Omron CX-Programmer project 新工程 (CX-Programmer 9.61)

# PLC 负压入盘机: CJ2M CPU33
I/O table (CPU CJ2M-CPU33): rack 0 slot 0 CJ1W-SCU21-V1; rack 0 slot 1 CJ1W-NC413; rack 0 slot 2 CJ1W-ID261; rack 0 slot 3 CJ1W-ID261; rack 0 slot 4 CJ1W-ID261; rack 0 slot 5 CJ1W-OD261; rack 0 slot 6 CJ1W-OD231; rack 0 slot 11 CJ2M-EIP21

## Global symbols (name address type ; comment)
17.10 BOOL  ; 料盘夹紧气缸伸出
2.13 BOOL  ; 料盒夹紧气缸伸出到位
0.00 BOOL  ; #3检漏仪行程1
0.01 BOOL  ; 上料有料感应
0.02 BOOL  ; 移栽前电池到位
0.03 BOOL  ; 移栽后电池到位
0.04 BOOL  ; #1模组左电池感应
0.05 BOOL  ; #1模组右电池感应
0.06 BOOL  ; #2模组左电池感应
0.07 BOOL  ; #2模组右电池感应
0.08 BOOL  ; #3模组左电池感应
0.09 BOOL  ; #3模组右电池感应
0.10 BOOL  ; #4模组左电池感应
0.11 BOOL  ; #4模组右电池感应
0.12 BOOL  ; #2空料盒到位感应
0.13 BOOL  ; 上料盒完成按钮（左）
0.14 BOOL  ; 龙门升降料盒到位
0.15 BOOL  ; #2满料盒到位感应
1000 CHANNEL  ; 移栽自动步序
1000.00 BOOL  ; 移栽机构在初始位
1000.15 BOOL  ; 移栽自动运行结束(步)
100.00 BOOL  ; 前门已打开
100.01 BOOL  ; 后门已打开
100.02 BOOL  ; 左侧门已打开
100.03 BOOL  ; 右侧门已打开
100.04 BOOL  ; 电脑未连接
100.05 BOOL  ; 进料移栽没归零
100.06 BOOL  ; 左机械手没归零
100.07 BOOL  ; 右机械手没归零
100.08 BOOL  ; 龙门升降伺服没归零
100.09 BOOL  ; 龙门前后伺服没归零
100.10 BOOL  ; 龙门左右伺服没归零
100.11 BOOL  ; 料盒升降伺服没归零
100.12 BOOL  ; 右机械手左夹爪有料但没夹紧
100.13 BOOL  ; 右机械手左夹爪没张开
100.14 BOOL  ; 右机械手右夹爪有料但没夹紧
100.15 BOOL  ; 右机械手右夹爪没张开
101.00 BOOL  ; 左机械手左夹爪有料但没夹紧
101.01 BOOL  ; 左机械手左夹爪没张开
101.02 BOOL  ; 左机械手右夹爪有料但没夹紧
101.03 BOOL  ; 左机械手右夹爪没张开
101.04 BOOL  ; #1模组左密封气缸没缩回
101.05 BOOL  ; #1模组右密封气缸没缩回
101.06 BOOL  ; #1模组左夹料气缸没松开
101.07 BOOL  ; #1模组右夹料气缸没松开
101.08 BOOL  ; #2模组左密封气缸没缩回
101.09 BOOL  ; #2模组右密封气缸没缩回
101.10 BOOL  ; #2模组左夹料气缸没松开
101.11 BOOL  ; #2模组右夹料气缸没松开
101.12 BOOL  ; #3模组左密封气缸没缩回
101.13 BOOL  ; #3模组右密封气缸没缩回
101.14 BOOL  ; #3模组左夹料气缸没松开
101.15 BOOL  ; #3模组右夹料气缸没松开
1020.00 BOOL  ; 移栽机构有错误
102.00 BOOL  ; #4模组左密封气缸没缩回
102.01 BOOL  ; #4模组右密封气缸没缩回
102.02 BOOL  ; #4模组左夹料气缸没松开
102.03 BOOL  ; #4模组右夹料气缸没松开
102.04 BOOL  ; 龙门夹爪没张开
102.05 BOOL  ; 龙门夹爪有料但没夹紧
103.00 BOOL  ; 移栽归零左机械手异常
103.01 BOOL  ; 移栽归零右机械手异常
103.02 BOOL  ; 移栽左移左机械手异常
103.03 BOOL  ; 移栽左移没归零异常
103.04 BOOL  ; 移栽左移左限位到达异常
103.05 BOOL  ; 移栽右移右机械手异常
103.06 BOOL  ; 移栽右移没归零异常
103.07 BOOL  ; 移栽右移右限位到达异常
103.08 BOOL  ; 移栽回进料位条件异常
103.09 BOOL  ; 移栽回进料位没归零异常
103.10 BOOL  ; 移栽回左下料位条件异常
103.11 BOOL  ; 移栽回左下料位没归零异常
103.12 BOOL  ; 移栽回右下料位条件异常
103.13 BOOL  ; 移栽回右下料没归零
104.00 BOOL  ; 左机械手升降气缸没缩回异常
104.01 BOOL  ; 左机械手伸缩气缸没缩回异常
104.02 BOOL  ; 左机械手没归零异常
104.03 BOOL  ; 伸缩气缸伸出异常
104.04 BOOL  ; 升降气缸伸出异常
104.05 BOOL  ; 左机械手夹爪松开升降气缸异常
104.06 BOOL  ; 左机械手夹爪松开伸缩气缸异常
104.07 BOOL  ; 左机械手左夹爪松开伸缩气缸异常
104.08 BOOL  ; 左机械手右夹爪松开升降气缸异常
104.09 BOOL  ; 左机械手右夹爪松开伸缩气缸异常
105.00 BOOL  ; 机械手升降气缸没缩回异常
105.01 BOOL  ; 右机械手伸缩气缸没缩回异常
105.02 BOOL  ; 右机械手没归零异常
105.03 BOOL  ; 伸缩气缸伸出异常
105.04 BOOL  ; 升降气缸伸出异常
105.05 BOOL  ; 右机械手夹爪松开升降气缸异常
106.00 BOOL  ; #1左密封气缸没缩回异常
106.01 BOOL  ; #1右密封气缸没缩回异常
106.04 BOOL  ; #2左密封气缸没缩回异常
106.05 BOOL  ; #2右密封气缸没缩回异常
106.08 BOOL  ; #3左密封气缸没缩回异常
106.09 BOOL  ; #3右密封气缸没缩回异常
106.12 BOOL  ; #4左密封气缸没缩回异常
106.13 BOOL  ; #4右密封气缸没缩回异常
107.00 BOOL  ; 龙门升降气缸没缩回异常
107.01 BOOL  ; 伺服没归零异常
107.02 BOOL  ; 料盒定位气缸没缩回
107.03 BOOL  ; 料盒升降下料处有料异常
107.04 BOOL  ; 伺服没归零异常
107.05 BOOL  ; 左、右脱离气缸没缩回异常
107.06 BOOL  ; 龙门升降气缸没缩回异常
107.07 BOOL  ; 龙门升降伺服不在原位
107.08 BOOL  ; 龙门前后、左右伺服没归零异常
107.09 BOOL  ; 龙门升降夹爪松开异常
107.10 BOOL  ; 此位有电池夹爪没打开不能下降
108.00 BOOL  ; 龙门升降气缸没缩回异常
10.00 BOOL  ; #1上顶升左气缸缩回位
10.01 BOOL  ; #1上顶升左气缸伸出位
10.02 BOOL  ; #1上顶升右气缸缩回位
10.03 BOOL  ; #1上顶升右气缸伸出位
10.04 BOOL  ; #2上顶升左气缸缩回位
10.05 BOOL  ; #2上顶升左气缸伸出位
10.06 BOOL  ; #2上顶升右气缸缩回位
10.07 BOOL  ; #2上顶升右气缸伸出位
10.08 BOOL  ; #1下顶升左气缸缩回位
10.09 BOOL  ; #1下顶升左气缸伸出位
10.10 BOOL  ; #1下顶升右气缸缩回位
10.11 BOOL  ; #1下顶升右气缸伸出位
10.12 BOOL  ; #2下顶升左气缸缩回位
10.13 BOOL  ; #2下顶升左气缸伸出位
10.14 BOOL  ; #2下顶升右气缸缩回位
10.15 BOOL  ; #2下顶升右气缸伸出位
11.00 BOOL  ; 叉车退出上对射
11.01 BOOL  ; 叉车退出下对射
11.02 BOOL  ; 右按钮（叉车伸出上到位）
11.03 BOOL  ; #1空料盒到位感应
11.04 BOOL  ; #2检漏仪行程1
11.05 BOOL  ; #2检漏仪行程0
11.06 BOOL  ; 上料盒区域1感应
11.07 BOOL  ; #2料盒区域感应
11.08 BOOL  ; 左拉带脱离气缸缩回位
11.09 BOOL  ; 左拉带脱离气缸伸出位
11.10 BOOL  ; 右拉带脱离气缸缩回位
11.11 BOOL  ; 右拉带脱离气缸伸出位
11.12 BOOL  ; 左#2放料电池感应
11.13 BOOL  ; 左#1放料电池感应
11.14 BOOL  ; 右#1放料电池感应
11.15 BOOL  ; 右#2放料电池感应
120.00 BOOL  ; 上料机构复位
120.01 BOOL  ; 上料机构在初始位
120.04 BOOL  ; 上料机构异常复位
120.05 BOOL  ; 上料机构异常复位完成
121.00 BOOL  ; 移栽机构复位
121.01 BOOL  ; 移栽伺服归零
121.02 BOOL  ; 移栽伺服到进料位置(复位)
121.03 BOOL  ; 移栽机构在初始位
121.04 BOOL  ; 移栽机构异常复位
121.05 BOOL  ; 移栽伺服异常归零
121.06 BOOL  ; 移栽伺服异常后到进料位置
121.07 BOOL  ; 移栽机构异常复位完成
121.10 BOOL  ; 龙门升降伺服异常复位
121.11 BOOL  ; 龙门升降伺服异常复位归零
121.12 BOOL  ; 龙门升降伺服异常归零后回上料盒位置
122.00 BOOL  ; 左机械手整机复位
122.01 BOOL  ; 左机械手伺服归零
122.02 BOOL  ; 左机械手回上料位(复位)
122.03 BOOL  ; 左机械手在初始位
122.04 BOOL  ; 左机械手异常复位
122.05 BOOL  ; 左机械手伺服异常归零
122.06 BOOL  ; 左机械手异常后回上料位
122.07 BOOL  ; 左机械手复位完成
123.00 BOOL  ; 右机械手复位
123.01 BOOL  ; 右机械手伺服归零
123.02 BOOL  ; 右机械手回上料位(复位)
123.03 BOOL  ; 右机械手在初始位
123.04 BOOL  ; 右机械手异常复位
123.05 BOOL  ; 右机械手伺服异常归零
123.06 BOOL  ; 右机械手伺服异常归零后回上料位
123.07 BOOL  ; 右机械手异常复位完成
124.00 BOOL  ; #1模组复位
124.01 BOOL  ; #1模组在初始位
124.02 BOOL  ; #2模组复位
124.03 BOOL  ; #2模组在初始位
124.04 BOOL  ; #3模组复位
124.05 BOOL  ; #3模组在初始位
124.06 BOOL  ; #4模组复位
124.07 BOOL  ; #4模组在初始位
124.08 BOOL  ; #1模组异常复位
124.09 BOOL  ; #1模组异常复位完成
124.10 BOOL  ; #2模组异常复位
124.11 BOOL  ; #2模组异常复位完成
124.12 BOOL  ; #3模组异常复位
124.13 BOOL  ; #3模组异常复位完成
124.14 BOOL  ; #4模组异常复位
124.15 BOOL  ; #4模组异常复位完成
125.00 BOOL  ; 龙门升降机构复位
125.01 BOOL  ; 龙门升降归零(复位)
125.02 BOOL  ; 龙门升降机构在初始位
125.03 BOOL  ; 龙门前后，左右复位
125.04 BOOL  ; 龙门前后伺服归零(复位)
125.05 BOOL  ; 龙门左右伺服归零(复位）
125.06 BOOL  ; 龙门前后，左右在初始位
125.08 BOOL  ; 龙门机构复位
125.09 BOOL  ; 料盒升降伺服整机归零
125.10 BOOL  ; 料盒升降回上料盒位置
125.11 BOOL  ; 龙门机构在初始位置
126.00 BOOL  ; 龙门升降异常复位
126.01 BOOL  ; 龙门升降伺服异常归零
126.02 BOOL  ; 龙门升降异常复位完成
126.05 BOOL  ; 龙门前后，左右异常复位
126.06 BOOL  ; 龙门前后异常复位归零
126.07 BOOL  ; 龙门左右异常复位归零
126.08 BOOL  ; 龙门前后，左右伺服异常复位完成
126.09 BOOL  ; 龙门升降伺服异常复位
126.10 BOOL  ; 料盒升降伺服异常复位归零
126.11 BOOL  ; 料盒升降伺服异常归零后回上料盒位置
126.12 BOOL  ; 料盒升降伺服异常复位完成
126.13 BOOL  ; 龙门机构异常复位
126.14 BOOL  ; 龙门机构异常复位完成
12.00 BOOL  ; 上料阻挡气缸
12.01 BOOL  ; 检测气缸
12.02 BOOL  ; 移栽阻挡气缸
12.03 BOOL  ; 左机械手升降气缸
12.04 BOOL  ; 左机械手伸缩气缸
12.05 BOOL  ; 左机械手左夹爪气缸
12.06 BOOL  ; 左机械手右夹爪气缸
12.07 BOOL  ; 右机械手升降气缸
12.08 BOOL  ; 右机械手伸缩气缸
12.09 BOOL  ; 右机械手左夹爪气缸
12.10 BOOL  ; 右机械手右夹爪气缸
12.11 BOOL  ; #1模组左夹料气缸
12.12 BOOL  ; #1模组右夹料气缸
12.13 BOOL  ; #1模组左密封气缸
12.14 BOOL  ; #1模组右密封气缸
12.15 BOOL  ; #1自检左气缸
134.15 BOOL  ; 移栽机构复位(M)
13.00 BOOL  ; #1自检右气缸
13.01 BOOL  ; #2模组左夹料气缸
13.02 BOOL  ; #2模组右夹料气缸
13.03 BOOL  ; #2模组左密封气缸
13.04 BOOL  ; #2模组右密封气缸
13.05 BOOL  ; #2自检左气缸
13.06 BOOL  ; #2自检右气缸
13.07 BOOL  ; #3左夹料气缸
13.08 BOOL  ; #3右夹料气缸
13.09 BOOL  ; #3左密封气缸
13.10 BOOL  ; #3右密封气缸
13.11 BOOL  ; #3自检左气缸
13.12 BOOL  ; #3自检右气缸
13.13 BOOL  ; #4左夹料气缸
13.14 BOOL  ; #4右夹料气缸
13.15 BOOL  ; #4左密封气缸
1404 CHANNEL  ; 第二排放料位置
1410.00 BOOL  ; 移栽机构在初始位
1410.01 BOOL  ; 前上料伺服在待机位置
1411.00 BOOL  ; 移栽机构有错误
1417 CHANNEL  ; 移栽自动步序
1417.15 BOOL  ; 移栽自动运行结束(步)
14.00 BOOL  ; #4右密封气缸
14.01 BOOL  ; #4自检左气缸
14.02 BOOL  ; #4自检右气缸
14.03 BOOL  ; 龙门#1上顶升气缸
14.04 BOOL  ; 龙门#2上顶升气缸
14.05 BOOL  ; #1下顶升气缸
14.06 BOOL  ; #2下顶升气缸
14.07 BOOL  ; 龙门料盒阻挡气缸
14.10 BOOL  ; 料盒定位气缸
14.11 BOOL  ; 龙门升降气缸
14.12 BOOL  ; 龙门夹爪气缸
14.13 BOOL  ; #1移栽电机
14.14 BOOL  ; #2移栽电机
14.15 BOOL  ; 检漏NG电机
1534.15 BOOL  ; 单元1的串口1协议执行标志
15.00 BOOL  ; 绝缘NG电机
15.01 BOOL  ; 料盒下料电机
15.02 BOOL  ; 下料缓存电机
15.03 BOOL  ; 料盒上料电机
15.04 BOOL  ; 真空泵
15.05 BOOL  ; 检测气缸
15.06 BOOL  ; 绝缘检测仪启动信号
15.07 BOOL  ; #1检漏仪启动
15.09 BOOL  ; #2检漏仪启动
15.11 BOOL  ; #3检漏仪启动
15.13 BOOL  ; #4检漏仪启动
15.14 BOOL  ; #4检漏仪启动
15.15 BOOL  ; 启动指示灯
16.00 BOOL  ; 停止指示灯
16.01 BOOL  ; 复位指示灯
16.02 BOOL  ; 三色绿灯
16.03 BOOL  ; 三色红灯
16.04 BOOL  ; 三色黄灯
16.05 BOOL  ; 蜂鸣器
16.06 BOOL  ; 移栽Serv_ON
16.08 BOOL  ; 左机械手Serv_ON
16.09 BOOL  ; 报警声关
16.10 BOOL  ; 右机械手Serv_ON
16.12 BOOL  ; 龙门升降Serv-ON
16.14 BOOL  ; 龙门左右Serv_ON
17.00 BOOL  ; 龙门前后Serv_ON
17.02 BOOL  ; 料盒Serv-ON
17.04 BOOL  ; 左拉带脱离气缸
17.05 BOOL  ; 右拉带脱离气缸
17.06 BOOL  ; 龙门升降刹车
17.07 BOOL  ; 料盒升降刹车
17.11 BOOL  ; 料盘夹紧气缸松开
18.00 BOOL  ; 扫描NG提示
19.00 BOOL  ; 左机械手左夹爪状态
19.01 BOOL  ; 左机械手右夹爪状态
19.02 BOOL  ; 右机械手左夹爪状态
19.03 BOOL  ; 右机械手右夹爪状态
1.00 BOOL  ; #1满料盒到位感应
1.01 BOOL  ; 入电池位料盒感应
1.02 BOOL  ; 料盒#1电池感应
1.03 BOOL  ; 料盒#2电池感应
1.04 BOOL  ; 料盒#3电池感应
1.05 BOOL  ; 料盒#4电池感应
1.06 BOOL  ; 料盒#5电池感应
1.07 BOOL  ; 料盒#6电池感应
1.08 BOOL  ; 料盒#7电池感应
1.09 BOOL  ; 料盒#8电池感应
1.10 BOOL  ; 料盒#9电池感应
1.11 BOOL  ; 料盒#10电池感应
1.12 BOOL  ; 料盒#11电池感应
1.13 BOOL  ; 料盒#12电池感应
1.14 BOOL  ; 料盒#13电池感应
1.15 BOOL  ; 料盒#14电池感应
2000.03 BOOL  ; 龙门前后绝对移动
2000.06 BOOL  ; 龙门前后归零
2000.09 BOOL  ; 龙门前后点动
2000.10 BOOL  ; 龙门前后方向
2000.12 BOOL  ; 龙门前后模块复位
2000.15 BOOL  ; 龙门前后停止
2002.03 BOOL  ; 龙门左右绝对运动
2002.06 BOOL  ; 龙门左右归零
2002.09 BOOL  ; 龙门左右点动
2002.10 BOOL  ; 龙门左右方向
2002.12 BOOL  ; 龙门左右模块复位
2002.15 BOOL  ; 龙门左右伺服停止
2004.03 BOOL  ; 料盒升降绝对移动
2004.06 BOOL  ; 料盒升降归零
2004.09 BOOL  ; 料盒升降点动
2004.10 BOOL  ; 料盒升降方向
2004.12 BOOL  ; 料盒升降模块复位
2004.15 BOOL  ; 料盒升降停止
2008.06 BOOL  ; 龙门前后无原点标志
2008.12 BOOL  ; 龙门前后模块有错误
2008.13 BOOL  ; 龙门前后忙标志
2009.08 BOOL  ; 龙门前后伺服前限位
2009.09 BOOL  ; 龙门前后伺服后限位
2009.10 BOOL  ; 前后近原点
2009.11 BOOL  ; 前后原点
200.00 BOOL  ; 复位位
2010 CHANNEL  ; 龙门前后轴错误代码
2011.06 BOOL  ; 龙门左右无原点标志
2011.12 BOOL  ; 龙门左右模块有错误
2011.13 BOOL  ; 龙门左右忙标志
2012.08 BOOL  ; 龙门左右伺服右限位
2012.09 BOOL  ; 龙门左右伺服左限位
2012.11 BOOL  ; 龙门左右原点
2013 CHANNEL  ; 龙门左右轴错误代码
2014.06 BOOL  ; 料盒升降无原点标志
2014.12 BOOL  ; 料盒升降模块有错误
2014.13 BOOL  ; 料盒升降忙标志
2015.08 BOOL  ; 料盒升降下限位
2015.09 BOOL  ; 料盒升降上限位
2016 CHANNEL  ; 料盒升降轴错误代码
20.00 BOOL  ; 移栽伺服手动回进料位置
20.01 BOOL  ; 移栽伺服手动回左下料位置
20.02 BOOL  ; 移栽伺服手动回右下料位置
20.03 BOOL  ; 移栽自动回右下料位
20.04 BOOL  ; 移栽自动回左下料位
20.05 BOOL  ; 移栽自动回上料位
21.00 BOOL  ; #1模组可放料
21.01 BOOL  ; #2模组可放料
21.02 BOOL  ; #3模组可放料
21.03 BOOL  ; #4模组可放料
21.04 BOOL  ; 回右下料位条件
21.05 BOOL  ; 回左下料位条件
22.00 BOOL  ; 左机械手上料位伸缩气缸伸出条件
22.01 BOOL  ; 左机械手下料位伸缩气缸伸出条件
22.02 BOOL  ; 左机械手#2模组伸缩气缸伸出条件
22.03 BOOL  ; 左机械手#4模组伸缩气缸伸出条件
22.04 BOOL  ; 左机械手伸缩气缸伸出条件
22.05 BOOL  ; 左机械手手动回上料位置
22.06 BOOL  ; 左机械手回下料位置
22.07 BOOL  ; 左机械手回#2位置
22.08 BOOL  ; 左机械手回#4位置
22.09 BOOL  ; 左机械手自动回上料位置
22.10 BOOL  ; 左机械手自动回#2位置
22.11 BOOL  ; 左机械手自动回#4位置
22.12 BOOL  ; 左机械手自动回下料位置
23 CHANNEL  ; 左机械手状态
235.02 BOOL  ; 右机械手升降气缸缩回
23.00 BOOL  ; 左机械手左夹爪上料处夹紧电池
23.01 BOOL  ; 左机械手上料处右夹爪夹紧到位
23.02 BOOL  ; 左机械手#2左放料
23.03 BOOL  ; 左机械手#4左放料
23.04 BOOL  ; 左机械手#2右放料
23.05 BOOL  ; 左机械手#4右放料
23.06 BOOL  ; 左机械手#2左取料
23.07 BOOL  ; 左机械手#2右取料
23.08 BOOL  ; 左机械手#4左取料
23.09 BOOL  ; 左机械手#4右取料
23.10 BOOL  ; 左机械手左夹爪有料状态
23.11 BOOL  ; 左机械手右夹爪有料状态
23.12 BOOL  ; 左机械手左夹爪模组放料完成
23.13 BOOL  ; 左机械手右夹爪模组放料完成
23.14 BOOL  ; 左机械手左夹爪上料处夹紧电池
23.15 BOOL  ; 左机械手上料处右夹爪夹紧到位
24.00 BOOL  ; 右机械手上料位伸缩气缸伸出条件
24.01 BOOL  ; 右机械手下料位伸缩气缸伸出条件
24.02 BOOL  ; 右机械手#1模组伸缩气缸伸出条件
24.03 BOOL  ; 右机械手#3模组伸缩气缸伸出条件
24.04 BOOL  ; 右机械手伸缩气缸伸出条件
24.05 BOOL  ; 右机械手手动回上料位置
24.06 BOOL  ; 右机械手回下料位置
24.07 BOOL  ; 右机械手回#1位置
24.08 BOOL  ; 右机械手回#3位置
24.09 BOOL  ; 右机械手自动回上料位置
24.10 BOOL  ; 右机械手自动回#1位置
24.11 BOOL  ; 右机械手回#3位置
24.12 BOOL  ; 右机械手自动回下料位
25 CHANNEL  ; 右机械手状态
25.00 BOOL  ; 右机械手右夹爪上料处夹紧电池
25.01 BOOL  ; 右机械手上料处左夹爪夹紧到位
25.02 BOOL  ; 右机械手#1左放料
25.03 BOOL  ; 右机械手#3左放料
25.04 BOOL  ; 右机械手#1右放料
25.05 BOOL  ; 右机械手#3右放料
25.06 BOOL  ; 右机械手#1左取料
25.07 BOOL  ; 右机械手#1右取料
25.08 BOOL  ; 右机械手#3左取料
25.09 BOOL  ; 右机械手#3右取料
25.10 BOOL  ; 右机械手左夹爪有料状态
25.11 BOOL  ; 右机械手右夹爪有料状态
25.12 BOOL  ; 右机械手左夹爪模组放料完成
25.13 BOOL  ; 右机械手右夹爪模组放料完成
25.14 BOOL  ; 右机械手右夹爪上料处夹紧电池
25.15 BOOL  ; 右机械手上料处左夹爪夹紧到位
2960.06 BOOL  ; 移栽伺服左限位
2960.07 BOOL  ; 移栽伺服右限位
2960.08 BOOL  ; 左机械手左限位
2960.09 BOOL  ; 左机械手右限位
2962.02 BOOL  ; 龙门升降原位
2962.06 BOOL  ; 右机械手左限位
2962.07 BOOL  ; 右机械手右限位
2962.08 BOOL  ; 龙门升降上限位
2962.09 BOOL  ; 龙门升降下限位
2.00 BOOL  ; 料盒#15电池感应
2.01 BOOL  ; 料盒#16电池感应
2.02 BOOL  ; 料盒#17电池感应
2.03 BOOL  ; 料盒#18电池感应
2.04 BOOL  ; 料盒#19电池感应
2.05 BOOL  ; 料盒#20电池感应
2.06 BOOL  ; 料盒#21电池感应
2.07 BOOL  ; 料盒#22电池感应
2.08 BOOL  ; 料盒#23电池感应
2.09 BOOL  ; 料盒#24电池感应
2.10 BOOL  ; 拉倒衔接处有料
2.11 BOOL  ; #1检漏仪行程1
2.12 BOOL  ; #1检漏仪行程0
2.14 BOOL  ; 绝缘NG放料位有料感应
2.15 BOOL  ; 检漏NG满
30.00 BOOL  ; #1检漏仪抽气临结束状态
30.01 BOOL  ; #2检漏仪抽气临结束状态
30.02 BOOL  ; #3检漏仪抽气临结束状态
30.03 BOOL  ; #4检漏仪抽气临结束状态
30.04 BOOL  ; #1#3模组不在抽气临结束状态
30.05 BOOL  ; #2#4模组不在抽气临结束状态
30.06 BOOL  ; #1模组在保压状态
30.07 BOOL  ; #1模组在保压1秒范围
30.08 BOOL  ; #1仪器抽气状态
311.00 BOOL  ; 整机复位条件
311.01 BOOL  ; 整机复位
311.02 BOOL  ; 整机在初始位
311.03 BOOL  ; 移栽机构复位
311.04 BOOL  ; 左机械手复位
311.05 BOOL  ; 右机械手复位
311.06 BOOL  ; #1模组异常复位
311.07 BOOL  ; #2模组复位
311.08 BOOL  ; #3模组复位
311.09 BOOL  ; #4模组复位
311.10 BOOL  ; 龙门升降复位
311.11 BOOL  ; 龙门前后，左右复位
311.12 BOOL  ; 龙门机构复位
311.13 BOOL  ; 上料机构复位
311.14 BOOL  ; 整机在初始位
313.00 BOOL  ; 移栽机构异常复位
313.01 BOOL  ; 左机械式异常复位
313.02 BOOL  ; 右机械式异常复位
313.03 BOOL  ; #1模组异常复位
313.04 BOOL  ; #2模组异常复位
313.05 BOOL  ; #3模组异常复位
313.06 BOOL  ; #4模组异常复位
313.07 BOOL  ; 龙门机构异常复位
313.08 BOOL  ; 龙门升降异常复位
313.09 BOOL  ; 龙门前后，左右伺服异常复位
313.10 BOOL  ; 料盒升降伺服异常复位
313.11 BOOL  ; 上料机构异常复位
31.00 BOOL  ; #2检漏仪抽气临结束状态
31.01 BOOL  ; #2检漏仪保压临结束状态
31.02 BOOL  ; #3检漏仪保压临结束状态
31.03 BOOL  ; #4检漏仪保压临结束状态
31.06 BOOL  ; #2模组在保压状态
31.07 BOOL  ; #2模组在保压1秒范围
31.08 BOOL  ; #2仪器抽气状态
32.00 BOOL  ; #3检漏仪抽气临结束状态
32.06 BOOL  ; #3模组在保压状态
32.07 BOOL  ; #3模组在保压1秒范围
32.08 BOOL  ; #3仪器抽气状态
33.00 BOOL  ; #4检漏仪抽气临结束状态
33.06 BOOL  ; #4模组在保压状态
33.07 BOOL  ; #4模组在保压1秒范围
33.08 BOOL  ; #4仪器抽气状态
34.00 BOOL  ; 龙门升降手动回取料位
34.01 BOOL  ; 龙门升降手动回OK放料位
34.02 BOOL  ; 龙门升降手动回绝缘NG位置
34.03 BOOL  ; 龙门升降手动回检漏NG位置
34.04 BOOL  ; 料盒升降伺服回上料盒位置
34.05 BOOL  ; 料盒升降伺服回放料盒位置
34.06 BOOL  ; 龙门升降自动回初始位置
34.07 BOOL  ; 龙门升降自动回取料位
34.08 BOOL  ; 龙门升降自动回OK放料位
34.09 BOOL  ; 龙门升降自动回绝缘NG位置
34.10 BOOL  ; 龙门升降在原始位置
34.11 BOOL  ; 龙门升降自动回检漏NG位置
35.00 BOOL  ; 龙门前后在#1位置
35.01 BOOL  ; 龙门前后在#2位置
35.02 BOOL  ; 龙门前后在#3位置
35.03 BOOL  ; 龙门前后在#4位置
35.04 BOOL  ; 龙门前后在#5位置
35.05 BOOL  ; 龙门前后在#6位置
35.06 BOOL  ; 龙门前后在#7位置
35.07 BOOL  ; 龙门前后在#8位置
35.08 BOOL  ; 龙门前后在#9位置
35.09 BOOL  ; 龙门前后在#10位置
35.10 BOOL  ; 龙门前后在#11位置
35.11 BOOL  ; 龙门前后在#12位置
35.12 BOOL  ; 龙门前后在#13位置
35.13 BOOL  ; 龙门前后在#14位置
35.14 BOOL  ; 龙门前后在#15位置
35.15 BOOL  ; 龙门前后在#16位置
36.00 BOOL  ; 龙门前后在#17位置
36.01 BOOL  ; 龙门前后在#18位置
36.02 BOOL  ; 龙门前后在#19位置
36.03 BOOL  ; 龙门前后在#20位置
36.04 BOOL  ; 龙门前后在#21位置
36.05 BOOL  ; 龙门前后在#22位置
36.06 BOOL  ; 龙门前后在#23位置
36.07 BOOL  ; 龙门前后在#24位置
36.08 BOOL  ; 龙门前后在#1左取料位
36.09 BOOL  ; 龙门前后在#2左取料位
36.10 BOOL  ; 龙门前后在#1右取料位
36.11 BOOL  ; 龙门前后在#2右取料位
36.12 BOOL  ; 龙门前后在绝缘NG位置
36.13 BOOL  ; 龙门前后在检漏NG位置
36.14 BOOL  ; 龙门前后在初始位置
37.00 BOOL  ; 龙门左右在#1位置
37.01 BOOL  ; 龙门左右在#2位置
37.02 BOOL  ; 龙门左右在#3位置
37.03 BOOL  ; 龙门左右在#4位置
37.04 BOOL  ; 龙门左右在#5位置
37.05 BOOL  ; 龙门左右在#6位置
37.06 BOOL  ; 龙门左右在#7位置
37.07 BOOL  ; 龙门左右在#8位置
37.08 BOOL  ; 龙门左右在#9位置
37.09 BOOL  ; 龙门左右在#10位置
37.10 BOOL  ; 龙门左右在#11位置
37.11 BOOL  ; 龙门左右在#12位置
37.12 BOOL  ; 龙门左右在#13位置
37.13 BOOL  ; 龙门左右在#14位置
37.14 BOOL  ; 龙门左右在#15位置
37.15 BOOL  ; 龙门左右在#16位置
38.00 BOOL  ; 龙门左右在#17位置
38.01 BOOL  ; 龙门左右在#18位置
38.02 BOOL  ; 龙门左右在#19位置
38.03 BOOL  ; 龙门左右在#20位置
38.04 BOOL  ; 龙门左右在#21位置
38.05 BOOL  ; 龙门左右在#22位置
38.06 BOOL  ; 龙门左右在#23位置
38.07 BOOL  ; 龙门左右在#24位置
38.08 BOOL  ; 龙门左右在#1左取料位
38.09 BOOL  ; 龙门左右在#2左取料位
38.10 BOOL  ; 龙门左右在#1右取料位
38.11 BOOL  ; 龙门左右在#2右取料位
38.12 BOOL  ; 龙门左右在绝缘NG位置
38.13 BOOL  ; 龙门左右在检漏NG位置
38.14 BOOL  ; 龙门左右在初始位置
39 CHANNEL  ; 龙门XY位置
39.01 BOOL  ; 龙门XY在#1放料位置
39.02 BOOL  ; 龙门XY在#2放料位置
39.03 BOOL  ; 龙门XY在#3放料位置
39.04 BOOL  ; 龙门XY在#4放料位置
39.05 BOOL  ; 龙门XY在#5放料位置
39.06 BOOL  ; 龙门XY在#6放料位置
39.07 BOOL  ; 龙门XY在#7放料位置
39.08 BOOL  ; 龙门XY在#8放料位置
39.09 BOOL  ; 龙门XY在#9放料位置
39.10 BOOL  ; 龙门XY在#10放料位置
39.11 BOOL  ; 龙门XY在#11放料位置
39.12 BOOL  ; 龙门XY在#12放料位置
3.00 BOOL  ; 检漏NG放料位有料感应
3.01 BOOL  ; #3检漏仪行程0
3.02 BOOL  ; #1检漏仪完成
3.03 BOOL  ; #1检漏仪异常
3.04 BOOL  ; #1检漏仪Busy信号
3.05 BOOL  ; #1检漏仪OK信号
3.06 BOOL  ; #1检漏仪NG
3.07 BOOL  ; #2检漏仪完成
3.08 BOOL  ; #2检漏仪异常
3.09 BOOL  ; #2检漏仪Busy信号
3.10 BOOL  ; #2检漏仪OK信号
3.11 BOOL  ; #2检漏仪NG
3.12 BOOL  ; #3检漏仪完成
3.13 BOOL  ; #3检漏仪异常
3.14 BOOL  ; #3检漏仪Busy信号
3.15 BOOL  ; #3检漏仪OK信号
4000 CHANNEL  ; #1模组左边状态
4001 CHANNEL  ; #1模组右边状态
4002 CHANNEL  ; #2模组左边状态
4003 CHANNEL  ; #2模组右边状态
4004 CHANNEL  ; #3模组左边状态
4005 CHANNEL  ; #3模组右边状态
4006 CHANNEL  ; #4模组左边状态
4007 CHANNEL  ; #4模组右边状态
4008 CHANNEL  ; 移栽状态
4009 CHANNEL  ; 左机械手状态
4010 CHANNEL  ; 右机械手状态
4011 CHANNEL  ; 上料机构状态
40.01 BOOL  ; 龙门XY在#13放料位置
40.02 BOOL  ; 龙门XY在#14放料位置
40.03 BOOL  ; 龙门XY在#15放料位置
40.04 BOOL  ; 龙门XY在#16放料位置
40.05 BOOL  ; 龙门XY在#17放料位置
40.06 BOOL  ; 龙门XY在#18放料位置
40.07 BOOL  ; 龙门XY在#19放料位置
40.08 BOOL  ; 龙门XY在#20放料位置
40.09 BOOL  ; 龙门XY在#21放料位置
40.10 BOOL  ; 龙门XY在#22放料位置
40.11 BOOL  ; 龙门XY在#23放料位置
40.12 BOOL  ; 龙门XY在#24放料位置
41.00 BOOL  ; 料盒升降在上料盒位置
41.01 BOOL  ; 料盒升降在放料盒位置
41.02 BOOL  ; 料盒升降在夹紧位置
42.00 BOOL  ; 龙门升降气缸下降条件
42.01 BOOL  ; 龙门升降夹爪夹紧、张开条件
42.02 BOOL  ; 右#2抓料特例
42.03 BOOL  ; 都无料回左#1待机
42.05 BOOL  ; 龙门XY在左#1取料位置
42.06 BOOL  ; 龙门XY在左#2取料位置
42.07 BOOL  ; 龙门XY在右#1取料位置
42.08 BOOL  ; 龙门XY在右#2取料位置
42.09 BOOL  ; 龙门XY在绝缘NG放料位置
42.10 BOOL  ; 龙门XY在检漏NG放料位置
43 CHANNEL  ; 上料盒状态
43.00 BOOL  ; #2下顶升气缸输出
43.01 BOOL  ; #1下顶升气缸输出
43.02 BOOL  ; #1下顶升气缸正常放料
43.03 BOOL  ; #1下顶升气缸缩回
43.04 BOOL  ; #2下顶升气缸正常放料
43.05 BOOL  ; #2下顶升气缸缩回
43.06 BOOL  ; 上料盒电机启动
44.00 BOOL  ; 料盒升降回放料盒位置
44.01 BOOL  ; 料盒升降自动回上料盒位置
44.02 BOOL  ; 左右拉带脱离气缸输出
44.03 BOOL  ; 料盒定位气缸输出
44.04 BOOL  ; 缓存电机启动
44.05 BOOL  ; 下料盒电机启动
44.06 BOOL  ; #2上顶升气缸伸出
44.07 BOOL  ; 料盒阻挡气缸伸出
44.08 BOOL  ; #1上顶升气缸伸出
44.09 BOOL  ; 绝缘NG电机启动
44.10 BOOL  ; 检漏NG电机启动
44.11 BOOL  ; 龙门回左#1抓料
44.12 BOOL  ; 龙门回左#2抓料
44.13 BOOL  ; 龙门回右#1抓料
44.14 BOOL  ; 龙门回右#2抓料
45.01 BOOL  ; 龙门回绝缘NG位
45.02 BOOL  ; 龙门回检测NG位
45.04 BOOL  ; 龙门XY到达绝缘NG位置
45.05 BOOL  ; 龙门XY到达检测NG位置
45.06 BOOL  ; 放料位判断完成
45.07 BOOL  ; 检漏电机走
45.08 BOOL  ; 绝缘NG电机走
46 CHANNEL  ; 龙门第一排位置
46.01 BOOL  ; 龙门回第一排#1位置
46.02 BOOL  ; 龙门回第一排#2位置
46.03 BOOL  ; 龙门回第一排#3位置
46.04 BOOL  ; 龙门回第一排#4位置
46.05 BOOL  ; 龙门回第一排#5位置
46.06 BOOL  ; 龙门回第一排#6位置
46.07 BOOL  ; 龙门回第一排#7位置
46.08 BOOL  ; 龙门回第一排#8位置
46.09 BOOL  ; 龙门回第一排#9位置
46.10 BOOL  ; 龙门回第一排#10位置
46.11 BOOL  ; 龙门回第一排#11位置
46.12 BOOL  ; 龙门回第一排#12位置
46.13 BOOL  ; 第一排#12位置有料
47 CHANNEL  ; 龙门第二排位置
47.00 BOOL  ; 第二排没料
47.01 BOOL  ; 龙门回第二排#1位置
47.02 BOOL  ; 龙门回第二排#2位置
47.03 BOOL  ; 龙门回第二排#3位置
47.04 BOOL  ; 龙门回第二排#4位置
47.05 BOOL  ; 龙门回第二排#5位置
47.06 BOOL  ; 龙门回第二排#6位置
47.07 BOOL  ; 龙门回第二排#7位置
47.08 BOOL  ; 龙门回第二排#8位置
47.09 BOOL  ; 龙门回第二排#9位置
47.10 BOOL  ; 龙门回第二排#10位置
47.11 BOOL  ; 龙门回第二排#11位置
47.12 BOOL  ; 龙门回第二排#12位置
48 CHANNEL  ; 龙门升降状态
48.00 BOOL  ; 龙门升降气缸输出
48.01 BOOL  ; 龙门升降回取料位置
48.02 BOOL  ; 龙门升降气缸缩回
48.03 BOOL  ; 龙门升降回原始位置
48.04 BOOL  ; 龙门升降回OK放料位置
48.05 BOOL  ; 龙门升降回绝缘NG放料位
48.06 BOOL  ; 龙门升降回检漏NG放料位
48.07 BOOL  ; 龙门升降到达指定位置
48.08 BOOL  ; 龙门升降放料完成
48.09 BOOL  ; 龙门升降回原点位置
4.00 BOOL  ; #3检漏仪NG
4.01 BOOL  ; #4检漏仪完成
4.02 BOOL  ; #4检漏仪异常
4.03 BOOL  ; #4检漏仪Busy信号
4.04 BOOL  ; #4检漏仪OK信号
4.05 BOOL  ; #4检漏仪NG
4.06 BOOL  ; 启动按钮
4.07 BOOL  ; 停止按钮
4.08 BOOL  ; 复位按钮
4.09 BOOL  ; 急停
4.10 BOOL  ; #4检漏仪行程1
4.11 BOOL  ; 后门磁感应
4.12 BOOL  ; 左门磁感应
4.13 BOOL  ; 右门磁感应
4.14 BOOL  ; 移栽Ready
4.15 BOOL  ; 移栽伺服Alarm
51.01 BOOL  ; 料盒#1电池感应
51.02 BOOL  ; 料盒#2电池感应
51.03 BOOL  ; 料盒#3电池感应
51.04 BOOL  ; 料盒#4电池感应
51.05 BOOL  ; 料盒#5电池感应
51.06 BOOL  ; 料盒#6电池感应
51.07 BOOL  ; 料盒#7电池感应
51.08 BOOL  ; 料盒#8电池感应
51.09 BOOL  ; 料盒#9电池感应
51.10 BOOL  ; 料盒#10电池感应
51.11 BOOL  ; 料盒#11电池感应
51.12 BOOL  ; 料盒#12电池感应
52.01 BOOL  ; 料盒#13电池感应
52.02 BOOL  ; 料盒#14电池感应
52.03 BOOL  ; 料盒#15电池感应
52.04 BOOL  ; 料盒#16电池感应
52.05 BOOL  ; 料盒#17电池感应
52.06 BOOL  ; 料盒#18电池感应
52.07 BOOL  ; 料盒#19电池感应
52.08 BOOL  ; 料盒#16电池感应
52.09 BOOL  ; 料盒#21电池感应
52.10 BOOL  ; 料盒#22电池感应
52.11 BOOL  ; 料盒#23电池感应
52.12 BOOL  ; 料盒#24电池感应
5.00 BOOL  ; 左机械手Ready
5.01 BOOL  ; 左机械手伺服报警
5.02 BOOL  ; 右机械手Ready
5.03 BOOL  ; 右机械手伺服报警信号
5.04 BOOL  ; 龙门升降Ready
5.05 BOOL  ; 龙门升降Alarm
5.06 BOOL  ; 龙门前后Ready
5.07 BOOL  ; 龙门前后Alarm
5.08 BOOL  ; 龙门左右Ready
5.09 BOOL  ; 龙门左右Alarm
5.10 BOOL  ; 料盒升降Ready
5.11 BOOL  ; 料盒升降Alarm
5.12 BOOL  ; 上料阻挡气缸缩回位
5.13 BOOL  ; 上料阻挡气缸伸出位
5.14 BOOL  ; 绝缘检测完成信号
5.15 BOOL  ; #4检漏仪行程0
60.01 BOOL  ; 移栽位记忆清除(HMI)
60.02 BOOL  ; 左机械手记忆清除(HMI)
60.03 BOOL  ; 右机械手记忆清除(HMI)
60.04 BOOL  ; #1模组记忆清除(HMI)
60.05 BOOL  ; #2模组记忆清除(HMI)
60.06 BOOL  ; #3模组记忆清除(HMI)
60.07 BOOL  ; #4模组记忆清除(HMI)
60.08 BOOL  ; 左下料位记忆清除(HMI)
60.09 BOOL  ; 右下料位记忆清除(HMI)
61.00 BOOL  ; 移栽位有料显示(HMI)
61.01 BOOL  ; 移栽位有料显示(HMI)
61.02 BOOL  ; 左机械手有料
61.03 BOOL  ; 右机械手有料显示(HMI)
61.04 BOOL  ; #1模组有料显示(HMI)
61.05 BOOL  ; #2模组有料显示(HMI)
61.06 BOOL  ; #3模组有料显示(HMI)
61.07 BOOL  ; #4模组有料显示(HMI)
61.08 BOOL  ; 左下料位有料显示(HMI)
61.09 BOOL  ; 右下料位有料显示(HMI)
6.00 BOOL  ; 检测气缸缩回位
6.01 BOOL  ; 检测气缸伸出位
6.02 BOOL  ; 移栽阻挡气缸缩回位
6.03 BOOL  ; 移栽阻挡气缸伸出位
6.04 BOOL  ; 左机械手升降气缸缩回位
6.05 BOOL  ; 左机械手升降气缸伸出位
6.06 BOOL  ; 左机械手伸缩气缸缩回位
6.07 BOOL  ; 左机械手伸缩气缸伸出位
6.08 BOOL  ; 左机械手左夹爪张开位
6.09 BOOL  ; 左机械手左夹爪夹紧位
6.10 BOOL  ; 左机械手右夹爪张开位
6.11 BOOL  ; 左机械手右夹爪夹紧位
6.12 BOOL  ; 右机械手升降气缸缩回位
6.13 BOOL  ; 右机械手升降气缸伸出位
6.14 BOOL  ; 右机械手伸缩气缸缩回位
6.15 BOOL  ; 右机械手伸缩气缸伸出位
7.00 BOOL  ; 右机械手左夹爪张开位
7.01 BOOL  ; 右机械手左夹爪夹紧位
7.02 BOOL  ; 右机械手右夹爪张开位
7.03 BOOL  ; 右机械手右夹爪夹紧位
7.04 BOOL  ; #1模组左密封气缸缩回位
7.05 BOOL  ; #1模组左密封气缸伸出位
7.06 BOOL  ; #1模组右密封气缸缩回位
7.07 BOOL  ; #1模组右密封气缸伸出位
7.08 BOOL  ; #1模组左夹料气缸缩回位
7.09 BOOL  ; #1模组左夹料气缸夹紧位
7.10 BOOL  ; #1模组右夹料气缸缩回位
7.11 BOOL  ; #1模组右夹料气缸夹紧位
7.12 BOOL  ; #2模组左密封气缸缩回位
7.13 BOOL  ; #2模组左密封气缸伸出位
7.14 BOOL  ; #2模组右密封气缸缩回位
7.15 BOOL  ; #2模组右密封气缸伸出位
8.00 BOOL  ; #2模组左夹料气缸张开位
8.01 BOOL  ; #2模组左夹料气缸夹紧位
8.02 BOOL  ; #2模组右夹料气缸张开位
8.03 BOOL  ; #2模组右夹料气缸夹紧位
8.04 BOOL  ; #3左密封气缸缩回位
8.05 BOOL  ; #3左密封气缸伸出位
8.06 BOOL  ; #3右密封气缸缩回位
8.07 BOOL  ; #3右密封气缸伸出位
8.08 BOOL  ; #3左夹料气张开位
8.09 BOOL  ; #3左夹料气夹紧位
8.10 BOOL  ; #3右夹料气张开位
8.11 BOOL  ; #3右夹料气夹紧位
8.12 BOOL  ; #4左密封气缸缩回位
8.13 BOOL  ; #4左密封气缸伸出位
8.14 BOOL  ; #4右密封气缸缩回位
8.15 BOOL  ; #4右密封气缸伸出位
9 CHANNEL  ; 龙门前后、左右手动按钮状态
9.00 BOOL  ; #4左夹料气缸张开位
9.01 BOOL  ; #4左夹料气缸夹紧位
9.02 BOOL  ; #4右夹料气缸张开位
9.03 BOOL  ; #4右夹料气缸夹紧位
9.04 BOOL  ; 龙门升降气缸缩回位
9.05 BOOL  ; 龙门升降气缸伸出位
9.06 BOOL  ; 龙门夹爪张开位
9.07 BOOL  ; 龙门夹爪夹紧位
9.08 BOOL  ; 料盒定位气缸缩回位
9.09 BOOL  ; 料盒定位气缸伸出位
9.10 BOOL  ; 上料盒阻挡左气缸缩回位
9.11 BOOL  ; 上料盒阻挡左气缸伸出位
9.12 BOOL  ; 龙门料盒阻挡右气缸缩回位
9.13 BOOL  ; 龙门料盒阻挡右气缸伸出位
9.14 BOOL  ; 龙门柔性报警
9.15 BOOL  ; 料盒升降下料处有料
A202.01 BOOL  ; 通信端口1允许
A276 CHANNEL  ; 移栽伺服当前脉冲
A278 CHANNEL  ; 左机械手当前脉冲
A280.04 BOOL  ; 移栽伺服脉冲输出中
A280.05 BOOL  ; 移栽伺服原点标志
A281.04 BOOL  ; 左机械手脉冲输出中
A281.05 BOOL  ; 左机械手原点标志
A322 CHANNEL  ; 右机械手当前脉冲
A324 CHANNEL  ; 龙门升降当前脉冲
A326.04 BOOL  ; 右机械手脉冲输出中
A326.05 BOOL  ; 右机械手原点标示
A327.04 BOOL  ; 龙门升降脉冲输出中
A327.05 BOOL  ; 龙门升降原点标示
A351 CHANNEL  ; 系统时间(分秒)
A352 CHANNEL  ; 系统时间(日时)
A353 CHANNEL  ; 系统时间(年月)
A540.08 BOOL  ; 移栽伺服CW
A540.09 BOOL  ; 移栽伺服CCW
A541.08 BOOL  ; 左机械手CW
A541.09 BOOL  ; 左机械手CCW
A542.08 BOOL  ; 右机械手CW
A542.09 BOOL  ; 右机械手CCW
A543.08 BOOL  ; 龙门升降CW
A543.09 BOOL  ; 龙门升降CCW
D0 CHANNEL  ; 移栽伺服自动速度(mm)
D10 CHANNEL  ; 右下料位置(mm)
D100 CHANNEL  ; 龙门前后#11位置
D1000 CHANNEL  ; 龙门前后脉冲当量
D1002 CHANNEL  ; 龙门前后脉冲当量(浮点)
D1004 CHANNEL  ; 龙门前后当前脉冲(浮点)
D1008 CHANNEL  ; 龙门前后当前位置(mm)
D1010 CHANNEL  ; 料盒前后中心距
D1012 CHANNEL  ; 料盒前后中心距(浮点)
D1014 CHANNEL  ; 料盒纵向中心距
D1016 CHANNEL  ; 料盒纵向中心距(浮点)
D102 CHANNEL  ; 龙门前后#12位置
D1020 CHANNEL  ; #1横向偏移距离
D1022 CHANNEL  ; #2横向偏移距离
D1024 CHANNEL  ; #3横向偏移距离
D1026 CHANNEL  ; #4横向偏移距离
D1028 CHANNEL  ; #5横向偏移距离
D1030 CHANNEL  ; #6横向偏移距离
D1032 CHANNEL  ; #7横向偏移距离
D1034 CHANNEL  ; #8横向偏移距离
D1036 CHANNEL  ; #9横向偏移距离
D1038 CHANNEL  ; #10横向偏移距离
D104 CHANNEL  ; 龙门前后#13位置
D1040 CHANNEL  ; #11横向偏移距离
D1050 CHANNEL  ; 抽气时间设定值
D106 CHANNEL  ; 龙门前后#14位置
D1060 CHANNEL  ; 检漏仪保压时间设定值
D1061 CHANNEL  ; 检漏仪保压结束延时设定值
D108 CHANNEL  ; 龙门前后#15位置
D110 CHANNEL  ; 龙门前后#16位置
D1102 CHANNEL  ; 龙门前后自动速度脉冲(脉冲)
D1106 CHANNEL  ; 龙门前后手动速度脉冲
D112 CHANNEL  ; 龙门前后#17位置
D114 CHANNEL  ; 龙门前后#18位置
D1140 CHANNEL  ; 报警画面跳转
D1150 CHANNEL  ; #1模组测试时间
D1152 CHANNEL  ; #2模组测试时间
D1154 CHANNEL  ; #3模组测试时间
D1156 CHANNEL  ; #4模组测试时间
D116 CHANNEL  ; 龙门前后#19位置
D118 CHANNEL  ; 龙门前后#20位置
D120 CHANNEL  ; 龙门前后#21位置
D1200 CHANNEL  ; 龙门左右脉冲当量
D1202 CHANNEL  ; 龙门左右脉冲当量(浮点)
D1204 CHANNEL  ; 龙门左右当前位置
D1208 CHANNEL  ; 龙门左右当前位置(mm)
D1210 CHANNEL  ; 料盒左右中心距
D1212 CHANNEL  ; 料盒左右中心距(浮点)
D1214 CHANNEL  ; 料盒纵向中心距(浮点)
D1216 CHANNEL  ; 料盒左右中心距*100
D122 CHANNEL  ; 龙门前后#22位置
D1220 CHANNEL  ; #1左右偏移距离
D124 CHANNEL  ; 龙门前后#23位置
D126 CHANNEL  ; 龙门前后#24位置
D130 CHANNEL  ; 龙门左右自动速度
D1300 CHANNEL  ; 轴控制预留
D1302 CHANNEL  ; 龙门左右速度脉冲(浮点)
D1304 CHANNEL  ; 龙门左右运动状态
D1306 CHANNEL  ; 龙门左右手动速度脉冲(浮点)
D132 CHANNEL  ; 龙门左右点动速度
D134 CHANNEL  ; 龙门左右加速度
D136 CHANNEL  ; 龙门左右#1位置
D138 CHANNEL  ; 龙门左右#2位置
D14 CHANNEL  ; 左机械手自动速度
D140 CHANNEL  ; 龙门左右#3位置
D1400 CHANNEL  ; 料盒升降脉冲当量
D1402 CHANNEL  ; 料盒升降脉冲当量(浮点)
D1404 CHANNEL  ; 料盒升降当前位置
D1408 CHANNEL  ; 料盒升降当前位置(mm)
D142 CHANNEL  ; 龙门左右#4位置
D144 CHANNEL  ; 龙门左右#5位置
D146 CHANNEL  ; 龙门左右#6位置
D148 CHANNEL  ; 龙门左右#7位置
D149 CHANNEL  ; 报警延迟时间
D150 CHANNEL  ; 龙门左右#8位置
D1500 CHANNEL  ; 龙门XY点位
D1502 CHANNEL  ; 料盒升降速度脉冲(浮点)
D1504 CHANNEL  ; 龙门左右运动状态
D1506 CHANNEL  ; 料盒升降手动速度脉冲(浮点)
D152 CHANNEL  ; 龙门左右#9位置
D154 CHANNEL  ; 龙门左右#10位置
D156 CHANNEL  ; 龙门左右#11位置
D158 CHANNEL  ; 龙门左右#12位置
D16 CHANNEL  ; 左机械手手动速度(mm/s)
D160 CHANNEL  ; 龙门左右#13位置
D1602 CHANNEL  ; 龙门前后运动状态
D1604 CHANNEL  ; 龙门左右运动状态
D1606 CHANNEL  ; 龙门前后、左右手动按钮状态
D162 CHANNEL  ; 龙门左右#14位置
D164 CHANNEL  ; 龙门左右#15位置
D166 CHANNEL  ; 龙门左右#16位置
D168 CHANNEL  ; 龙门左右#17位置
D170 CHANNEL  ; 龙门左右#18位置
D172 CHANNEL  ; 龙门左右#19位置
D174 CHANNEL  ; 龙门左右#20位置
D176 CHANNEL  ; 龙门左右#21位置
D178 CHANNEL  ; 龙门左右#22位置
D18 CHANNEL  ; 左机械手加速度
D180 CHANNEL  ; 龙门左右#23位置
D1800 CHANNEL  ; 报警代码
D1802 CHANNEL  ; 设备状态
D1803 CHANNEL  ; 设备状态(存储)
D1804 CHANNEL  ; 设备状态变更
D1806 CHANNEL  ; 设备状态(存储)
D182 CHANNEL  ; 龙门左右#24位置
D184 CHANNEL  ; 伺服脉冲当量(浮点)
D186 CHANNEL  ; 上料机械手当前位置(mm)
D188 CHANNEL  ; 伺服脉冲当量
D190 CHANNEL  ; 电池条码长度
D192 CHANNEL  ; 电池条码字节数
D1920 CHANNEL  ; 系统时间(年)
D1922 CHANNEL  ; 系统时间(日)
D1924 CHANNEL  ; 系统时间(分)
D1930 CHANNEL  ; #2模组电池时间
D194 CHANNEL  ; 电池条码比较字节数
D1940 CHANNEL  ; #4模组电池时间
D1950 CHANNEL  ; 左机械手电池时间
D1960 CHANNEL  ; #1模组电池时间
D1970 CHANNEL  ; #3模组电池时间
D1980 CHANNEL  ; 右机械手模组电池时间
D1990 CHANNEL  ; #1模组自检状态
D1991 CHANNEL  ; #1模组自检结果 1:OK；2:NG
D1992 CHANNEL  ; #2模组自检状态
D1993 CHANNEL  ; #2模组自检结果 1:OK；2:NG
D1994 CHANNEL  ; #3模组自检状态
D1995 CHANNEL  ; #3模组自检结果 1:OK；2:NG
D1996 CHANNEL  ; #4模组自检状态
D1997 CHANNEL  ; #4模组自检结果 1:OK；2:NG
D2 CHANNEL  ; 移栽伺服手动伺服(mm)
D20 CHANNEL  ; 左机械手进料位置(mm)
D200 CHANNEL  ; 上料阻挡气缸缩回位延时
D2000 CHANNEL  ; 龙门前后#1左取料位脉冲(浮点)
D20004 CHANNEL  ; 龙门前后伺服I/O设置
D20005 CHANNEL  ; 龙门前后伺服归零模式
D20008 CHANNEL  ; 龙门前后伺服归零初始速度
D20010 CHANNEL  ; 龙门前后伺服原点搜索高速度
D20012 CHANNEL  ; 龙门前后伺服接近原点速度
D20020 CHANNEL  ; 龙门前后伺服归零加速度
D20022 CHANNEL  ; 龙门前后伺服减速度
D20032 CHANNEL  ; 龙门左右伺服I/O设置
D20033 CHANNEL  ; 龙门左右伺服归零模式
D20036 CHANNEL  ; 龙门左右伺服归零初始速度
D20038 CHANNEL  ; 龙门左右伺服原点搜索高速度
D2004 CHANNEL  ; 龙门左右#2左取料位脉冲(浮点)
D20040 CHANNEL  ; 龙门左右伺服接近原点速度
D20048 CHANNEL  ; 龙门左右伺服归零加速度
D20050 CHANNEL  ; 龙门左右伺服减速度
D20060 CHANNEL  ; 料盒升降伺服I/O设置
D20061 CHANNEL  ; 料盒升降伺服归零模式
D20064 CHANNEL  ; 料盒升降伺服归零初始速度
D20066 CHANNEL  ; 料盒升降伺服原点搜索高速度
D20068 CHANNEL  ; 料盒升降伺服接近原点速度
D20076 CHANNEL  ; 料盒升降伺服归零加速度
D20078 CHANNEL  ; 料盒升降伺服减速度
D2008 CHANNEL  ; 龙门前后#1右取料位脉冲(浮点)
D2010 CHANNEL  ; 龙门前后轴错误
D2012 CHANNEL  ; 龙门前后#2右取料脉冲(浮点)
D20124 CHANNEL  ; 龙门前后运动位置
D20126 CHANNEL  ; 龙门前后伺服速度
D20128 CHANNEL  ; 龙门前后伺服加速度
D2013 CHANNEL  ; 龙门左右轴错误代码
D20130 CHANNEL  ; 龙门前后伺服减速度
D20132 CHANNEL  ; 龙门左右手动速度
D20136 CHANNEL  ; 龙门左右运动位移
D20138 CHANNEL  ; 龙门左右伺服速度
D20140 CHANNEL  ; 龙门左右加速度
D20142 CHANNEL  ; 龙门左右减速度
D20148 CHANNEL  ; 料盒升降运动位置
D20150 CHANNEL  ; 料盒升降伺服速度
D20152 CHANNEL  ; 料盒升降加速度
D20154 CHANNEL  ; 料盒升降加速度
D2016 CHANNEL  ; 龙门前后#1取料位置脉冲(浮点)
D20172 CHANNEL  ; 龙门前后当前脉冲
D20176 CHANNEL  ; 龙门左右当前脉冲
D20180 CHANNEL  ; 料盒升降当前脉冲
D202 CHANNEL  ; 上料阻挡气缸伸出到位延时
D2020 CHANNEL  ; 龙门前后#2取料位置脉冲(浮点)
D2024 CHANNEL  ; 龙门前后#3取料位置脉冲(浮点)
D2028 CHANNEL  ; 龙门前后#4取料位置脉冲(浮点)
D2032 CHANNEL  ; 龙门前后#5取料位置脉冲(浮点)
D2036 CHANNEL  ; 龙门前后#6取料位置脉冲(浮点)
D204 CHANNEL  ; 上料定位气缸缩回位延时
D2040 CHANNEL  ; 龙门前后#7取料位置脉冲(浮点)
D2044 CHANNEL  ; 龙门前后#8取料位置脉冲(浮点)
D2048 CHANNEL  ; 龙门前后#9取料位置脉冲(浮点)
D2052 CHANNEL  ; 龙门前后#10取料位置脉冲(浮点)
D2056 CHANNEL  ; 龙门前后#11取料位置脉冲(浮点)
D206 CHANNEL  ; 上料定位气缸伸出位延时
D2060 CHANNEL  ; 龙门前后#12取料位置脉冲(浮点)
D2064 CHANNEL  ; 龙门前后#13取料位置脉冲(浮点)
D2068 CHANNEL  ; 龙门前后#14取料位置脉冲(浮点)
D2072 CHANNEL  ; 龙门前后#15取料位置脉冲(浮点)
D2076 CHANNEL  ; 龙门前后#16取料位置脉冲(浮点)
D208 CHANNEL  ; 检测气缸缩回位延时
D2080 CHANNEL  ; 龙门前后#17取料位置脉冲(浮点)
D2084 CHANNEL  ; 龙门前后#18取料位置脉冲(浮点)
D2088 CHANNEL  ; 龙门前后#19取料位置脉冲(浮点)
D2092 CHANNEL  ; 龙门前后#20取料位置脉冲(浮点)
D2096 CHANNEL  ; 龙门前后#21取料位置脉冲(浮点)
D210 CHANNEL  ; 检测气缸伸出位延时
D2100 CHANNEL  ; 龙门前后#22取料位置脉冲(浮点)
D2104 CHANNEL  ; 龙门前后#23取料位置脉冲(浮点)
D2106 CHANNEL  ; 前上料伺服手动启动速度
D2108 CHANNEL  ; 龙门前后#24取料位置脉冲(浮点)
D2112 CHANNEL  ; 龙门前后绝缘NG位置脉冲(浮点)
D2116 CHANNEL  ; 龙门前后检漏NG位置脉冲(浮点)
D212 CHANNEL  ; 移栽阻挡气缸缩回位延时
D214 CHANNEL  ; 移栽阻挡气缸伸出位延时
D216 CHANNEL  ; 左机械手升降气缸缩回延时
D218 CHANNEL  ; 左机械手升降气缸伸出延时
D22 CHANNEL  ; 左机械手出料位置(mm）
D220 CHANNEL  ; 左机械手伸缩气缸缩回延时
D2200 CHANNEL  ; 龙门左右#1左取料位脉冲(浮点)
D2204 CHANNEL  ; 龙门左右#2左取料位脉冲(浮点)
D2208 CHANNEL  ; 龙门左右#1右取料脉冲(浮点)
D2212 CHANNEL  ; 龙门左右#2右取料脉冲(浮点)
D2216 CHANNEL  ; 龙门左右#1取料位脉冲(浮点)
D222 CHANNEL  ; 左机械手伸缩气缸伸出延时
D2220 CHANNEL  ; 龙门左右#2取料位脉冲(浮点)
D2224 CHANNEL  ; 龙门左右#3取料位脉冲(浮点)
D2228 CHANNEL  ; 龙门左右#4取料位脉冲(浮点)
D2232 CHANNEL  ; 龙门左右#5取料位脉冲(浮点)
D2236 CHANNEL  ; 龙门左右#6取料位脉冲(浮点)
D224 CHANNEL  ; 左机械手左夹爪张开位延时
D2240 CHANNEL  ; 龙门左右#7取料位脉冲(浮点)
D2244 CHANNEL  ; 龙门左右#8取料位脉冲(浮点)
D2248 CHANNEL  ; 龙门左右#9取料位脉冲(浮点)
D2252 CHANNEL  ; 龙门左右#10取料位脉冲(浮点)
D2256 CHANNEL  ; 龙门左右#11取料位脉冲(浮点)
D226 CHANNEL  ; 左机械手左夹爪夹紧位延时
D2260 CHANNEL  ; 龙门左右#12取料位脉冲(浮点)
D2264 CHANNEL  ; 龙门左右#13取料位脉冲(浮点)
D2268 CHANNEL  ; 龙门左右#14取料位脉冲(浮点)
D2272 CHANNEL  ; 龙门左右#15取料位脉冲(浮点)
D2276 CHANNEL  ; 龙门左右#16取料位脉冲(浮点)
D228 CHANNEL  ; 左机械手右夹爪张开位延时
D2280 CHANNEL  ; 龙门左右#17取料位脉冲(浮点)
D2284 CHANNEL  ; 龙门左右#18取料位脉冲(浮点)
D2288 CHANNEL  ; 龙门左右#19取料位脉冲(浮点)
D2292 CHANNEL  ; 龙门左右#20取料位脉冲(浮点)
D2294 CHANNEL  ; 龙门左右#21取料位脉冲(浮点)
D2296 CHANNEL  ; 龙门左右#21取料位脉冲(浮点)
D230 CHANNEL  ; 左机械手右夹爪夹紧位延时
D2300 CHANNEL  ; 龙门左右#22取料位脉冲(浮点)
D2304 CHANNEL  ; 龙门左右#23取料位脉冲(浮点)
D2308 CHANNEL  ; 龙门左右#24取料位脉冲(浮点)
D2312 CHANNEL  ; 龙门左右绝缘NG位脉冲(浮点)
D2316 CHANNEL  ; 龙门左右检漏NG位脉冲(浮点)
D232 CHANNEL  ; 右机械手升降气缸缩回延时
D234 CHANNEL  ; 右机械手升降气缸伸出延时
D236 CHANNEL  ; 右机械手伸缩气缸缩回延时
D238 CHANNEL  ; 右机械手伸缩气缸伸出延时
D24 CHANNEL  ; 左机械手#2进料位置(mm)
D240 CHANNEL  ; 右机械手左夹爪张开位延时
D2400 CHANNEL  ; 料盒升降上料盒位置脉冲(浮点)
D2404 CHANNEL  ; 料盒升降下料盒位置脉冲(浮点)
D242 CHANNEL  ; 右机械手左夹爪夹紧位延时
D244 CHANNEL  ; 右机械手右夹爪张开位延时
D246 CHANNEL  ; 右机械手右夹爪夹紧位延时
D248 CHANNEL  ; #1模组左密封气缸缩回延时
D250 CHANNEL  ; #1模组左密封气缸伸出延时
D2500 CHANNEL  ; 龙门左右#1取料位脉冲
D2502 CHANNEL  ; 龙门左右#2取料位脉冲
D2504 CHANNEL  ; 龙门左右#3取料位脉冲
D2506 CHANNEL  ; 龙门左右#4取料位脉冲
D2508 CHANNEL  ; 龙门左右#5取料位脉冲
D2510 CHANNEL  ; 龙门左右#6取料位脉冲
D2512 CHANNEL  ; 龙门左右#7取料位脉冲
D2514 CHANNEL  ; 龙门左右#8取料位脉冲
D2516 CHANNEL  ; 龙门左右#9取料位脉冲
D2518 CHANNEL  ; 龙门左右#10取料位脉冲
D252 CHANNEL  ; #1模组右密封气缸缩回延时
D2520 CHANNEL  ; 龙门左右#11取料位脉冲
D2522 CHANNEL  ; 龙门左右#12取料位脉冲
D2524 CHANNEL  ; 龙门左右#13取料位脉冲
D2526 CHANNEL  ; 龙门左右#14取料位脉冲
D2528 CHANNEL  ; 龙门左右#15取料位脉冲
D2530 CHANNEL  ; 龙门左右#16取料位脉冲
D2532 CHANNEL  ; 龙门左右#17取料位脉冲
D2534 CHANNEL  ; 龙门左右#18取料位脉冲
D2536 CHANNEL  ; 龙门左右#19取料位脉冲
D2538 CHANNEL  ; 龙门左右#20取料位脉冲
D254 CHANNEL  ; #1模组右密封气缸伸出延时
D2540 CHANNEL  ; 龙门左右#21取料位脉冲
D2542 CHANNEL  ; 龙门左右#22取料位脉冲
D2544 CHANNEL  ; 龙门左右#23取料位脉冲
D2546 CHANNEL  ; 龙门左右#24取料位脉冲
D256 CHANNEL  ; #1模组左夹电池张开位延时
D258 CHANNEL  ; #1模组左夹电池夹紧位延时
D26 CHANNEL  ; 左机械手#4位置(mm）
D260 CHANNEL  ; #1模组右夹电池张开位延时
D2600 CHANNEL  ; 龙门左右#1左取料位脉冲
D2602 CHANNEL  ; 龙门左右#2左取料位脉冲
D2604 CHANNEL  ; 龙门左右#1右取料脉冲
D2606 CHANNEL  ; 龙门左右#2右取料脉冲
D2608 CHANNEL  ; 龙门左右#1取料位脉冲
D262 CHANNEL  ; #1模组右夹电池夹紧位延时
D264 CHANNEL  ; #2模组左密封气缸缩回延时
D266 CHANNEL  ; #2模组左密封气缸伸出延时
D268 CHANNEL  ; #2模组右密封气缸缩回延时
D270 CHANNEL  ; #2模组右密封气缸伸出延时
D272 CHANNEL  ; #2模组左夹电池张开位延时
D274 CHANNEL  ; #2模组左夹电池夹紧位延时
D276 CHANNEL  ; #2模组右夹电池张开位延时
D278 CHANNEL  ; #2模组右夹电池夹紧位延时
D280 CHANNEL  ; #3模组左密封气缸缩回延时
D282 CHANNEL  ; #3模组左密封气缸伸出延时
D284 CHANNEL  ; #3模组右密封气缸缩回延时
D286 CHANNEL  ; #3模组右密封气缸伸出延时
D288 CHANNEL  ; #3模组左夹电池张开位延时
D290 CHANNEL  ; #3模组左夹电池夹紧位延时
D292 CHANNEL  ; #3模组右夹电池张开位延时
D294 CHANNEL  ; #3模组右夹电池夹紧位延时
D296 CHANNEL  ; #4模组左密封气缸缩回延时
D298 CHANNEL  ; #4模组左密封气缸伸出延时
D30 CHANNEL  ; 右机械手自动速度(mm)
D300 CHANNEL  ; #4模组右密封气缸缩回延时
D3000 CHANNEL  ; 托盘脱离料盒的距离
D3002 CHANNEL  ; 托盘脱离料盒的距离(浮点)
D3004 CHANNEL  ; 料盒下降安全距离
D3006 CHANNEL  ; 料盒下降安全距离
D3008 CHANNEL  ; 料盒脱离安全距离
D302 CHANNEL  ; #4模组右密封气缸伸出延时
D304 CHANNEL  ; #4模组左夹电池张开位延时
D306 CHANNEL  ; #4模组左夹电池夹紧位延时
D308 CHANNEL  ; #4模组右夹电池张开位延时
D310 CHANNEL  ; #4模组右夹电池夹紧位延时
D312 CHANNEL  ; 龙门升降气缸缩回位延时
D314 CHANNEL  ; 龙门升降气缸伸出位延时
D316 CHANNEL  ; 龙门夹爪气缸张开位延时
D318 CHANNEL  ; 龙门夹爪气缸夹紧位延时
D32 CHANNEL  ; 右机械手手动速度
D320 CHANNEL  ; 上料盒阻挡气缸缩回位延时
D322 CHANNEL  ; 上料盒阻挡气缸伸出位延时
D324 CHANNEL  ; #1上顶升左气缸缩回位延时
D326 CHANNEL  ; #1上顶升左气缸伸出位延时
D328 CHANNEL  ; #1上顶升右气缸缩回位延时
D330 CHANNEL  ; #1上顶升右气缸伸出位延时
D332 CHANNEL  ; #2上顶升左气缸缩回位延时
D334 CHANNEL  ; #2上顶升左气缸伸出位延时
D336 CHANNEL  ; #2上顶升右气缸缩回位延时
D338 CHANNEL  ; #2上顶升右气缸伸出位延时
D34 CHANNEL  ; 右机械手加速度
D340 CHANNEL  ; #1下顶升左气缸缩回位延时
D342 CHANNEL  ; #1下顶升左气缸伸出位延时
D344 CHANNEL  ; #1下顶升右气缸缩回位延时
D346 CHANNEL  ; #1下顶升右气缸伸出位延时
D348 CHANNEL  ; #2下顶升左气缸缩回位延时
D350 CHANNEL  ; #2下顶升左气缸伸出位延时
D352 CHANNEL  ; #2下顶升右气缸缩回位延时
D354 CHANNEL  ; #2下顶升右气缸伸出位延时
D356 CHANNEL  ; 上料阻挡右气缸缩回位时间
D358 CHANNEL  ; 上料盒阻挡右气缸伸出位时间
D36 CHANNEL  ; 右机械手进料位置(mm)
D360 CHANNEL  ; 左拉带脱离气缸缩回位时间
D362 CHANNEL  ; 左拉带脱离气缸伸出位时间
D364 CHANNEL  ; 右拉带脱离气缸缩回位时间
D366 CHANNEL  ; 右拉带脱离气缸伸出位时间
D368 CHANNEL  ; 料盒定位气缸缩回位时间
D370 CHANNEL  ; 料盒定位气缸伸出位时间
D372 CHANNEL  ; 龙门前后绝缘NG位置
D374 CHANNEL  ; 龙门前后检漏NG位置
D376 CHANNEL  ; 龙门左右绝缘NG位
D378 CHANNEL  ; 龙门左右检漏NG位置
D38 CHANNEL  ; 右机械手出料位置(mm)
D380 CHANNEL  ; #1左取料位置
D382 CHANNEL  ; #2左取料位置
D384 CHANNEL  ; #1右取料位置
D386 CHANNEL  ; #2右取料位置
D388 CHANNEL  ; 龙门左右#1左取料位置
D390 CHANNEL  ; 龙门左右#2左取料位置
D392 CHANNEL  ; 龙门左右#1右取料位置
D394 CHANNEL  ; 龙门左右#2右取料位置
D396 CHANNEL  ; 传感器到位延时
D398 CHANNEL  ; 报警延时时间
D4 CHANNEL  ; 移栽伺服加速度
D40 CHANNEL  ; 右机械手#1位置(mm)
D400 CHANNEL  ; 上料阻挡气缸缩回位延时
D4000 CHANNEL  ; #1模组状态
D4002 CHANNEL  ; #2模组状态
D4004 CHANNEL  ; #3模组状态
D4006 CHANNEL  ; #4模组状态
D402 CHANNEL  ; 上料阻挡气缸伸出到位延时
D404 CHANNEL  ; 上料定位气缸缩回位延时
D406 CHANNEL  ; 上料定位气缸伸出位延时
D408 CHANNEL  ; 检测气缸缩回位延时
D410 CHANNEL  ; 检测气缸伸出位延时
D4100 CHANNEL  ; 条码长度
D412 CHANNEL  ; 移栽阻挡气缸缩回位延时
D414 CHANNEL  ; 移栽阻挡气缸伸出位延时
D416 CHANNEL  ; 左机械手升降气缸缩回延时
D418 CHANNEL  ; 左机械手升降气缸伸出延时
D42 CHANNEL  ; 右机械手#3位置(mm）
D420 CHANNEL  ; 左机械手伸缩气缸缩回延时
D422 CHANNEL  ; 左机械手伸缩气缸伸出延时
D424 CHANNEL  ; 左机械手左夹爪张开位延时
D426 CHANNEL  ; 左机械手左夹爪夹紧位延时
D428 CHANNEL  ; 左机械手右夹爪张开位延时
D430 CHANNEL  ; 左机械手右夹爪夹紧位延时
D432 CHANNEL  ; 右机械手升降气缸缩回延时
D434 CHANNEL  ; 右机械手升降气缸伸出延时
D436 CHANNEL  ; 右机械手伸缩气缸缩回延时
D438 CHANNEL  ; 右机械手伸缩气缸伸出延时
D440 CHANNEL  ; 右机械手左夹爪张开位延时
D442 CHANNEL  ; 右机械手左夹爪夹紧位延时
D444 CHANNEL  ; 右机械手右夹爪张开位延时
D446 CHANNEL  ; 右机械手右夹爪夹紧位延时
D448 CHANNEL  ; #1模组左密封气缸缩回延时
D450 CHANNEL  ; #1模组左密封气缸伸出延时
D452 CHANNEL  ; #1模组右密封气缸缩回延时
D454 CHANNEL  ; #1模组右密封气缸伸出延时
D456 CHANNEL  ; #1模组左夹电池张开位延时
D458 CHANNEL  ; #1模组左夹电池夹紧位延时
D46 CHANNEL  ; 龙门升降自动速度(mm）
D460 CHANNEL  ; #1模组右夹电池张开位延时
D462 CHANNEL  ; #1模组右夹电池夹紧位延时
D464 CHANNEL  ; #2模组左密封气缸缩回延时
D466 CHANNEL  ; #2模组左密封气缸伸出延时
D468 CHANNEL  ; #2模组右密封气缸缩回延时
D470 CHANNEL  ; #2模组右密封气缸伸出延时
D472 CHANNEL  ; #2模组左夹电池张开位延时
D474 CHANNEL  ; #2模组左夹电池夹紧位延时
D476 CHANNEL  ; #2模组右夹电池张开位延时
D478 CHANNEL  ; #2模组右夹电池夹紧位延时
D48 CHANNEL  ; 龙门升降手动速度
D480 CHANNEL  ; #3模组左密封气缸缩回延时
D482 CHANNEL  ; #3模组左密封气缸伸出延时
D484 CHANNEL  ; #3模组右密封气缸缩回延时
D486 CHANNEL  ; #3模组右密封气缸伸出延时
D488 CHANNEL  ; #3模组左夹电池张开位延时
D490 CHANNEL  ; #3模组左夹电池夹紧位延时
D492 CHANNEL  ; #3模组右夹电池张开位延时
D494 CHANNEL  ; #3模组右夹电池夹紧位延时
D496 CHANNEL  ; #4模组左密封气缸缩回延时
D498 CHANNEL  ; #4模组左密封气缸伸出延时
D50 CHANNEL  ; 龙门升降加速度
D500 CHANNEL  ; #4模组右密封气缸缩回延时
D502 CHANNEL  ; #4模组右密封气缸伸出延时
D504 CHANNEL  ; #4模组左夹电池张开位延时
D506 CHANNEL  ; #4模组左夹电池夹紧位延时
D508 CHANNEL  ; #4模组右夹电池张开位延时
D510 CHANNEL  ; #4模组右夹电池夹紧位延时
D512 CHANNEL  ; 龙门升降气缸缩回位延时
D514 CHANNEL  ; 龙门升降气缸伸出位延时
D516 CHANNEL  ; 龙门夹爪气缸张开位延时
D518 CHANNEL  ; 龙门夹爪气缸夹紧位延时
D52 CHANNEL  ; 龙门升降取料位置(mm）
D520 CHANNEL  ; 上料盒阻挡左气缸缩回位延时
D522 CHANNEL  ; 上料盒阻挡左气缸伸出位延时
D524 CHANNEL  ; #1上顶升左气缸缩回位延时
D526 CHANNEL  ; #1上顶升左气缸伸出位延时
D528 CHANNEL  ; #1上顶升右气缸缩回位延时
D530 CHANNEL  ; #1上顶升右气缸伸出位延时
D532 CHANNEL  ; #2上顶升左气缸缩回位延时
D534 CHANNEL  ; #2上顶升左气缸伸出位延时
D536 CHANNEL  ; #2上顶升右气缸缩回位延时
D538 CHANNEL  ; #2上顶升右气缸伸出位延时
D54 CHANNEL  ; 龙门升降绝缘NG位置(mm)
D540 CHANNEL  ; #1下顶升左气缸缩回位延时
D542 CHANNEL  ; #1下顶升左气缸伸出位延时
D544 CHANNEL  ; #1下顶升右气缸缩回位延时
D546 CHANNEL  ; #1下顶升右气缸伸出位延时
D548 CHANNEL  ; #2下顶升左气缸缩回位延时
D550 CHANNEL  ; #2下顶升左气缸伸出位延时
D552 CHANNEL  ; #2下顶升右气缸缩回位延时
D554 CHANNEL  ; #2下顶升右气缸伸出位延时
D556 CHANNEL  ; 上料阻挡右气缸缩回位时间
D558 CHANNEL  ; 上料盒阻挡右气缸伸出位时间
D56 CHANNEL  ; 龙门升降检测NG位置(mm)
D560 CHANNEL  ; 左拉带脱离气缸缩回位时间
D562 CHANNEL  ; 左拉带脱离气缸伸出位时间
D564 CHANNEL  ; 右拉带脱离气缸缩回位时间
D566 CHANNEL  ; 右拉带脱离气缸伸出位时间
D568 CHANNEL  ; 料盒定位气缸缩回位时间
D570 CHANNEL  ; 料盒定位气缸伸出位时间
D572 CHANNEL  ; 料盒夹紧气缸伸出位时间
D58 CHANNEL  ; 龙门升降OK位置(mm)
D6 CHANNEL  ; 进料位置(mm)
D600 CHANNEL  ; 移栽伺服脉冲当量
D602 CHANNEL  ; 移栽伺服脉冲当量(浮点)
D604 CHANNEL  ; 移栽伺服当前脉冲
D606 CHANNEL  ; 移栽伺服当前脉冲(浮点)
D608 CHANNEL  ; 移栽伺服当前位置(mm)
D610 CHANNEL  ; 移栽伺服自动加速度
D611 CHANNEL  ; 移栽伺服自动减速带
D612 CHANNEL  ; 移栽伺服自动速度(PPM/s)
D614 CHANNEL  ; 移栽伺服自动位移量
D616 CHANNEL  ; 移栽伺服自动起动速度
D62 CHANNEL  ; 料盒升降自动速度
D620 CHANNEL  ; 移栽伺服手动加速度
D621 CHANNEL  ; 移栽伺服手动减速度
D622 CHANNEL  ; 移栽伺服手动速度(HZ/S)
D6224 CHANNEL  ; 移栽伺服手动位移
D622.00 BOOL  ; 移栽伺服运动参数
D624 CHANNEL  ; 移栽伺服手动位移量
D626 CHANNEL  ; 移栽伺服手动起动速度
D630 CHANNEL  ; 进料位置脉冲(浮点）
D634 CHANNEL  ; 进料位置脉冲
D64 CHANNEL  ; 料盒升降点动速度
D640 CHANNEL  ; 左下料位置脉冲(浮点)
D644 CHANNEL  ; 左下料位置脉冲
D650 CHANNEL  ; 右下料位置脉冲(浮点)
D654 CHANNEL  ; 右下料位置脉冲
D66 CHANNEL  ; 料盒升降加速度
D68 CHANNEL  ; 料盒夹紧位置
D690 CHANNEL  ; 移栽伺服自动速度(浮点)
D694 CHANNEL  ; 移栽伺服手动速度(浮点)
D70 CHANNEL  ; 料盒升降上料盒位置
D700 CHANNEL  ; 左机械脉冲当量
D7001 CHANNEL  ; 电池条码
D702 CHANNEL  ; 左机械手脉冲当量(浮点)
D704 CHANNEL  ; 左机械手当前位置脉冲
D706 CHANNEL  ; 左机械手当前位置脉冲(浮点)
D708 CHANNEL  ; 左机械手当前位置(mm)
D710 CHANNEL  ; 左机械手自动加速度
D711 CHANNEL  ; 左机械手自动减速度
D712 CHANNEL  ; 左机械手自动速度(HZ/S)
D714 CHANNEL  ; 左机械手自动位移量
D716 CHANNEL  ; 左机械手自动起动速度
D72 CHANNEL  ; 料盒升降下料盒位置
D720 CHANNEL  ; 左机械手手动加速度
D721 CHANNEL  ; 左机械手手动减速度
D722 CHANNEL  ; 左机械手手动速度(HZ/s)
D724 CHANNEL  ; 左机械手手动位移
D726 CHANNEL  ; 左机械手手动起动速度
D730 CHANNEL  ; 左机械手进料位置脉冲(浮点)
D734 CHANNEL  ; 左机械手进料位置脉冲
D74 CHANNEL  ; 龙门左右自动速度
D740 CHANNEL  ; 左机械手出料位置脉冲(浮点)
D744 CHANNEL  ; 左机械手出料位置脉冲
D750 CHANNEL  ; 左机械手#2位置脉冲(浮点)
D754 CHANNEL  ; 左机械手#2位置脉冲
D76 CHANNEL  ; 龙门前后手动速度
D760 CHANNEL  ; 左机械手#4位置脉冲(浮点）
D764 CHANNEL  ; 左机械手#4位置脉冲
D78 CHANNEL  ; 龙门左右加速度
D790 CHANNEL  ; 左机械手自动速度(浮点)
D794 CHANNEL  ; 左机械手手动速度
D8 CHANNEL  ; 左下料位置(mm)
D80 CHANNEL  ; 龙门前后#1位置
D800 CHANNEL  ; 右机械手脉冲当量
D8000 CHANNEL  ; 扫码位条码
D8001 CHANNEL  ; 扫码位条码
D802 CHANNEL  ; 右机械手脉冲当量(浮点）
D8020 CHANNEL  ; 移栽前电池条码
D804 CHANNEL  ; 右机械手当前位置脉冲
D8040 CHANNEL  ; 移栽后电池条码
D806 CHANNEL  ; 右机械手当前位置脉冲(浮点)
D8060 CHANNEL  ; #1左夹料电池条码
D808 CHANNEL  ; 右机械手当前位置(mm)
D8080 CHANNEL  ; #1右夹料电池条码
D810 CHANNEL  ; 右机械手自动加速度
D8100 CHANNEL  ; #2左夹料电池条码
D811 CHANNEL  ; 右机械手自动减速度
D812 CHANNEL  ; 右机械手自动速度
D8120 CHANNEL  ; #2右夹料电池条码
D814 CHANNEL  ; 右机械手自动位移
D8140 CHANNEL  ; #3左夹料电池条码
D816 CHANNEL  ; 右机械手自动启动速度
D8160 CHANNEL  ; #3右夹料电池条码
D8180 CHANNEL  ; #4左夹料电池条码
D82 CHANNEL  ; 龙门前后#2位置
D820 CHANNEL  ; 右机械手手动加速度
D8200 CHANNEL  ; #4右夹料电池条码
D821 CHANNEL  ; 右机械手手动减速度
D822 CHANNEL  ; 右机械手手动速度
D8220 CHANNEL  ; 左机械手左夹爪电池条码
D824 CHANNEL  ; 右机械手手动位移
D8240 CHANNEL  ; 左机械手右夹爪条码
D826 CHANNEL  ; 右机械手手动起动速度
D8260 CHANNEL  ; 右机械手左夹爪电池条码
D8280 CHANNEL  ; 右机械手右夹爪条码
D830 CHANNEL  ; 右机械手进料位置脉冲(浮点)
D8300 CHANNEL  ; 检测检测值(欧)
D8304 CHANNEL  ; 检测检测值(欧)浮点
D834 CHANNEL  ; 右机械手进料位置脉冲
D84 CHANNEL  ; 龙门前后#3位置
D840 CHANNEL  ; 右机械手出料位置脉冲(浮点)
D8400 CHANNEL  ; 检测位绝缘值(M欧)
D8402 CHANNEL  ; 移栽前电池绝缘值
D8404 CHANNEL  ; 移栽后电池绝缘值
D8406 CHANNEL  ; #1左夹料电池绝缘值
D8408 CHANNEL  ; #1右夹料电池绝缘值
D8410 CHANNEL  ; #2左夹料电池绝缘值
D8412 CHANNEL  ; #2右夹料电池绝缘值
D8414 CHANNEL  ; #3左夹料电池绝缘值
D8416 CHANNEL  ; #3右夹料电池绝缘值
D8418 CHANNEL  ; #4左夹料电池绝缘值
D8420 CHANNEL  ; #4右夹料电池绝缘值
D8422 CHANNEL  ; 左机械手左夹爪电池绝缘值
D8424 CHANNEL  ; 左机械手右夹爪电池绝缘值
D8426 CHANNEL  ; 右机械手左夹爪电池绝缘值
D8428 CHANNEL  ; 右机械手右夹爪电池绝缘值
D844 CHANNEL  ; 右机械手出料位置脉冲
D850 CHANNEL  ; 右机械手#1位置脉冲(浮点)
D8500 CHANNEL  ; 左机械手左夹爪电池位置
D8501 CHANNEL  ; 左机械手左夹爪电池结果
D8502 CHANNEL  ; 左机械手右夹爪电池位置
D8503 CHANNEL  ; $?St$Bk?_#[17] / 左机械手右夹爪电池结果$?St$Bk?_#[17]
D8504 CHANNEL  ; 右机械手左夹爪电池位置
D8505 CHANNEL  ; 右机械手左夹爪电池结果
D8506 CHANNEL  ; 右机械手右夹爪电池位置
D8507 CHANNEL  ; 右机械手右夹爪电池结果
D8510 CHANNEL  ; 左机械手左夹爪电池条码
D8530 CHANNEL  ; 左机械手右夹爪条码
D854 CHANNEL  ; 右机械手#1位置脉冲
D8550 CHANNEL  ; 右机械手左夹爪电池条码
D8570 CHANNEL  ; 右机械手右夹爪条码
D8590 CHANNEL  ; 左机械手左夹爪电池绝缘值
D8592 CHANNEL  ; 左机械手右夹爪电池绝缘值
D8594 CHANNEL  ; 右机械手左夹爪电池绝缘值
D8596 CHANNEL  ; 右机械手右夹爪电池绝缘值
D86 CHANNEL  ; 龙门前后#4位置
D860 CHANNEL  ; 右机械手#3位置脉冲(浮点)
D864 CHANNEL  ; 右机械手#3位置脉冲
D88 CHANNEL  ; 龙门前后#5位置
D890 CHANNEL  ; 右机械手自动速度(浮点)
D894 CHANNEL  ; 右机械手手动速度(浮点)
D90 CHANNEL  ; 龙门前后#6位置
D900 CHANNEL  ; 龙门升降脉冲当量
D9000 CHANNEL  ; #1模组测试->PC
D9001 CHANNEL  ; #2模组测试->PC
D9002 CHANNEL  ; #3模组测试->PC
D9003 CHANNEL  ; #4模组测试->PC
D9010 CHANNEL  ; #1模组测试完成->PC
D9011 CHANNEL  ; #2模组测试完成->PC
D9012 CHANNEL  ; #3模组测试完成->PC
D9013 CHANNEL  ; #4模组测试完成->PC
D902 CHANNEL  ; 龙门升降脉冲当量(浮点）
D9020 CHANNEL  ; #1模组左电池结果
D9021 CHANNEL  ; #1模组右电池结果
D9022 CHANNEL  ; #2模组左电池结果
D9023 CHANNEL  ; #2模组右电池结果
D9024 CHANNEL  ; #3模组左电池结果
D9025 CHANNEL  ; #3模组右电池结果
D9026 CHANNEL  ; #4模组左电池结果
D9027 CHANNEL  ; #4模组右电池结果
D904 CHANNEL  ; 龙门升降当前位置脉冲
D906 CHANNEL  ; 龙门升降当前位置脉冲(浮点)
D908 CHANNEL  ; 龙门升降当前位置(mm)
D910 CHANNEL  ; 龙门升降自动加速度
D9100 CHANNEL  ; #1左夹料电池条码
D911 CHANNEL  ; 龙门升降自动减速度
D912 CHANNEL  ; 龙门升降自动速度
D9120 CHANNEL  ; #1右夹料电池条码
D9121 CHANNEL  ; 左机械手右夹爪电池结果
D9122 CHANNEL  ; 左机械手左夹爪电池位置
D9123 CHANNEL  ; 左机械手右夹爪电池位置
D914 CHANNEL  ; 龙门升降自动位移量
D9140 CHANNEL  ; #1左夹料电池绝缘值
D9142 CHANNEL  ; #1右夹料电池绝缘值
D916 CHANNEL  ; 龙门升降自动起动速度
D92 CHANNEL  ; 龙门前后#7位置
D920 CHANNEL  ; 龙门升降手动加速度
D9200 CHANNEL  ; #2左夹料电池条码
D921 CHANNEL  ; 龙门升降手动减速度
D922 CHANNEL  ; 龙门机械手手动速度
D9220 CHANNEL  ; #2右夹料电池条码
D9221 CHANNEL  ; #2左放料处电池结果
D924 CHANNEL  ; 龙门升降手动位移量
D9240 CHANNEL  ; #2左夹料电池绝缘值
D9242 CHANNEL  ; #2右夹料电池绝缘值
D926 CHANNEL  ; 龙门升降手动速度
D930 CHANNEL  ; 龙门升降取料位置脉冲(浮点)
D9300 CHANNEL  ; #3左夹料电池条码
D9320 CHANNEL  ; #3右夹料电池条码
D9321 CHANNEL  ; 右机械手右夹爪电池结果
D9322 CHANNEL  ; 右机械手左夹爪电池位置
D9323 CHANNEL  ; 右机械手左夹爪电池结果
D9324 CHANNEL  ; 右机械手右夹爪电池位置
D9325 CHANNEL  ; 右机械手右夹爪电池结果
D934 CHANNEL  ; 龙门升降取料位置脉冲
D9340 CHANNEL  ; #3左夹料电池绝缘值
D9342 CHANNEL  ; #3右夹料电池绝缘值
D94 CHANNEL  ; 龙门前后#8位置
D940 CHANNEL  ; 龙门升降绝缘NG位置脉冲(浮点)
D9400 CHANNEL  ; #4左夹料电池条码
D9420 CHANNEL  ; #4右夹料电池条码
D9421 CHANNEL  ; #2右放料处电池结果
D944 CHANNEL  ; 龙门升降绝缘NG位置脉冲
D9440 CHANNEL  ; #4左夹料电池绝缘值
D9442 CHANNEL  ; #4右夹料电池绝缘值
D950 CHANNEL  ; 龙门升降检测NG位置脉冲(浮点)
D9500 CHANNEL  ; 检测完成--->PC
D9502 CHANNEL  ; 左机械手右夹爪电池位置状态
D9504 CHANNEL  ; 右机械手左夹爪电池位置
D9505 CHANNEL  ; 右机械手左夹爪电池结果
D9506 CHANNEL  ; 右机械手右夹爪电池位置
D9507 CHANNEL  ; 右机械手右夹爪电池结果
D9510 CHANNEL  ; 左机械手左夹爪电池位置状态
D9512 CHANNEL  ; 左机械手右夹爪电池位置状态
D9514 CHANNEL  ; 右机械手左夹爪放料
D9516 CHANNEL  ; 右机械手右夹爪放料
D9520 CHANNEL  ; 龙门夹爪电池结果
D954 CHANNEL  ; 龙门升降检测NG位置脉冲
D96 CHANNEL  ; 龙门前后#9位置
D960 CHANNEL  ; 龙门升降OK位置脉冲(浮点)
D9600 CHANNEL  ; #1左放料电池结果
D9602 CHANNEL  ; #2左放料电池结果
D9604 CHANNEL  ; #1右放料电池结果
D9606 CHANNEL  ; #2右放料电池结果
D964 CHANNEL  ; 龙门升降OK位置脉冲
D98 CHANNEL  ; 龙门前后#10位置
D990 CHANNEL  ; 龙门升降自动速度(浮点)
D994 CHANNEL  ; 龙门升降手动速度(浮点)
H0.00 BOOL  ; #1模组屏蔽
H0.01 BOOL  ; #2模组屏蔽
H0.02 BOOL  ; #3模组屏蔽
H0.03 BOOL  ; #4模组屏蔽
H0.04 BOOL  ; 扫码屏蔽-HMI
H0.06 BOOL  ; 电脑屏蔽
H0.07 BOOL  ; 空跑
H0.08 BOOL  ; 门磁屏蔽
H0.09 BOOL  ; 检测屏蔽-HMI
H0.10 BOOL  ; NG后重测-HMI
H10.00 BOOL  ; OK
H11.00 BOOL  ; 上料机械手归零完成
H12.00 BOOL  ; 下料机械手归零完成
H13.00 BOOL  ; 进料旋转归零完成
H14.00 BOOL  ; 出料旋转归零完成
H18 CHANNEL  ; 上料电池的检测结果
H18.00 BOOL  ; 扫码OK
H18.01 BOOL  ; 扫码NG
H18.02 BOOL  ; 检测OK
H18.03 BOOL  ; 检测NG
H18.04 BOOL  ; 进料到移栽位有料
H1.00 BOOL  ; 上料阻挡气缸缩回位
H1.01 BOOL  ; 上料阻挡气缸伸出位
H1.02 BOOL  ; 上料定位气缸缩回位-HMI
H1.03 BOOL  ; 上料定位气缸伸出位-HMI
H1.04 BOOL  ; 检测气缸缩回位-HMI
H1.05 BOOL  ; 检测气缸伸出位-HMI
H1.06 BOOL  ; 移栽阻挡气缸缩回位-HMI
H1.07 BOOL  ; 移栽阻挡气缸伸出位-HMI
H1.08 BOOL  ; 左机械手升降气缸缩回-HMI
H1.09 BOOL  ; 左机械手升降气缸伸出-HMI
H1.10 BOOL  ; 左机械手伸缩气缸缩回-HMI
H1.11 BOOL  ; 左机械手伸缩气缸伸出-HMI
H1.12 BOOL  ; 左机械手左夹爪张开位-HMI
H1.13 BOOL  ; 左机械手左夹爪夹紧位-HMI
H1.14 BOOL  ; 左机械手右夹爪张开位-HMI
H1.15 BOOL  ; 左机械手右夹爪夹紧位-HMI
H20.00 BOOL  ; 移栽归零完成
H21 CHANNEL  ; 移栽有料状态
H21.00 BOOL  ; 移栽#1有料
H21.01 BOOL  ; #1电池绝缘检测NG
H21.02 BOOL  ; 移栽#2有料
H21.03 BOOL  ; #2电池NG
H22 CHANNEL  ; 左机械手记忆标志
H22.00 BOOL  ; 左机械手归零完成
H22.01 BOOL  ; 左机械手左夹爪手动夹紧
H22.02 BOOL  ; 左机械手右夹爪手动夹紧
H23.00 BOOL  ; 左机械手左夹爪夹紧
H23.01 BOOL  ; 左机械手右夹爪夹紧
H23.02 BOOL  ; 左机械手模组取料左夹爪有电池
H23.03 BOOL  ; 左机械手模组取料右夹爪有料
H23.04 BOOL  ; #1左放料处有料
H23.05 BOOL  ; #2左放料处有料
H24 CHANNEL  ; 右机械手记忆标志
H24.00 BOOL  ; 右机械手归零完成
H24.01 BOOL  ; 右机械手左夹爪手动夹紧
H24.02 BOOL  ; 右机械手右夹爪手动夹紧
H25.00 BOOL  ; 右机械手左夹爪夹紧
H25.01 BOOL  ; 右机械手右夹爪夹紧
H25.02 BOOL  ; 右机械手模组取料左夹爪有电池
H25.03 BOOL  ; 右机械手模组取料右夹爪有料
H25.04 BOOL  ; #1右放料处有料
H25.05 BOOL  ; #2右放料处有料
H26 CHANNEL  ; 模组手动记忆标志
H26.00 BOOL  ; #1自检结果
H27.00 BOOL  ; #2自检结果
H28.00 BOOL  ; #3自检结果
H29.00 BOOL  ; #4自检结果
H2.00 BOOL  ; 右机械手升降气缸缩回-HMI
H2.01 BOOL  ; 右机械手升降气缸伸出-HMI
H2.02 BOOL  ; 右机械手伸缩气缸缩回-HMI
H2.03 BOOL  ; 右机械手伸缩气缸伸出-HMI
H2.04 BOOL  ; 右机械手左夹爪张开位-HMI
H2.05 BOOL  ; 右机械手左夹爪夹紧位-HMI
H2.06 BOOL  ; 右机械手右夹爪张开位-HMI
H2.07 BOOL  ; 右机械手右夹爪夹紧位-HMI
H2.08 BOOL  ; #1模组左密封气缸缩回-HMI
H2.09 BOOL  ; #1模组左密封气缸伸出-HMI
H2.10 BOOL  ; #1模组右密封气缸缩回-HMI
H2.11 BOOL  ; #1模组右密封气缸伸出-HMI
H2.12 BOOL  ; #1模组左夹电池张开位-HMI
H2.13 BOOL  ; #1模组左夹电池夹紧位-HMI
H2.14 BOOL  ; #1模组右夹电池张开位-HMI
H2.15 BOOL  ; #1模组右夹电池夹紧位-HMI
H30 CHANNEL  ; #1模组放料
H30.00 BOOL  ; #1模组左有料
H30.01 BOOL  ; #1模组右有料
H30.02 BOOL  ; #1模组测试完成
H30.03 BOOL  ; #1模组测试中
H30.04 BOOL  ; #1模组放料完成
H30.06 BOOL  ; #1左电池结果
H30.07 BOOL  ; #1右电池结果
H30.08 BOOL  ; #1仪器检测完成信号
H30.10 BOOL  ; #1模组左电池OK
H31 CHANNEL  ; #2模组放料
H31.00 BOOL  ; #2模组左有料
H31.01 BOOL  ; #2模组右有料
H31.02 BOOL  ; #2模组测试完成
H31.03 BOOL  ; #2模组测试中
H31.04 BOOL  ; #2模组放料完成
H31.06 BOOL  ; #2左电池结果
H31.07 BOOL  ; #2右电池结果
H31.08 BOOL  ; #2仪器检测完成信号
H32 CHANNEL  ; #3模组放料
H32.00 BOOL  ; #3模组左有料
H32.01 BOOL  ; #3模组右有料
H32.02 BOOL  ; #3模组测试完成
H32.03 BOOL  ; #3模组测试中
H32.04 BOOL  ; #3模组放料完成
H32.06 BOOL  ; #3左电池结果
H32.07 BOOL  ; #3右电池结果
H32.08 BOOL  ; #3仪器检测完成信号
H33 CHANNEL  ; #4模组放料
H33.00 BOOL  ; #4模组左有料
H33.01 BOOL  ; #4模组右有料
H33.02 BOOL  ; #4模组测试完成
H33.03 BOOL  ; #4模组测试中
H33.04 BOOL  ; #4模组放料完成
H33.06 BOOL  ; #4左电池结果
H33.07 BOOL  ; #4右电池结果
H33.08 BOOL  ; #4仪器检测完成信号
H34.00 BOOL  ; 龙门升降归零完成
H35.00 BOOL  ; 龙门前后归零完成
H36.00 BOOL  ; 龙门左右归零完成
H37.00 BOOL  ; 料盒升降归零完成
H3.00 BOOL  ; #2模组左密封气缸缩回-HMI
H3.01 BOOL  ; #2模组左密封气缸伸出-HMI
H3.02 BOOL  ; #2模组右密封气缸缩回-HMI
H3.03 BOOL  ; #2模组右密封气缸伸出-HMI
H3.04 BOOL  ; #2模组左夹电池张开位-HMI
H3.05 BOOL  ; #2模组左夹电池夹紧位-HMI
H3.06 BOOL  ; #2模组右夹电池张开位-HMI
H3.07 BOOL  ; #2模组右夹电池夹紧位-HMI
H3.08 BOOL  ; #3模组左密封气缸缩回-HMI
H3.09 BOOL  ; #3模组左密封气缸伸出-HMI
H3.10 BOOL  ; #3模组右密封气缸缩回-HMI
H3.11 BOOL  ; #3模组右密封气缸伸出-HMI
H3.12 BOOL  ; #3模组左夹电池张开位-HMI
H3.13 BOOL  ; #3模组左夹电池夹紧位-HMI
H3.14 BOOL  ; #3模组右夹电池张开位-HMI
H3.15 BOOL  ; #3模组右夹电池夹紧位-HMI
H42 CHANNEL  ; 龙门记忆状态
H42.00 BOOL  ; 龙门夹爪气缸手动伸出
H42.01 BOOL  ; 龙门夹爪气缸手动伸出
H43.00 BOOL  ; 上料拉带有料
H43.01 BOOL  ; 上料盒完成
H43.02 BOOL  ; 料盒放料完成
H43.03 BOOL  ; #2下顶升气缸有料
H43.04 BOOL  ; #1下顶升气缸有料
H43.05 BOOL  ; 料盒回上料盒状态
H44.00 BOOL  ; 下料拉带上有料盒
H44.01 BOOL  ; 龙门夹爪夹紧
H44.02 BOOL  ; 龙门夹爪有料
H44.04 BOOL  ; 缓存拉带上有料
H44.06 BOOL  ; #2下料盒位有料
H44.07 BOOL  ; #1下料盒位有料
H45 CHANNEL  ; 第一排料盒的放料标记
H45.00 BOOL  ; 第一排#1电池有料
H45.01 BOOL  ; 第一排#2电池有料
H45.02 BOOL  ; 第一排#3电池有料
H45.03 BOOL  ; 第一排#4电池有料
H45.04 BOOL  ; 第一排#5电池有料
H45.05 BOOL  ; 第一排#6电池有料
H45.06 BOOL  ; 第一排#7电池有料
H45.07 BOOL  ; 第一排#8电池有料
H45.08 BOOL  ; 第一排#9电池有料
H45.09 BOOL  ; 第一排#10电池有料
H45.10 BOOL  ; 第一排#11电池有料
H45.11 BOOL  ; 第一排#12电池有料
H46 CHANNEL  ; 第二排料盒放料标记
H46.00 BOOL  ; 第二排#1电池有料
H46.01 BOOL  ; 第二排#2电池有料
H46.02 BOOL  ; 第二排#3电池有料
H46.03 BOOL  ; 第二排#4电池有料
H46.04 BOOL  ; 第二排#5电池有料
H46.05 BOOL  ; 第二排#6电池有料
H46.06 BOOL  ; 第二排#7电池有料
H46.07 BOOL  ; 第二排#8电池有料
H46.08 BOOL  ; 第二排#9电池有料
H46.09 BOOL  ; 第二排#10电池有料
H46.10 BOOL  ; 第二排#11电池有料
H46.11 BOOL  ; 第二排#12电池有料
H4.00 BOOL  ; #4模组左密封气缸缩回-HMI
H4.01 BOOL  ; #4模组左密封气缸伸出-HMI
H4.02 BOOL  ; #4模组右密封气缸缩回-HMI
H4.03 BOOL  ; #4模组右密封气缸伸出-HMI
H4.04 BOOL  ; #4模组左夹电池张开位-HMI
H4.05 BOOL  ; #4模组左夹电池夹紧位-HMI
H4.06 BOOL  ; #4模组右夹电池张开位-HMI
H4.07 BOOL  ; #4模组右夹电池夹紧位-HMI
H4.08 BOOL  ; 龙门升降气缸缩回位-HMI
H4.09 BOOL  ; 龙门升降气缸伸出位-HMI
H4.10 BOOL  ; 龙门夹爪气缸张开位-HMI
H4.11 BOOL  ; 龙门夹爪气缸夹紧位-HMI
H4.12 BOOL  ; 上料盒阻挡左气缸缩回位-HMI
H4.13 BOOL  ; 上料盒阻挡左气缸伸出位-HMI
H4.14 BOOL  ; #1上顶升左气缸缩回位-HMI
H4.15 BOOL  ; #1上顶升左气缸伸出位-HMI
H51.00 BOOL  ; 前上料夹爪有料
H5.00 BOOL  ; #1上顶升右气缸缩回位-HMI
H5.01 BOOL  ; #1上顶升右气缸伸出位-HMI
H5.02 BOOL  ; #2上顶升左气缸缩回位-HMI
H5.03 BOOL  ; #2上顶升左气缸伸出位-HMI
H5.04 BOOL  ; #2上顶升右气缸缩回位-HMI
H5.05 BOOL  ; #2上顶升右气缸伸出位-HMI
H5.06 BOOL  ; #1下顶升左气缸缩回位-HMI
H5.07 BOOL  ; #1下顶升左气缸伸出位-HMI
H5.08 BOOL  ; #1下顶升右气缸缩回位-HMI
H5.09 BOOL  ; #1下顶升右气缸伸出位-HMI
H5.10 BOOL  ; #2下顶升左气缸缩回位-HMI
H5.11 BOOL  ; #2下顶升左气缸伸出位-HMI
H5.12 BOOL  ; #2下顶升右气缸缩回位-HMI
H5.13 BOOL  ; #2下顶升右气缸伸出位-HMI
H5.14 BOOL  ; 上料盒阻挡右气缸缩回位-HMI
H5.15 BOOL  ; 上料盒阻挡右气缸伸出位-HMI
H6.00 BOOL  ; 左拉带脱离气缸缩回位-HMI
H6.01 BOOL  ; 左拉带脱离气缸伸出位-HMI
H6.02 BOOL  ; 右拉带脱离气缸缩回位-HMI
H6.03 BOOL  ; 右拉带脱离气缸伸出位-HMI
H6.04 BOOL  ; 料盒定位气缸缩回位
H6.05 BOOL  ; 料盒定位气缸伸出位屏蔽
H8.11 BOOL  ; 料盒夹紧伸出到位屏蔽
T0000 BOOL  ; 上料阻挡气缸缩回位时间
T0001 BOOL  ; 上料阻挡气缸伸出位时间
T0002 BOOL  ; 电脑启动按钮按下时间
T0003 BOOL  ; 上料定位气缸伸出位时间
T0004 BOOL  ; 检测气缸缩回位时间
T0005 BOOL  ; 检测气缸伸出位时间
T0006 BOOL  ; 移栽阻挡气缸缩回位时间
T0007 BOOL  ; 移栽阻挡气缸伸出位时间
T0008 BOOL  ; 左机械手升降气缸缩回位时间
T0009 BOOL  ; 左机械手升降气缸伸出位时间
T0010 BOOL  ; 左机械手伸缩气缸缩回位时间
T0011 BOOL  ; 左机械手伸缩气缸伸出位时间
T0012 BOOL  ; 左机械手左夹爪张开位时间
T0013 BOOL  ; 左机械手左夹爪夹紧位时间
T0014 BOOL  ; 左机械手右夹爪张开位时间
T0015 BOOL  ; 左机械手右夹爪夹紧位时间
T0016 BOOL  ; 右机械手升降气缸缩回位时间
T0017 BOOL  ; 右机械手升降气缸伸出位时间
T0018 BOOL  ; 右机械手伸缩气缸缩回位时间
T0019 BOOL  ; 右机械手伸缩气缸伸出位时间
T0020 BOOL  ; 右机械手左夹爪张开位时间
T0021 BOOL  ; 右机械手左夹爪夹紧位时间
T0022 BOOL  ; 右机械手右夹爪张开位时间
T0023 BOOL  ; 右机械手右夹爪夹紧位时间
T0024 BOOL  ; #1模组左密封气缸缩回位时间
T0025 BOOL  ; #1模组左密封气缸伸出位时间
T0026 BOOL  ; #1模组右密封气缸缩回位时间
T0027 BOOL  ; #1模组右密封气缸伸出位时间
T0028 BOOL  ; #1模组左夹料气缸张开位时间
T0029 BOOL  ; #1模组左夹料气缸夹紧位时间
T0030 BOOL  ; #1模组右夹料气缸张开位时间
T0031 BOOL  ; #1模组右夹料气缸夹紧位时间
T0032 BOOL  ; #2模组左密封气缸缩回位时间
T0033 BOOL  ; #2模组左密封气缸伸出位时间
T0034 BOOL  ; #2模组右密封气缸缩回位时间
T0035 BOOL  ; #2模组右密封气缸伸出位时间
T0036 BOOL  ; #2模组左夹料气缸张开位时间
T0037 BOOL  ; #2模组左夹料气缸夹紧位时间
T0038 BOOL  ; #2模组右夹料气缸张开位时间
T0039 BOOL  ; #2模组右夹料气缸夹紧位时间
T0040 BOOL  ; #3左密封气缸缩回位时间
T0041 BOOL  ; #3左密封气缸伸出位时间
T0042 BOOL  ; #3右密封气缸缩回位时间
T0043 BOOL  ; #3右密封气缸伸出位时间
T0044 BOOL  ; #3左夹料气缸张开位时间
T0045 BOOL  ; #3左夹料气缸夹紧位时间
T0046 BOOL  ; #3右夹料气缸张开位时间
T0047 BOOL  ; #3右夹料气缸夹紧位时间
T0048 BOOL  ; #4左密封气缸缩回位时间
T0049 BOOL  ; #4左密封气缸伸出位时间
T0050 BOOL  ; #4右密封气缸缩回位时间
T0051 BOOL  ; #4右密封气缸伸出位时间
T0052 BOOL  ; #4左夹料气缸张开位时间
T0053 BOOL  ; #4左夹料气缸夹紧位时间
T0054 BOOL  ; #4右夹料气缸张开位时间
T0055 BOOL  ; #4右夹料气缸夹紧位
T0056 BOOL  ; 龙门升降气缸缩回位时间
T0057 BOOL  ; 龙门升降气缸伸出位时间
T0058 BOOL  ; 龙门夹爪张开位时间
T0059 BOOL  ; 龙门夹爪夹紧位时间
T0060 BOOL  ; 上料盒阻挡左气缸缩回位时间
T0061 BOOL  ; 上料盒阻挡左气缸伸出位延时
T0062 BOOL  ; 上料盒阻挡右气缸缩回位延时
T0063 BOOL  ; 上料盒阻挡右气缸伸出位延时
T0064 BOOL  ; #1上顶升左气缸缩回位延时
T0065 BOOL  ; #1上顶升左气缸伸出位延时
T0066 BOOL  ; #1上顶升右气缸缩回位延时
T0067 BOOL  ; #1上顶升右气缸伸出位延时
T0068 BOOL  ; #2上顶升左气缸缩回位延时
T0069 BOOL  ; #2上顶升左气缸伸出位延时
T0070 BOOL  ; #2上顶升右气缸缩回位延时
T0071 BOOL  ; #2上顶升右气缸伸出位延时
T0072 BOOL  ; #1下顶升左气缸缩回位
T0073 BOOL  ; #1下顶升左气缸伸出位延时
T0074 BOOL  ; #1下顶升右气缸缩回位延时
T0075 BOOL  ; #1下顶升右气缸伸出位延时
T0076 BOOL  ; #2下顶升左气缸缩回位延时
T0077 BOOL  ; #2下顶升左气缸伸出位延时
T0078 BOOL  ; #2下顶升右气缸缩回位延时
T0079 BOOL  ; #2下顶升右气缸伸出位延时
T0080 BOOL  ; 左拉带脱离气缸缩回位时间
T0081 BOOL  ; 左拉带脱离气缸伸出位时间
T0082 BOOL  ; 右拉带脱离气缸缩回位时间
T0083 BOOL  ; 右拉带脱离气缸伸出位时间
T0084 BOOL  ; 料盒定位气缸缩回位延时
T0085 BOOL  ; 料盒定位气缸伸出位延时
T0086 BOOL  ; 移栽前电池感应
T0087 BOOL  ; 移栽后电池感应
T0088 BOOL  ; #1模组左电池感应屏蔽
T0089 BOOL  ; #1模组右电池感应屏蔽
T0090 BOOL  ; #2模组左电池感应屏蔽
T0091 BOOL  ; #2模组右电池感应屏蔽
T0092 BOOL  ; #3模组左电池感应屏蔽
T0093 BOOL  ; #3模组右电池感应屏蔽
T0094 BOOL  ; #4模组左电池感应屏蔽
T0095 BOOL  ; #4模组右电池感应屏蔽
T0096 BOOL  ; 左#1放料电池感应屏蔽
T0097 BOOL  ; 左#2放料电池感应屏蔽
T0098 BOOL  ; 右#1放料电池感应屏蔽
T0099 BOOL  ; 右#2放料电池感应屏蔽
T0100 BOOL  ; 上料阻挡气缸缩回位报警
T0101 BOOL  ; 上料阻挡气缸伸出位报警
T0102 BOOL  ; 上料定位气缸缩回位报警
T0103 BOOL  ; 上料定位气缸伸出位报警
T0104 BOOL  ; 检测气缸缩回位报警
T0105 BOOL  ; 检测气缸伸出位报警
T0106 BOOL  ; 移栽阻挡气缸缩回位报警
T0107 BOOL  ; 移栽阻挡气缸伸出位报警
T0108 BOOL  ; 左机械手升降气缸缩回位报警
T0109 BOOL  ; 左机械手升降气缸伸出位报警
T0110 BOOL  ; 左机械手伸缩气缸缩回位报警
T0111 BOOL  ; 左机械手伸缩气缸伸出位报警
T0112 BOOL  ; 左机械手左夹爪张开位报警
T0113 BOOL  ; 左机械手左夹爪夹紧位报警
T0114 BOOL  ; 左机械手右夹爪张开位报警
T0115 BOOL  ; 左机械手右夹爪夹紧位报警
T0116 BOOL  ; 右机械手升降气缸缩回位报警
T0117 BOOL  ; 右机械手升降气缸伸出位报警
T0118 BOOL  ; 右机械手伸缩气缸缩回位报警
T0119 BOOL  ; 右机械手伸缩气缸伸出位报警
T0120 BOOL  ; 右机械手左夹爪张开位报警
T0121 BOOL  ; 右机械手左夹爪夹紧位报警
T0122 BOOL  ; 右机械手右夹爪张开位报警
T0123 BOOL  ; 右机械手右夹爪夹紧位报警
T0124 BOOL  ; #1模组左密封气缸缩回位报警
T0125 BOOL  ; #1模组左密封气缸伸出位报警
T0126 BOOL  ; #1模组右密封气缸缩回位报警
T0127 BOOL  ; #1模组右密封气缸伸出位报警
T0128 BOOL  ; #1模组左夹料气缸缩回位报警
T0129 BOOL  ; #1模组左夹料气缸伸出位报警
T0130 BOOL  ; #1模组右夹料气缸缩回报警
T0131 BOOL  ; #1模组右夹料气缸伸出位报警
T0132 BOOL  ; #2模组左密封气缸缩回报警
T0133 BOOL  ; #2模组左密封气缸伸出位报警
T0134 BOOL  ; #2模组右密封气缸缩回位报警
T0135 BOOL  ; #2模组右密封气缸伸出位报警
T0136 BOOL  ; #2模组左夹料气缸张开位报警
T0137 BOOL  ; #2模组左夹料气缸夹紧位报警
T0138 BOOL  ; #2模组右夹料气缸张开位报警
T0139 BOOL  ; #2模组右夹料气缸夹紧位报警
T0140 BOOL  ; #3左密封气缸缩回位报警
T0141 BOOL  ; #3左密封气缸伸出位报警
T0142 BOOL  ; #3右密封气缸缩回位报警
T0143 BOOL  ; #3右密封气缸伸出位报警
T0144 BOOL  ; #3左夹料气缸张开位报警
T0145 BOOL  ; #3左夹料气缸夹紧位报警
T0146 BOOL  ; #3右夹料气缸缩回位报警
T0147 BOOL  ; #3右夹料气缸夹紧位报警
T0148 BOOL  ; #4左密封气缸缩回位报警
T0149 BOOL  ; #4左密封气缸伸出位报警
T0150 BOOL  ; #4右密封气缸缩回位报警
T0151 BOOL  ; #4右密封气缸伸出位报警
T0152 BOOL  ; #4左夹料气缸张开位报警
T0153 BOOL  ; #4左夹料气缸伸出位报警
T0154 BOOL  ; #4右夹料气缸缩回位报警
T0155 BOOL  ; #4右夹料气缸夹紧位报警
T0156 BOOL  ; 龙门升降气缸缩回位报警
T0157 BOOL  ; 龙门升降气缸伸出位报警
T0158 BOOL  ; 龙门夹爪气缸张开位报警
T0159 BOOL  ; 龙门夹爪气缸伸出位报警
T0160 BOOL  ; 上料盒阻挡左气缸缩回位报警
T0161 BOOL  ; 上料盒阻挡左气缸伸出位报警
T0162 BOOL  ; 上料盒阻挡右气缸缩回位报警
T0163 BOOL  ; 上料盒阻挡右气缸伸出位报警
T0164 BOOL  ; #1上顶升左气缸缩回位报警
T0165 BOOL  ; #1上顶升左气缸伸出位报警
T0166 BOOL  ; #1上顶升右气缸缩回位报警
T0167 BOOL  ; #1上顶升右气缸伸出位报警
T0168 BOOL  ; #2上顶升左气缸缩回位报警
T0169 BOOL  ; #2上顶升左气缸伸出位报警
T0170 BOOL  ; #2上顶升右气缸伸出位报警
T0171 BOOL  ; #2上顶升右气缸伸出位报警延时
T0172 BOOL  ; #1下顶升左气缸缩回位报警
T0173 BOOL  ; #1下顶升气缸伸出位报警
T0174 BOOL  ; #1下顶升右气缸缩回位报警
T0175 BOOL  ; #1下顶升右气缸缩回位报警
T0176 BOOL  ; #2下顶升左气缸缩回位报警
T0177 BOOL  ; #2下顶升气缸伸出位报警
T0178 BOOL  ; #2下顶升右气缸缩回位报警
T0179 BOOL  ; #2下料顶升右气缸伸出位报警
T0180 BOOL  ; 左拉带脱离气缸缩回位报警
T0181 BOOL  ; 左拉带脱离气缸伸出位报警
T0182 BOOL  ; 右拉带脱离气缸缩回位报警
T0183 BOOL  ; 右拉带脱离气缸伸出位报警
T0184 BOOL  ; 料盒定位气缸缩回位报警
T0185 BOOL  ; 料盒定位气缸伸出位报警
T0186 BOOL  ; 复位延时
T0187 BOOL  ; 料盒夹紧气缸伸出位延时
T0188 BOOL  ; 料盒夹紧气缸伸出位报警
T0190 BOOL  ; 复位按钮持续时间
T0191 BOOL  ; 启动按钮持续时间
T0192 BOOL  ; 停止按钮持续时间
T0193 BOOL  ; 整机在初始位延时
T0194 BOOL  ; 整机复位延时
T0195 BOOL  ; 程序强制清零延时
T0196 BOOL  ; 异常复位延时
T0200 BOOL  ; 移栽归零左机械手异常提示时间
T0201 BOOL  ; 移栽归零右机械手异常提示时间
T0202 BOOL  ; 移栽左移左机械手异常提示时间
T0203 BOOL  ; 移栽左移没归零异常提示时间
T0204 BOOL  ; 移栽左移左限位到达异常提示时间
T0205 BOOL  ; 移栽右移右机械手异常提示时间
T0206 BOOL  ; 移栽右移没归零异常提示时间
T0207 BOOL  ; 移栽右移右限位异常提示时间
T0208 BOOL  ; 移栽回进料位条件异常提示时间
T0209 BOOL  ; 移栽回进料位没归零异常提示时间
T0210 BOOL  ; 移栽回左下料位条件异常提示时间
T0211 BOOL  ; 移栽回左下料位没归零异常提示时间
T0212 BOOL  ; 移栽回右下料位条件异常提示时间
T0213 BOOL  ; 移栽回右下料位没归零提示时间
T0220 BOOL  ; 左机械手归零升降气缸异常提示时间
T0221 BOOL  ; 左机械手伸缩升降气缸异常提示时间
T0222 BOOL  ; 左机械手没归零异常提示时间
T0223 BOOL  ; 左机械手伸缩气缸伸出异常提示时间
T0224 BOOL  ; 左机械手升降气缸伸出异常提示时间
T0225 BOOL  ; 左机械手夹爪松开升降气缸异常提示时间
T0226 BOOL  ; 左机械手夹爪松开伸缩气缸异常提示时间
T0227 BOOL  ; 左机械手左夹爪松开伸缩气缸异常提示时间
T0228 BOOL  ; 左机械手右夹爪松开升降气缸异常提示时间
T0229 BOOL  ; 左机械手右夹爪松开伸缩气缸异常提示时间
T0230 BOOL  ; 左机械手左夹爪松开延时
T0231 BOOL  ; 左机械手右夹爪松开延时
T0232 BOOL  ; 左机械手左夹爪放料->PC延时
T0233 BOOL  ; 左机械手右夹爪放料->PC延时
T0234 BOOL  ; 前上料机械手2级升降气缸上位
T0240 BOOL  ; 机械手归零升降气缸异常提示时间
T0241 BOOL  ; 右机械手伸缩升降气缸异常提示时间
T0242 BOOL  ; 右机械手没归零异常提示时间
T0243 BOOL  ; 右机械手伸缩气缸伸出异常提示时间
T0244 BOOL  ; 右机械手升降气缸伸出异常提示时间
T0245 BOOL  ; 右机械手夹爪松开升降气缸异常提示时间
T0250 BOOL  ; 右机械手左夹爪松开延时
T0251 BOOL  ; 右机械手右夹爪松开延时
T0252 BOOL  ; 右机械手左夹爪放料延时
T0253 BOOL  ; 右机械手右夹爪放料延时
T0260 BOOL  ; #1左密封气缸没缩回异常提示持续时间
T0261 BOOL  ; #1右密封气缸没缩回异常
T0264 BOOL  ; #2左密封气缸没缩回异常提示持续时间
T0265 BOOL  ; #2右密封气缸没缩回异常
T0268 BOOL  ; #3左密封气缸没缩回异常提示持续时间
T0269 BOOL  ; #3右密封气缸没缩回异常
T0272 BOOL  ; #4左密封气缸没缩回异常提示持续时间
T0273 BOOL  ; #4右密封气缸没缩回异常
T0275 BOOL  ; 放电时间
T0278 BOOL  ; 此位有电池夹爪没打开不能下降延时
T0280 BOOL  ; 龙门升降气缸没缩回异常持续时间
T0281 BOOL  ; 伺服没归零异常持续时间
T0282 BOOL  ; 定位气缸没缩回异常提示持续时间
T0283 BOOL  ; 龙门夹爪松开异常提示持续时间
T0284 BOOL  ; 下料处有料异常提示持续时间
T0285 BOOL  ; 伺服没归零异常提示持续时间
T0286 BOOL  ; 左、右脱离气缸没缩回提示持续时间
T0287 BOOL  ; 龙门升降没缩回异常提示持续时间
T0288 BOOL  ; 龙门升降伺服不在原位提示持续时间
T0289 BOOL  ; 龙门前后、左右伺服没归零提示持续时间
T0290 BOOL  ; 上料机构在初始位
T0291 BOOL  ; 上料有料感应持续时间
T0292 BOOL  ; 来料流出时间
T0293 BOOL  ; 来料流出时间2
T0294 BOOL  ; 来料流出时间
T0295 BOOL  ; 扫码超时
T0296 BOOL  ; 检测超时
T0297 BOOL  ; 来料流出时间
T0298 BOOL  ; 上料无料感应持续时间
T0300 BOOL  ; 移栽伺服左移延时
T0301 BOOL  ; 移栽伺服右移延时
T0302 BOOL  ; 移栽伺服回进料位置延时
T0303 BOOL  ; 移栽伺服回左下料位置延时
T0304 BOOL  ; 移栽伺服回右下料位置延时
T0305 BOOL  ; 移栽伺服回右下料位置延时
T0306 BOOL  ; 移栽伺服回左下料位置延时
T0307 BOOL  ; 移栽伺服回上料位置延时
T0310 BOOL  ; 移栽前电池到位持续时间
T0311 BOOL  ; 移栽后电池到位持续时间
T0312 BOOL  ; 空跑移栽到位延时
T0313 BOOL  ; 移栽机构在初始位
T0314 BOOL  ; 出料处无料延时
T0320 BOOL  ; 移栽#1电池到位超时报警
T0321 BOOL  ; 移栽#2电池到位超时报警
T0322 BOOL  ; 移栽伺服右限位报警
T0323 BOOL  ; 移栽伺服左限位报警
T0324 BOOL  ; 移栽伺服报警
T0325 BOOL  ; 报警延时
T0330 BOOL  ; 检测触发脉冲
T0331 BOOL  ; 检测触发脉冲
T0340 BOOL  ; #1 检漏仪保压结束延时
T0341 BOOL  ; #2 检漏仪保压结束延时
T0342 BOOL  ; #3 检漏仪保压结束延时
T0343 BOOL  ; #3 检漏仪保压结束延时
T0350 BOOL  ; 前上料夹爪气缸张开位
T0351 BOOL  ; 前上料夹爪气缸夹紧位
T0360 BOOL  ; 启动脉冲
T0361 BOOL  ; 检测延时->pc
T0362 BOOL  ; 检测延时->pc
T0370 BOOL  ; 扫描延时
T0400 BOOL  ; 左机械手前进延时
T0401 BOOL  ; 左机械手后退延时
T0402 BOOL  ; 左机械手回上位置延时
T0403 BOOL  ; 左机械手手动回下料位置延时
T0404 BOOL  ; 左机械手回#2位置延时
T0405 BOOL  ; 左机械手回#位4置延时
T0406 BOOL  ; 左机械手回上位置延时
T0407 BOOL  ; 左机械手回#2位置延时
T0408 BOOL  ; 左机械手回#位4置延时
T0409 BOOL  ; 左机械手自动回下料位置延时
T0410 BOOL  ; 左机械手模组放料完成延时
T0411 BOOL  ; 左机械手模组夹料延时
T0420 BOOL  ; 左#1电池有料异常延时
T0421 BOOL  ; 左#2电池有料异常延时
T0422 BOOL  ; 左机械手伺服报警延时
T0423 BOOL  ; 左机械手左限位报警
T0424 BOOL  ; 左机械手右限位报警延时
T0425 BOOL  ; 左机械手在初始位延时
T0427 BOOL  ; 左#1电池有料感应器异常延时
T0428 BOOL  ; 左#2电池有料感应器异常延时
T0430 BOOL  ; 右机械手左限位报警延时
T0431 BOOL  ; 右机械手右限位报警延时
T0432 BOOL  ; 右#1电池有料异常延时
T0433 BOOL  ; 右#2电池有料异常延时
T0434 BOOL  ; 右机械手伺服报警延时
T0435 BOOL  ; 右机械手在初始位延时
T0437 BOOL  ; 右#1电池有料感应器异常延时
T0438 BOOL  ; 右#2电池有料感应器异常延时
T0500 BOOL  ; 右机械手前进延时
T0501 BOOL  ; 右机械手后退延时
T0502 BOOL  ; 右机械手回上位置延时
T0503 BOOL  ; 右机械手手动回下料位置延时
T0504 BOOL  ; 右机械手回#1位置延时
T0505 BOOL  ; 右机械手回#3位置延时
T0506 BOOL  ; 右机械手回上位置延时
T0507 BOOL  ; 右机械手回#1位置延时
T0508 BOOL  ; 右机械手回#3位置延时
T0509 BOOL  ; 右机械手自动回下料位置延时
T0510 BOOL  ; 右机械手模组放料完成延时
T0511 BOOL  ; 右机械手模组夹料延时
T0600 BOOL  ; 自检气缸输出延时
T0601 BOOL  ; 密封气缸自检输出延时
T0602 BOOL  ; #1检漏仪启动时间
T0610 BOOL  ; 自检气缸输出延时
T0611 BOOL  ; 密封气缸自检输出延时
T0612 BOOL  ; #2检漏仪启动时间
T0620 BOOL  ; 自检气缸输出延时
T0621 BOOL  ; 密封气缸自检输出延时
T0622 BOOL  ; #3检漏仪启动时间
T0630 BOOL  ; 自检气缸输出延时
T0631 BOOL  ; 密封气缸自检输出延时
T0632 BOOL  ; #4检漏仪启动时间
T0640 BOOL  ; #1左自检气缸输出延时
T0641 BOOL  ; #1右自检气缸输出延时
T0642 BOOL  ; #1检漏仪启动脉冲时间
T0643 BOOL  ; 左密封气缸伸出延时
T0644 BOOL  ; #1右密封气缸伸出延时
T0645 BOOL  ; 测试结束完成延时
T0646 BOOL  ; #1模组状态复位延时
T0647 BOOL  ; #1左重测延时
T0648 BOOL  ; #1右自检气缸伸出延时
T0649 BOOL  ; #1检漏仪启动脉冲时间
T0650 BOOL  ; #2左自检气缸输出延时
T0651 BOOL  ; #2右自检气缸输出延时
T0652 BOOL  ; #2检漏仪启动脉冲时间
T0653 BOOL  ; #2左密封气缸输出延时
T0654 BOOL  ; #2右密封气缸伸出延时
T0655 BOOL  ; 测试结束完成延时
T0656 BOOL  ; #2模组状态复位延时
T0657 BOOL  ; #2左重测延时
T0658 BOOL  ; #2右自检气缸伸出延时
T0659 BOOL  ; #2检漏仪启动脉冲时间
T0660 BOOL  ; #3左自检气缸输出延时
T0661 BOOL  ; #3右自检气缸输出延时
T0662 BOOL  ; #3检漏仪启动脉冲时间
T0663 BOOL  ; #3左密封气缸输出延时
T0664 BOOL  ; #3右密封气缸输出延时
T0665 BOOL  ; 测试结束完成延时
T0666 BOOL  ; #3模组状态复位延时
T0667 BOOL  ; #3左重测延时
T0668 BOOL  ; #3右自检气缸伸出延时
T0669 BOOL  ; #3检漏仪启动脉冲时间
T0670 BOOL  ; #4左自检气缸输出延时
T0671 BOOL  ; #4右自检气缸输出延时
T0672 BOOL  ; #4检漏仪启动脉冲时间
T0673 BOOL  ; #4左密封气缸输出延时
T0674 BOOL  ; #4右密封气缸输出延时
T0675 BOOL  ; 测试结束完成延时
T0676 BOOL  ; #4模组状态复位延时
T0677 BOOL  ; #4左重测延时
T0678 BOOL  ; #4右自检气缸伸出延时
T0679 BOOL  ; #4检漏仪启动脉冲时间
T0680 BOOL  ; #1模组左有料异常延时
T0681 BOOL  ; #1模组右有料异常延时
T0682 BOOL  ; #1检漏仪Busy异常延时
T0683 BOOL  ; #1检漏仪启动->PC持续时间
T0684 BOOL  ; #1左自检气缸缩回延时
T0685 BOOL  ; #1左重测完成延时
T0686 BOOL  ; #1右自检气缸缩回延时
T0687 BOOL  ; #1左自检气缸伸出延时
T0688 BOOL  ; #1检漏仪启动脉冲时间
T0689 BOOL  ; #1右重测完成延时
T0690 BOOL  ; #2模组左有料异常延时
T0691 BOOL  ; #2模组右有料异常延时
T0692 BOOL  ; #2检漏仪Busy异常延时
T0693 BOOL  ; #2检漏仪启动->PC持续时间
T0694 BOOL  ; #2左自检气缸缩回延时
T0695 BOOL  ; #2左重测完成延时
T0696 BOOL  ; #2右自检气缸缩回延时
T0697 BOOL  ; #2左自检气缸伸出延时
T0698 BOOL  ; #2检漏仪启动脉冲时间
T0699 BOOL  ; #2右重测完成延时
T0700 BOOL  ; 龙门回#1左取料位延时
T0701 BOOL  ; 龙门回#2左取料位延时
T0702 BOOL  ; 龙门回#1右取料位延时
T0703 BOOL  ; 龙门回#2右取料位延时
T0704 BOOL  ; 龙门回#1放料位延时
T0705 BOOL  ; 龙门回#2放料位延时
T0706 BOOL  ; 龙门回#3放料位延时
T0707 BOOL  ; 龙门回#4放料位延时
T0708 BOOL  ; 龙门回#5放料位延时
T0709 BOOL  ; 龙门回#6放料位延时
T0710 BOOL  ; 龙门回#7放料位延时
T0711 BOOL  ; 龙门回#8放料位延时
T0712 BOOL  ; 龙门回#9放料位延时
T0713 BOOL  ; 龙门回#10放料位延时
T0714 BOOL  ; 龙门回#11放料位延时
T0715 BOOL  ; 龙门回#12放料位延时
T0716 BOOL  ; 龙门回#13放料位延时
T0717 BOOL  ; 龙门回#14放料位延时
T0718 BOOL  ; 龙门回#15放料位延时
T0719 BOOL  ; 龙门回#16放料位延时
T0720 BOOL  ; 龙门回#17放料位延时
T0721 BOOL  ; 龙门回#18放料位延时
T0722 BOOL  ; 龙门回#19放料位延时
T0723 BOOL  ; 龙门回#20放料位延时
T0724 BOOL  ; 龙门回#21放料位延时
T0725 BOOL  ; 龙门回#22放料位延时
T0726 BOOL  ; 龙门回#23放料位延时
T0727 BOOL  ; 龙门回#24放料位延时
T0728 BOOL  ; 龙门回绝缘NG位延时
T0729 BOOL  ; 龙门回检漏NG位延时
T0730 BOOL  ; 龙门前后点动延时
T0731 BOOL  ; 龙门左右点动延时
T0732 BOOL  ; 龙门回#2右取料位延时
T0744 BOOL  ; #3左自检气缸缩回延时
T0745 BOOL  ; #3左重测完成延时
T0746 BOOL  ; #3右自检气缸缩回延时
T0747 BOOL  ; #3左自检气缸伸出延时
T0748 BOOL  ; #3检漏仪启动脉冲时间
T0749 BOOL  ; #3右重测完成延时
T0750 BOOL  ; 右密封气缸伸出延时
T0752 BOOL  ; #2右密封气缸伸延时
T0753 BOOL  ; #2左密封气缸伸出延时
T0754 BOOL  ; #3右密封气缸输出延时
T0755 BOOL  ; #4左重测完成延时
T0756 BOOL  ; #4右自检气缸缩回延时
T0757 BOOL  ; #4左自检气缸伸出延时
T0758 BOOL  ; #4检漏仪启动脉冲时间
T0759 BOOL  ; #4右重测完成延时
T0760 BOOL  ; #1检漏仪测试完成->PC持续时间
T0761 BOOL  ; #2检漏仪测试完成->PC持续时间
T0764 BOOL  ; #4右自检气缸缩回延时
T0770 BOOL  ; #3左密封气缸伸出延时
T0771 BOOL  ; #4右密封气缸伸出延时
T0772 BOOL  ; #4左密封气缸伸出延时
T0780 BOOL  ; #2检漏仪完成
T0800 BOOL  ; 龙门升降手动上升延时
T0801 BOOL  ; 龙门升降手动下降延时
T0802 BOOL  ; 龙门升降回取料位置延时
T0803 BOOL  ; 龙门升降回OK放料位置延时
T0804 BOOL  ; 龙门升降回绝缘NG放料位置延时
T0805 BOOL  ; 龙门升降回检漏NG放料位置延时
T0806 BOOL  ; 料盒升降回上料盒位置延时
T0807 BOOL  ; 料盒升降回放料盒位置延时
T0808 BOOL  ; 料盒升降点动延时
T0809 BOOL  ; 龙门升降回初始位置延时
T0810 BOOL  ; 龙门升降回取料位置延时
T0811 BOOL  ; 龙门升降回OK放料位置延时
T0812 BOOL  ; 龙门升降回绝缘NG放料位置延时
T0813 BOOL  ; 龙门升降回检漏NG放料位置延时
T0821 BOOL  ; v料盒#1电池感应延时
T0822 BOOL  ; 料盒#2电池感应延时
T0823 BOOL  ; 料盒#3电池感应延时
T0824 BOOL  ; 料盒#4电池感应延时
T0825 BOOL  ; 料盒#5电池感应延时
T0826 BOOL  ; 料盒#6电池感应延时
T0827 BOOL  ; 料盒#7电池感应延时
T0828 BOOL  ; 料盒#8电池感应延时
T0829 BOOL  ; 料盒#9电池感应延时
T0830 BOOL  ; 料盒#10电池感应延时
T0831 BOOL  ; 料盒#11电池感应延时
T0832 BOOL  ; 料盒#12电池感应延时
T0841 BOOL  ; 料盒#13电池感应延时
T0842 BOOL  ; 料盒#14电池感应延时
T0843 BOOL  ; 料盒#15电池感应延时
T0844 BOOL  ; 料盒#16电池感应延时
T0845 BOOL  ; 料盒#17电池感应延时
T0846 BOOL  ; 料盒#18电池感应延时
T0847 BOOL  ; 料盒#19电池感应延时
T0848 BOOL  ; 料盒#20电池感应延时
T0849 BOOL  ; 料盒#21电池感应延时
T0850 BOOL  ; 料盒#22电池感应延时
T0851 BOOL  ; 料盒#23电池感应延时
T0852 BOOL  ; 料盒#24电池感应延时
T0853 BOOL  ; 检漏电机延时走
T0855 BOOL  ; 绝缘NG电机延时走
T0900 BOOL  ; #1料盒没料感应延时
T0901 BOOL  ; #2料盒没料感应延时
T0902 BOOL  ; 料盒到位延时
T0910 BOOL  ; 料盒到达#2位置延时
T0911 BOOL  ; #2顶升气缸缩回延时
T0912 BOOL  ; 料盒到达#1位置延时
T0913 BOOL  ; #1上顶升气缸缩回延时
T0914 BOOL  ; 龙门放OK料延时
T0915 BOOL  ; 龙门升降回OK放料位延时
T0916 BOOL  ; 龙门升降回绝缘NG放料位延时
T0917 BOOL  ; 龙门升降回检漏NG放料位延时
T0920 BOOL  ; 料盒上料到位时间
T0921 BOOL  ; 料盒下料到位时间
T0922 BOOL  ; 龙门升降伺服报警延时
T0923 BOOL  ; 龙门前后伺服报警延时
T0924 BOOL  ; 龙门左右伺服报警延时
T0925 BOOL  ; 料盒升降伺服报警延时
T0926 BOOL  ; 龙门升降在初始位延时
T0927 BOOL  ; 龙门前后，左右在初始位延时
T0928 BOOL  ; 龙门机构在初始位延时
T0929 BOOL  ; 检漏NG满输送带料满延时
T0930 BOOL  ; 绝缘NG满输送带料满延时
T0931 BOOL  ; 龙门升降上限位异常
T0932 BOOL  ; #1缩回延时
T0933 BOOL  ; #2缩回延时
T0934 BOOL  ; 龙门升降下限位异常
T0935 BOOL  ; 龙门前后前限位异常持续时间
T0936 BOOL  ; 龙门前后后限位异常持续时间
T0937 BOOL  ; 龙门左右右限位异常持续时间
T0938 BOOL  ; 龙门左右左限位异常持续时间
T0939 BOOL  ; 料盒升降下限位异常持续时间
T0940 BOOL  ; 料盒升降上限位异常持续时间
T0959 BOOL  ; 放料位有电池不能放料延时报警
T0962 BOOL  ; 延时判断
T1000 BOOL  ; #3模组左有料异常延时
T1001 BOOL  ; #3模组右有料异常延时
T1002 BOOL  ; #3检漏仪Busy异常延时
T1003 BOOL  ; #3检漏仪启动->PC持续时间
T1004 BOOL  ; #3检漏仪测试完成->PC持续时间
T1100 BOOL  ; #4模组左有料异常延时
T1101 BOOL  ; #4模组右有料异常延时
T1102 BOOL  ; #4检漏仪Busy异常延时
T1103 BOOL  ; #4检漏仪启动->PC持续时间
T1104 BOOL  ; #4检漏仪测试完成->PC持续时间
T1110 BOOL  ; #1模组在初始位延时
T1112 BOOL  ; #2模组在初始位延时
T1114 BOOL  ; #3模组在初始位延时
T1116 BOOL  ; #4模组在初始位延时
T1200 BOOL  ; 检测->移栽前数据移转延时
T1201 BOOL  ; 检测->移栽后数据移转延时
T1202 BOOL  ; 移栽前->左机械手左夹爪据移转延时
T1203 BOOL  ; 移栽后->左机械手右夹爪据移转延时
T1204 BOOL  ; 左机械手左夹爪->#2左夹料据移转延时
T1205 BOOL  ; 左机械手左夹爪->#4左夹料据移转延时
T1206 BOOL  ; 左机械手右夹爪->#2右夹料据移转延时
T1207 BOOL  ; 左机械手右夹爪->#4右夹料据移转延时
T1208 BOOL  ; #2左夹料->左机械手左夹爪据移转延时
T1209 BOOL  ; #2右夹料->左机械手右夹爪据移转延时
T1210 BOOL  ; #4左夹料->左机械手左夹爪据移转延时
T1211 BOOL  ; #4右夹料->左机械手右夹爪据移转延时
T1212 BOOL  ; 移栽前->右机械手右夹爪据移转延时
T1213 BOOL  ; 移栽后->右机械手左夹爪据移转延时
T1214 BOOL  ; 右机械手左夹爪->#1左夹料据移转延时
T1215 BOOL  ; 右机械手左夹爪->#3左夹料据移转延时
T1216 BOOL  ; 右机械手右夹爪->#1右夹料据移转延时
T1217 BOOL  ; 右机械手右夹爪->#3右夹料据移转延时
T1218 BOOL  ; #1左夹料->右机械手左夹爪据移转延时
T1219 BOOL  ; #1右夹料->右机械手右夹爪据移转延时
T1220 BOOL  ; #3左夹料->右机械手左夹爪据移转延时
T1221 BOOL  ; #3右夹料->右机械手右夹爪据移转延时
T1230 BOOL  ; 检测延时
T1300 CHANNEL  ; #1检漏仪抽气时间
T1300 BOOL  ; #1检漏仪抽气时间
T1301 BOOL  ; #2检漏仪抽气时间
T1302 BOOL  ; #3检漏仪抽气时间
T1303 BOOL  ; #4检漏仪抽气时间
T1400 BOOL  ; #1检漏仪加压后延时
T1401 BOOL  ; #2检漏仪保压时间
T1402 BOOL  ; #3检漏仪保压时间
T1403 BOOL  ; #4检漏仪保压时间
T1410 BOOL  ; #1 检漏仪保压结束延时
T1411 BOOL  ; #2 检漏仪保压结束延时
T1412 BOOL  ; #3 检漏仪保压结束延时
T1413 BOOL  ; #4 检漏仪保压结束延时
T2000 BOOL  ; PC运行标志断开时间
W0.00 BOOL  ; 手动/自动
W0.01 BOOL  ; 启动-HMI
W0.02 BOOL  ; 复位-HMI
W0.03 BOOL  ; 停止-HMI
W0.04 BOOL  ; 清料开
W0.05 BOOL  ; 再次扫描-HMI
W10.00 BOOL  ; #7放料位-HMI
W10.01 BOOL  ; #8放料位-HMI
W10.02 BOOL  ; #9放料位-HMI
W10.03 BOOL  ; #10放料位-HMI
W10.04 BOOL  ; #11放料位-HMI
W10.05 BOOL  ; #12放料位-HMI
W10.06 BOOL  ; #13放料位-HMI
W10.07 BOOL  ; #14放料位-HMI
W10.08 BOOL  ; #15放料位-HMI
W10.09 BOOL  ; #16放料位-HMI
W10.10 BOOL  ; #17放料位-HMI
W10.11 BOOL  ; #18放料位-HMI
W10.12 BOOL  ; #19放料位-HMI
W10.13 BOOL  ; #20放料位-HMI
W10.14 BOOL  ; #21放料位-HMI
W10.15 BOOL  ; #22放料位-HMI
W11.00 BOOL  ; 进料位置-HMI
W11.01 BOOL  ; 左下料位置-HMI
W11.02 BOOL  ; 右下料位置-HMI
W11.03 BOOL  ; 左机械手进料位置-HMI
W11.04 BOOL  ; 左机械手出料位置-HMI
W11.05 BOOL  ; 左机械手#2位置-HMI
W11.06 BOOL  ; 左机械手#4位置-HMI
W11.07 BOOL  ; 右机械手进料位置-HMI
W11.08 BOOL  ; 右机械出料位置-HMI
W11.09 BOOL  ; 右机械手#1位置-HMI
W11.10 BOOL  ; 右机械手#3位置-HMI
W11.11 BOOL  ; 龙门升降取料位置-HMI
W11.12 BOOL  ; 绝缘NG位置-HMI
W11.13 BOOL  ; 龙门升降检测NG位置-HMI
W11.14 BOOL  ; 龙门升降OK位置-HMI
W11.15 BOOL  ; 上料盒位置-HMI
W12.00 BOOL  ; 下料盒位置-HMI
W12.01 BOOL  ; 料盒夹紧位置-HMI
W12.03 BOOL  ; #1位置-HMI
W12.04 BOOL  ; #2位置-HMI
W12.05 BOOL  ; #3位置-HMI
W12.06 BOOL  ; #4位置-HMI
W12.07 BOOL  ; #5位置-HMI
W12.08 BOOL  ; #6位置-HMI
W12.09 BOOL  ; #7位置-HMI
W12.10 BOOL  ; #8位置-HMI
W12.11 BOOL  ; #9位置-HMI
W12.12 BOOL  ; #10位置-HMI
W12.13 BOOL  ; #11位置-HMI
W12.14 BOOL  ; #12位置-HMI
W12.15 BOOL  ; #13位置-HMI
W13.00 BOOL  ; #14位置-HMI
W13.01 BOOL  ; #15位置-HMI
W13.02 BOOL  ; #16位置-HMI
W13.03 BOOL  ; #17位置-HMI
W13.04 BOOL  ; #18位置-HMI
W13.05 BOOL  ; #19位置-HMI
W13.06 BOOL  ; #20位置-HMI
W13.07 BOOL  ; #21位置-HMI
W13.08 BOOL  ; #22位置-HMI
W13.09 BOOL  ; #23位置-HMI
W13.10 BOOL  ; #24位置-HMI
W13.11 BOOL  ; #1位置-HMI
W13.12 BOOL  ; #2位置-HMI
W13.13 BOOL  ; #3位置-HMI
W13.14 BOOL  ; #4位置-HMI
W13.15 BOOL  ; #5位置-HMI
W14.00 BOOL  ; #6位置-HMI
W14.01 BOOL  ; #7位置-HMI
W14.02 BOOL  ; #8位置-HMI
W14.03 BOOL  ; #9位置-HMI
W14.04 BOOL  ; #10位置-HMI
W14.05 BOOL  ; #11位置-HMI
W14.06 BOOL  ; #12位置-HMI
W14.07 BOOL  ; #13位置-HMI
W14.08 BOOL  ; #14位置-HMI
W14.09 BOOL  ; #15位置-HMI
W14.10 BOOL  ; #16位置-HMI
W14.11 BOOL  ; #17位置-HMI
W14.12 BOOL  ; #18位置-HMI
W14.13 BOOL  ; #19位置-HMI
W14.14 BOOL  ; #20位置-HMI
W14.15 BOOL  ; #21位置-HMI
W15.00 BOOL  ; #22位置-HMI
W15.01 BOOL  ; #23位置-HMI
W15.02 BOOL  ; #24位置-HMI
W15.03 BOOL  ; #1左放料位置-HMI
W15.04 BOOL  ; #2左放料位置-HMI
W15.05 BOOL  ; #1右放料位置-HMI
W15.06 BOOL  ; #2右放料位置-HMI
W15.07 BOOL  ; #1左放料位置-HMI
W15.08 BOOL  ; #2左放料位置-HMI
W15.09 BOOL  ; #1右放料位置-HMI
W15.10 BOOL  ; #2右放料位置-HMI
W15.11 BOOL  ; 绝缘NG位置-HMI
W15.12 BOOL  ; 检漏NG位置-HMI
W15.13 BOOL  ; 绝缘NG位置-HMI
W15.14 BOOL  ; 检漏NG位置-HMI
W15.15 BOOL  ; 计算位置-HMI
W161.01 BOOL  ; 程序强制清零-HMI
W161.07 BOOL  ; 程序强制清零-HMI
W16.00 BOOL  ; 计算位置-HMI
W16.02 BOOL  ; 左机械手左夹爪打开-HMI
W16.03 BOOL  ; 左机械手右夹爪打开-HMI
W16.04 BOOL  ; 右机械手左夹爪打开-HMI
W16.05 BOOL  ; 右机械手右夹爪打开-HMI
W16.06 BOOL  ; 龙门升降夹爪松开-HMI
W16.07 BOOL  ; 程序强制清零-HMI
W16.08 BOOL  ; 整机复位按钮-HMI
W16.09 BOOL  ; 报警声音关-HMI
W16.10 BOOL  ; 电脑启动
W17.00 BOOL  ; #23放料位-HMI
W17.01 BOOL  ; #24放料位-HMI
W17.02 BOOL  ; 绝缘NG位-HMI
W17.03 BOOL  ; 检漏NG位-HMI
W18 CHANNEL  ; 上料机构状态
W18.00 BOOL  ; 进料挡料气缸输出
W18.01 BOOL  ; 检测气缸输出
W18.02 BOOL  ; 上料阻挡气缸伸出
W18.03 BOOL  ; 检测气缸伸出
W18.04 BOOL  ; 扫码触发
W18.05 BOOL  ; 检测触发信号
W18.06 BOOL  ; 扫码触发
W18.07 BOOL  ; 检测触发信号
W18.08 BOOL  ; 绝缘检测完成
W18.09 BOOL  ; 绝缘检测完成
W18.10 BOOL  ; 手动检测气缸输出
W18.11 BOOL  ; 绝缘检测仪启动
W18.12 BOOL  ; 检测结果判断开始
W18.14 BOOL  ; 扫描完成
W18.15 BOOL  ; 测试放电
W19.00 BOOL  ; 门磁条件
W19.01 BOOL  ; PC系统条件
W19.02 BOOL  ; 机械手归零条件
W19.03 BOOL  ; 左机械手气缸状态
W19.04 BOOL  ; 右机械手气缸状态
W19.05 BOOL  ; #1模组气缸状态
W19.06 BOOL  ; #2模组气缸状态
W19.07 BOOL  ; #3模组气缸状态
W19.08 BOOL  ; #4模组气缸状态
W19.09 BOOL  ; 龙门夹爪气缸状态
W19.10 BOOL  ; 启动状态
W19.11 BOOL  ; 暂停
W19.12 BOOL  ; 延时检测
W19.13 BOOL  ; 自动延时检测
W1.00 BOOL  ; 移栽归零-HMI
W1.01 BOOL  ; 移栽左移-HMI
W1.02 BOOL  ; 移栽右移-HMI
W1.03 BOOL  ; 移栽进料位置-HMI
W1.04 BOOL  ; 移栽左下料位-HMI
W1.05 BOOL  ; 移栽右下料位-HMI
W1.07 BOOL  ; 进料挡料-HMI
W1.08 BOOL  ; 挡料气缸-HMI
W1.09 BOOL  ; #1移栽电机-HMI
W1.10 BOOL  ; #2移栽电机-HMI
W1.11 BOOL  ; 真空泵-HMI
W1.12 BOOL  ; 检测气缸-HMI
W1.13 BOOL  ; 手动扫描-HMI
W1.14 BOOL  ; 手动检测-HMI
W20 CHANNEL  ; 移栽手动状态
W200.00 BOOL  ; 调试
W200.01 BOOL  ; 调试
W200.02 BOOL  ; 调试
W200.03 BOOL  ; 调试
W200.04 BOOL  ; 调试
W200.05 BOOL  ; 调试
W200.06 BOOL  ; 调试
W200.10 BOOL  ; 手动检测调试
W200.12 BOOL  ; 调试
W200.13 BOOL  ; 手动扫描
W200.15 BOOL  ; 调试
W20.00 BOOL  ; 移栽伺服在上料位置
W20.01 BOOL  ; 移栽伺服在左下料位置
W20.02 BOOL  ; 移栽伺服在右下料位置
W20.03 BOOL  ; 移栽左移条件
W20.04 BOOL  ; 移栽右移条件
W20.05 BOOL  ; 回进料位条件
W20.06 BOOL  ; 移栽伺服归零
W20.07 BOOL  ; 移栽伺服左移
W20.08 BOOL  ; 移栽伺服右移
W20.09 BOOL  ; 移栽回进料位置
W20.10 BOOL  ; 移栽回左下料位置
W20.11 BOOL  ; 移栽回右下料位置
W20.12 BOOL  ; 移栽挡料气缸手动输出
W20.13 BOOL  ; #1移栽挡料电机
W20.14 BOOL  ; #2移栽挡料电机
W20.15 BOOL  ; 真空泵启动
W21 CHANNEL  ; 移栽自动状态
W21.00 BOOL  ; #1移栽电机启动
W21.01 BOOL  ; 移栽挡料气缸输出
W21.02 BOOL  ; #2移栽电机启动
W21.03 BOOL  ; #2移栽电机停止
W21.04 BOOL  ; 移栽回右下料位
W21.05 BOOL  ; 移栽回左下料位
W21.06 BOOL  ; 移栽回上料位
W21.07 BOOL  ; 移栽回右下料位
W21.08 BOOL  ; 移栽回左下料位
W21.09 BOOL  ; 真空泵启动
W21.12 BOOL  ; 移栽挡料气缸手动输出
W22.00 BOOL  ; 左机械手在进料位置
W22.01 BOOL  ; 左机械手在出料位置
W22.02 BOOL  ; 左机械手在#2模组位置
W22.03 BOOL  ; 左机械手在#4模组位置
W22.04 BOOL  ; 左机械手手动归零
W22.05 BOOL  ; 左机械手手动后退
W22.06 BOOL  ; 左机械手手动前进
W22.07 BOOL  ; 左机械手手动上料位置
W22.08 BOOL  ; 左机械手手动下料位置
W22.09 BOOL  ; 左机械手手动回#2位置
W22.10 BOOL  ; 左机械手手动回#4位置
W22.11 BOOL  ; 左机械手伸缩气缸手动伸出
W22.12 BOOL  ; 左机械手升降气缸手动伸出
W22.13 BOOL  ; 左机械手左夹爪手动夹紧
W22.14 BOOL  ; 左机械手右夹爪手动夹紧
W23 CHANNEL  ; 左机械手动作
W23.00 BOOL  ; 左机械手去上料位置
W23.01 BOOL  ; 左机械手伸缩气缸伸出
W23.02 BOOL  ; 左机械手升降气缸伸出
W23.03 BOOL  ; 左机械手回#2模组放料
W23.04 BOOL  ; 左机械手回#4模组放料
W23.05 BOOL  ; 回上料处待料条件
W23.06 BOOL  ; 回#2模组位待料条件
W23.07 BOOL  ; 回#4模组位待料条件
W23.08 BOOL  ; 左机械手回#2模组取料
W23.09 BOOL  ; 左机械手回#4模组取料
W23.10 BOOL  ; 左机械手回上料位待料
W23.11 BOOL  ; 左机械手取料后回放料位置
W23.12 BOOL  ; 左机械手回#4模组待料
W23.13 BOOL  ; 左机械手回#2模组位待料
W23.14 BOOL  ; 左机械手回#4模组位待料
W23.15 BOOL  ; 左机械手放料完成
W24.00 BOOL  ; 右机械手在进料位置
W24.01 BOOL  ; 右机械手在出料位置
W24.02 BOOL  ; 右机械手在#1模组位置
W24.03 BOOL  ; 右机械手在#3模组位置
W24.04 BOOL  ; 右机械手手动归零
W24.05 BOOL  ; 右机械手手动后退
W24.06 BOOL  ; 右机械手手动前进
W24.07 BOOL  ; 右机械手手动上料位置
W24.08 BOOL  ; 右机械手手动下料位置
W24.09 BOOL  ; 右机械手手动回#1位置
W24.10 BOOL  ; 右机械手手动回#3位置
W24.11 BOOL  ; 右机械手伸缩气缸手动伸出
W24.12 BOOL  ; 右机械手升降气缸手动伸出
W24.13 BOOL  ; 右机械手回#1模组位待料
W24.14 BOOL  ; 右机械手回#3模组位待料
W25 CHANNEL  ; 右机械手动作
W25.00 BOOL  ; 右机械手去上料位置
W25.01 BOOL  ; 右机械手伸缩气缸伸出
W25.02 BOOL  ; 右机械手升降气缸伸出
W25.03 BOOL  ; 右机械手回#1模组放料
W25.04 BOOL  ; 右机械手回#3模组放料
W25.05 BOOL  ; 回上料处待料条件
W25.06 BOOL  ; 回#1模组待料条件
W25.07 BOOL  ; 回#3模组待料条件
W25.08 BOOL  ; 右机械手回#1模组取料
W25.09 BOOL  ; 右机械手回#3模组取料
W25.10 BOOL  ; 右机械手回上料位待料
W25.11 BOOL  ; 右机械手取料后回放料位置
W25.12 BOOL  ; 右机械手回#3模组待料
W25.13 BOOL  ; 右机械手回#1模组位待料
W25.14 BOOL  ; 右机械手回#3模组位待料
W25.15 BOOL  ; 右机械手放料完成
W26 CHANNEL  ; #1模组手动状态
W26.00 BOOL  ; #1自检左气缸手动输出
W26.01 BOOL  ; #1自检右气缸手动输出
W26.02 BOOL  ; #1左密封气缸手动输出
W26.03 BOOL  ; #1右密封气缸手动输出
W26.04 BOOL  ; #1左夹爪气缸手动输出
W26.05 BOOL  ; #1右夹爪气缸手动输出
W26.06 BOOL  ; #1模组自检
W26.07 BOOL  ; #1左右自检气缸自检输出
W26.08 BOOL  ; #1左右密封气缸自检输出
W26.09 BOOL  ; #1检漏仪启动
W26.10 BOOL  ; #1自检结束
W26.11 BOOL  ; #1左右自检气缸自检缩回
W27 CHANNEL  ; #2模组手动状态
W27.00 BOOL  ; #2自检左气缸手动输出
W27.01 BOOL  ; #2自检右气缸手动输出
W27.02 BOOL  ; #2左密封气缸手动输出
W27.03 BOOL  ; #2右密封气缸手动输出
W27.04 BOOL  ; #2左夹爪气缸手动输出
W27.05 BOOL  ; #2右夹爪气缸手动输出
W27.06 BOOL  ; #2模组自检
W27.07 BOOL  ; #2左右自检气缸自检输出
W27.08 BOOL  ; #2左右密封气缸自检输出
W27.09 BOOL  ; #2检漏仪启动
W27.10 BOOL  ; #2自检结束
W27.11 BOOL  ; #2左右自检气缸自检缩回
W28 CHANNEL  ; #3模组手动状态
W28.00 BOOL  ; #3自检左气缸手动输出
W28.01 BOOL  ; #3自检右气缸手动输出
W28.02 BOOL  ; #3左密封气缸手动输出
W28.03 BOOL  ; #3右密封气缸手动输出
W28.04 BOOL  ; #3左夹爪气缸手动输出
W28.05 BOOL  ; #3右夹爪气缸手动输出
W28.06 BOOL  ; #3模组自检
W28.07 BOOL  ; #3左右自检气缸自检输出
W28.08 BOOL  ; #3左右密封气缸自检输出
W28.09 BOOL  ; #3检漏仪启动
W28.10 BOOL  ; #3自检结束
W28.11 BOOL  ; #3左右自检气缸自检缩回
W29 CHANNEL  ; #4模组手动状态
W29.00 BOOL  ; #4自检左气缸手动输出
W29.01 BOOL  ; #4自检右气缸手动输出
W29.02 BOOL  ; #4左密封气缸手动输出
W29.03 BOOL  ; #4右密封气缸手动输出
W29.04 BOOL  ; #4左夹爪气缸手动输出
W29.05 BOOL  ; #4右夹爪气缸手动输出
W29.06 BOOL  ; #4模组自检
W29.07 BOOL  ; #4左右自检气缸自检输出
W29.08 BOOL  ; #4左右密封气缸自检输出
W29.09 BOOL  ; #4检漏仪启动
W29.10 BOOL  ; #4自检结束
W29.11 BOOL  ; #4左右自检气缸自检缩回
W2.10 BOOL  ; 电脑启动-HMI
W30 CHANNEL  ; #1模组状态
W300 CHANNEL  ; 上料移栽报警状态
W300.00 BOOL  ; 异常
W300.01 BOOL  ; 移栽阻挡气缸伸出报警
W300.02 BOOL  ; 移栽#1电池到位超时报警
W300.03 BOOL  ; 移栽#2电池到位超时报警
W300.04 BOOL  ; 移栽伺服右限位报警
W300.05 BOOL  ; 移栽伺服左限位报警
W300.06 BOOL  ; 移栽伺服报警
W300.07 BOOL  ; 移栽伺服没就绪
W300.08 BOOL  ; 拉带与移栽处有料报警
W301 CHANNEL  ; 左机械手报警状态
W301.00 BOOL  ; 左机械手升降气缸缩回报警
W301.01 BOOL  ; 左机械手升降气缸伸出报警
W301.02 BOOL  ; 左机械手伸缩气缸缩回报警
W301.03 BOOL  ; 左机械手伸缩气缸伸出报警
W301.04 BOOL  ; 左机械手左夹爪张开报警
W301.05 BOOL  ; 左机械手左夹爪夹紧报警
W301.06 BOOL  ; 左机械手右夹爪张开报警
W301.07 BOOL  ; 左机械手右夹爪夹紧报警
W301.08 BOOL  ; 左机械手左限位报警
W301.09 BOOL  ; 左机械手右限位报警
W301.10 BOOL  ; 左#1电池放料有料异常
W301.11 BOOL  ; 左#2电池放料有俩异常
W301.12 BOOL  ; 左机械手伺服报警
W301.13 BOOL  ; 左机械手伺服没就绪
W301.14 BOOL  ; 左#1电池有料感应器异常
W301.15 BOOL  ; 左#2电池有料感应器异常
W303 CHANNEL  ; 右机械手报警状态
W303.00 BOOL  ; 右机械手升降气缸缩回报警
W303.01 BOOL  ; 右机械手升降气缸伸出报警
W303.02 BOOL  ; 右机械手伸缩气缸缩回报警
W303.03 BOOL  ; 右机械手伸缩气缸伸出报警
W303.04 BOOL  ; 右机械手左夹爪张开报警
W303.05 BOOL  ; 右机械手左夹爪夹紧报警
W303.06 BOOL  ; 右机械手右夹爪张开报警
W303.07 BOOL  ; 右机械手右夹爪夹紧报警
W303.08 BOOL  ; 右机械手左限位报警
W303.09 BOOL  ; 右机械手右限位报警
W303.10 BOOL  ; 右#1放料位有料异常报警
W303.11 BOOL  ; 右#2放料位有料异常报警
W303.12 BOOL  ; 右机械手伺服报警
W303.13 BOOL  ; 右机械手伺服没就绪
W303.14 BOOL  ; 右#1电池有料感应器异常
W303.15 BOOL  ; 右#2电池有料感应器异常
W305 CHANNEL  ; #1模组报警状态
W305.00 BOOL  ; #1左密封气缸缩回报警
W305.01 BOOL  ; #1左密封气缸伸出位报警
W305.02 BOOL  ; #1右密封气缸缩回位报警
W305.03 BOOL  ; #1右密封气缸伸出位报警
W305.04 BOOL  ; #1左夹料气缸张开报警
W305.05 BOOL  ; #1左夹料气缸夹紧报警
W305.06 BOOL  ; #1右夹料气缸张开报警
W305.07 BOOL  ; #1右夹料气缸夹紧报警
W305.08 BOOL  ; #1模组左有料异常报警
W305.09 BOOL  ; #1模组右有料异常报警
W305.10 BOOL  ; #1模组Busy信号异常报警
W305.11 BOOL  ; PC处理#1模组启动超时
W305.12 BOOL  ; PC处理#1模组测试完成超时
W306 CHANNEL  ; #2模组报警状态
W306.00 BOOL  ; #2左密封气缸缩回报警
W306.01 BOOL  ; #2左密封气缸伸出位报警
W306.02 BOOL  ; #2右密封气缸缩回位报警
W306.03 BOOL  ; #2右密封气缸伸出位报警
W306.04 BOOL  ; #2左夹料气缸张开报警
W306.05 BOOL  ; #2左夹料气缸夹紧报警
W306.06 BOOL  ; #2右夹料气缸张开报警
W306.07 BOOL  ; #2右夹料气缸夹紧报警
W306.08 BOOL  ; #2模组左有料异常报警
W306.09 BOOL  ; #2模组右有料异常报警
W306.10 BOOL  ; #2模组Busy信号异常报警
W306.11 BOOL  ; PC处理#2模组启动超时
W306.12 BOOL  ; PC处理#2模组测试完成超时
W307 CHANNEL  ; #3模组报警状态
W307.00 BOOL  ; #3左密封气缸缩回报警
W307.01 BOOL  ; #3左密封气缸伸出位报警
W307.02 BOOL  ; #3右密封气缸缩回位报警
W307.03 BOOL  ; #3右密封气缸伸出位报警
W307.04 BOOL  ; #3左夹料气缸张开报警
W307.05 BOOL  ; #3左夹料气缸夹紧报警
W307.06 BOOL  ; #3右夹料气缸张开报警
W307.07 BOOL  ; #3右夹料气缸夹紧报警
W307.08 BOOL  ; #3模组左有料异常报警
W307.09 BOOL  ; #3模组右有料异常报警
W307.10 BOOL  ; #3模组Busy信号异常报警
W307.11 BOOL  ; PC处理#3模组启动超时
W307.12 BOOL  ; PC处理#3模组测试完成超时
W308 CHANNEL  ; #4模组报警状态
W308.00 BOOL  ; #4左密封气缸缩回报警
W308.01 BOOL  ; #4左密封气缸伸出位报警
W308.02 BOOL  ; #4右密封气缸缩回位报警
W308.03 BOOL  ; #4右密封气缸伸出位报警
W308.04 BOOL  ; #4左夹料气缸张开报警
W308.05 BOOL  ; #4左夹料气缸夹紧报警
W308.06 BOOL  ; #4右夹料气缸张开报警
W308.07 BOOL  ; #4右夹料气缸夹紧报警
W308.08 BOOL  ; #4模组左有料异常报警
W308.09 BOOL  ; #4模组右有料异常报警
W308.10 BOOL  ; #4模组Busy信号异常报警
W308.11 BOOL  ; PC处理#4模组启动超时
W308.12 BOOL  ; PC处理#4模组测试完成超时
W309 CHANNEL  ; 龙门报警状态
W309.00 BOOL  ; #1下顶升左气缸缩回位报警
W309.01 BOOL  ; #1下顶升左气缸伸出位报警
W309.02 BOOL  ; #1下顶升右气缸缩回位报警
W309.03 BOOL  ; #1下顶升右气缸伸出位报警
W309.04 BOOL  ; #2下顶升左气缸缩回位报警
W309.05 BOOL  ; #2下顶升左气缸伸出位报警
W309.06 BOOL  ; #2下顶升右气缸缩回位报警
W309.07 BOOL  ; #2下顶升右气缸伸出位报警
W309.08 BOOL  ; 左拉带脱离气缸缩回位报警
W309.09 BOOL  ; 左拉带脱离气缸伸出位报警
W309.10 BOOL  ; 右拉带脱离气缸缩回位报警
W309.11 BOOL  ; 右拉带脱离气缸伸出位报警
W309.12 BOOL  ; 料盒定位气缸缩回位报警
W309.13 BOOL  ; 料盒定位气缸伸出位报警
W309.14 BOOL  ; 上料盒到位超时报警
W309.15 BOOL  ; 下料盒到位超时报警
W30.00 BOOL  ; #1左夹料气缸输出
W30.01 BOOL  ; #1右夹料气缸输出
W30.02 BOOL  ; #1左自检气缸输出
W30.03 BOOL  ; #1左密封气缸输出
W30.04 BOOL  ; #1右自检气缸输出
W30.05 BOOL  ; #1右密封气缸输出
W30.06 BOOL  ; #1检漏仪启动
W30.07 BOOL  ; #1检漏仪启动
W30.08 BOOL  ; #1氦检仪启动
W30.09 BOOL  ; #1左密封气缸到位屏蔽
W30.10 BOOL  ; #1右密封气缸到位屏蔽
W31 CHANNEL  ; #2模组状态
W310.00 BOOL  ; 料盒阻挡左气缸缩回报警
W310.01 BOOL  ; 料盒阻挡左气缸伸出报警
W310.02 BOOL  ; 料盒阻挡右气缸缩回报警
W310.03 BOOL  ; 料盒阻挡右气缸伸出报警
W310.04 BOOL  ; 料盒夹紧气缸伸出报警
W310.05 BOOL  ; 龙门前后伺服没就绪
W310.06 BOOL  ; 龙门左右伺服报警
W310.07 BOOL  ; 龙门左右伺服没就绪
W310.08 BOOL  ; 龙门升降柔性报警
W310.09 BOOL  ; 放料位有电池不能放料报警
W311.00 BOOL  ; 异常报警
W312 CHANNEL  ; 急停报警
W312.00 BOOL  ; 急停报警
W314 CHANNEL  ; 龙门升降报警状态
W314.00 BOOL  ; 龙门升降气缸缩回报警
W314.01 BOOL  ; 龙门升降气缸伸出报警
W314.02 BOOL  ; 龙门夹爪气缸张开报警
W314.03 BOOL  ; 龙门夹爪气缸夹紧报警
W314.04 BOOL  ; 龙门升降伺服报警
W314.05 BOOL  ; 龙门升降伺服没就绪
W314.06 BOOL  ; 检漏NG满输送带料满报警
W314.07 BOOL  ; 绝缘NG满输送带料满报警
W314.08 BOOL  ; 龙门升降柔性报警
W314.09 BOOL  ; 龙门升降上限位感应异常
W314.10 BOOL  ; 龙门升降下限位感应异常
W315 CHANNEL  ; 龙门前后，左右伺服报警
W315.00 BOOL  ; 龙门前后伺服报警
W315.01 BOOL  ; 龙门前后伺服没就绪
W315.02 BOOL  ; 龙门左右伺服报警
W315.03 BOOL  ; 龙门左右伺服没就绪
W315.04 BOOL  ; 龙门左右定位模块报警
W315.05 BOOL  ; 龙门前后定位模块报警
W315.06 BOOL  ; 龙门前后伺服前限位异常
W315.07 BOOL  ; 龙门前后伺服后限位异常
W315.08 BOOL  ; 龙门左右伺服右限位报警
W315.09 BOOL  ; 龙门左右伺服左限位报警
W316 CHANNEL  ; 料盒升降伺服报警
W316.00 BOOL  ; 料盒升降伺服报警
W316.01 BOOL  ; 料盒升降伺服没就绪
W316.02 BOOL  ; 料盒升降定位模块异常
W316.03 BOOL  ; 料盒升降伺服下限位报警
W316.04 BOOL  ; 料盒升降伺服上限位报警
W317 CHANNEL  ; 上料机构报警
W317.00 BOOL  ; 上料阻挡气缸缩回报警
W317.01 BOOL  ; 上料阻挡气缸伸出报警
W317.02 BOOL  ; 检测气缸缩回报警
W317.03 BOOL  ; 检测气缸伸出报警
W317.04 BOOL  ; 扫码超时
W317.05 BOOL  ; 检测超时
W318.00 BOOL  ; 第一排#1电池有料异常
W318.01 BOOL  ; 第一排#2电池有料异常
W318.02 BOOL  ; 第一排#3电池有料异常
W318.03 BOOL  ; 第一排#4电池有料异常
W318.04 BOOL  ; 第一排#5电池有料异常
W318.05 BOOL  ; 第一排#6电池有料异常
W318.06 BOOL  ; 第一排#7电池有料异常
W318.07 BOOL  ; 第一排#8电池有料异常
W318.08 BOOL  ; 第一排#9电池有料异常
W318.09 BOOL  ; 第一排#10电池有料异常
W318.10 BOOL  ; 第一排#11电池有料异常
W318.11 BOOL  ; 第一排#12电池有料异常
W319.00 BOOL  ; 第二排#1电池有料异常
W319.01 BOOL  ; 第二排#2电池有料异常
W319.02 BOOL  ; 第二排#3电池有料异常
W319.03 BOOL  ; 第二排#4电池有料异常
W319.04 BOOL  ; 第二排#5电池有料异常
W319.05 BOOL  ; 第二排#6电池有料异常
W319.06 BOOL  ; 第二排#7电池有料异常
W319.07 BOOL  ; 第二排#8电池有料异常
W319.08 BOOL  ; 第二排#9电池有料异常
W319.09 BOOL  ; 第二排#10电池有料异常
W319.10 BOOL  ; 第二排#11电池有料异常
W319.11 BOOL  ; 第二排#12电池有料异常
W31.00 BOOL  ; #2左夹料气缸输出
W31.01 BOOL  ; #2右夹料气缸输出
W31.02 BOOL  ; #2左自检气缸输出
W31.03 BOOL  ; #2左密封气缸输出
W31.04 BOOL  ; #2右自检气缸输出
W31.05 BOOL  ; #2右密封气缸输出
W31.06 BOOL  ; #2检漏仪启动
W31.07 BOOL  ; #2检漏仪启动
W31.08 BOOL  ; #2氦检仪启动
W31.09 BOOL  ; #2左密封气缸到位屏蔽
W31.10 BOOL  ; #2右密封气缸到位屏蔽
W32 CHANNEL  ; #3模组状态
W32.00 BOOL  ; #3左夹料气缸输出
W32.01 BOOL  ; #3右夹料气缸输出
W32.02 BOOL  ; #3左自检气缸输出
W32.03 BOOL  ; #3左密封气缸输出
W32.04 BOOL  ; #3右自检气缸输出
W32.05 BOOL  ; #3右密封气缸输出
W32.06 BOOL  ; #3检漏仪启动
W32.07 BOOL  ; #3检漏仪启动
W32.08 BOOL  ; #3氦检仪启动
W32.09 BOOL  ; #3左密封气缸到位屏蔽
W32.10 BOOL  ; #3右密封气缸到位屏蔽
W33 CHANNEL  ; #4模组状态
W33.00 BOOL  ; #4左夹料气缸输出
W33.01 BOOL  ; #4右夹料气缸输出
W33.02 BOOL  ; #4左自检气缸输出
W33.03 BOOL  ; #4左密封气缸输出
W33.04 BOOL  ; #4右自检气缸输出
W33.05 BOOL  ; #4右密封气缸输出
W33.06 BOOL  ; #4检漏仪启动
W33.07 BOOL  ; #4检漏仪启动
W33.08 BOOL  ; #4氦检仪启动
W33.09 BOOL  ; #4左密封气缸到位屏蔽
W33.10 BOOL  ; #4右密封气缸到位屏蔽
W34.00 BOOL  ; 龙门升降在取料位置
W34.01 BOOL  ; 龙门升降在绝缘NG位置
W34.02 BOOL  ; 龙门升降在测试NG位置
W34.03 BOOL  ; 龙门升降在OK位置
W34.04 BOOL  ; 龙门升降归零
W34.05 BOOL  ; 龙门升降上升
W34.06 BOOL  ; 龙门升降下降
W34.07 BOOL  ; 龙门升降取料位置
W34.08 BOOL  ; 龙门升降OK放料位置
W34.09 BOOL  ; 龙门升降绝缘NG位置
W34.10 BOOL  ; 龙门升降测试NG位置
W34.11 BOOL  ; 料盒升降伺服手动归零
W34.12 BOOL  ; 料盒升降伺服手动下降
W34.13 BOOL  ; 料盒升降伺服手动上升
W34.14 BOOL  ; 料盒升降伺服手动回上料盒位置
W34.15 BOOL  ; 料盒升降伺服手动回放料盒位置
W35.00 BOOL  ; 龙门前后伺服手动归零
W35.01 BOOL  ; 龙门前后手动前进
W35.02 BOOL  ; 龙门前后手动后退
W35.03 BOOL  ; 龙门左右伺服手动归零
W35.04 BOOL  ; 龙门左右手动左移
W35.05 BOOL  ; 龙门左右手动右移
W35.06 BOOL  ; 龙门回#1左取料位
W35.07 BOOL  ; 龙门回#2左取料位
W35.08 BOOL  ; 龙门回#1右取料位
W35.09 BOOL  ; 龙门回#2右取料位
W35.10 BOOL  ; 龙门回#1放料位
W35.11 BOOL  ; 龙门回#2放料位
W35.12 BOOL  ; 龙门前后在#3位置
W35.13 BOOL  ; 龙门回#4放料位
W35.14 BOOL  ; 龙门回#5放料位
W35.15 BOOL  ; 龙门回#6放料位
W36.00 BOOL  ; 龙门回#7放料位
W36.01 BOOL  ; 龙门回#8放料位
W36.02 BOOL  ; 龙门回#9放料位
W36.03 BOOL  ; 龙门回#10放料位
W36.04 BOOL  ; 龙门回#11位放料
W36.05 BOOL  ; 龙门回#12放料位
W36.06 BOOL  ; 龙门回#13放料位
W36.07 BOOL  ; 龙门回#14放料位
W36.08 BOOL  ; 龙门回#15放料位
W36.09 BOOL  ; 龙门回#16放料位
W36.10 BOOL  ; 龙门回#17放料位
W36.11 BOOL  ; 龙门回#18放料位
W36.12 BOOL  ; 龙门回#19放料位
W36.13 BOOL  ; 龙门回#20放料位
W36.14 BOOL  ; 龙门回#21放料位
W36.15 BOOL  ; 龙门回#22放料位
W37.00 BOOL  ; 龙门回#23放料位
W37.01 BOOL  ; 龙门回#24放料位
W37.02 BOOL  ; 龙门回绝缘NG放料位
W37.03 BOOL  ; 龙门回检漏NG放料位
W37.04 BOOL  ; 龙门回检漏NG放料位
W38 CHANNEL  ; 龙门前后运动状态
W38.00 BOOL  ; 龙门前后手动回#1左取料位
W38.01 BOOL  ; 龙门前后手动回#2左取料位
W38.02 BOOL  ; 龙门前后手动回#1右取料位
W38.03 BOOL  ; 龙门前后手动回#2右取料位
W38.04 BOOL  ; 龙门前后手动回#1放料位
W38.05 BOOL  ; 龙门前后手动回#2放料位
W38.06 BOOL  ; 龙门前后手动回#3放料位
W38.07 BOOL  ; 龙门前后手动回#4放料位
W38.08 BOOL  ; 龙门前后手动回#5放料位
W38.09 BOOL  ; 龙门前后手动回#6放料位
W38.10 BOOL  ; 龙门前后手动回#7放料位
W38.11 BOOL  ; 龙门前后手动回#8放料位
W38.12 BOOL  ; 龙门前后手动回#9放料位
W38.13 BOOL  ; 龙门前后手动回#10放料位
W38.14 BOOL  ; 龙门前后手动回#11放料位
W38.15 BOOL  ; 龙门前后手动回#12放料位
W39 CHANNEL  ; 龙门前后运动状态
W39.00 BOOL  ; 龙门前后手动回#13放料位
W39.01 BOOL  ; 龙门前后手动回#14放料位
W39.02 BOOL  ; 龙门前后手动回#15放料位
W39.03 BOOL  ; 龙门前后手动回#16放料位
W39.04 BOOL  ; 龙门前后手动回#17放料位
W39.05 BOOL  ; 龙门前后手动回#18放料位
W39.06 BOOL  ; 龙门前后手动回#19放料位
W39.07 BOOL  ; 龙门前后手动回#20放料位
W39.08 BOOL  ; 龙门前后手动回#21放料位
W39.09 BOOL  ; 龙门前后手动回#22放料位
W39.10 BOOL  ; 龙门前后手动回#23放料位
W39.11 BOOL  ; 龙门前后手动回#24放料位
W39.12 BOOL  ; 龙门前后手动回绝缘NG放料位
W39.13 BOOL  ; 龙门前后手动回检漏NG放料位
W3.00 BOOL  ; 左机械手归零-HMI
W3.01 BOOL  ; 左机械手后退-HMI
W3.02 BOOL  ; 左机械手前进-HMI
W3.03 BOOL  ; 上料位置-HMI
W3.04 BOOL  ; 下料位置-HMI
W3.05 BOOL  ; #2模组位置-HMI
W3.06 BOOL  ; #4模组位置-HMI
W3.07 BOOL  ; 升降气缸-HMI
W3.08 BOOL  ; 伸缩气缸-HMI
W3.09 BOOL  ; 左夹爪-HMI
W3.10 BOOL  ; 右夹爪-HMI
W40 CHANNEL  ; 龙门左右运动状态
W40.00 BOOL  ; 龙门左右手动回#1左取料位
W40.01 BOOL  ; 龙门左右手动回#2左取料位
W40.02 BOOL  ; 龙门左右手动回#1右取料位
W40.03 BOOL  ; 龙门左右手动回#2右取料位
W40.04 BOOL  ; 龙门左右手动回#1放料位
W40.05 BOOL  ; 龙门左右手动回#2放料位
W40.06 BOOL  ; 龙门左右手动回#3放料位
W40.07 BOOL  ; 龙门左右手动回#4放料位
W40.08 BOOL  ; 龙门左右手动回#5放料位
W40.09 BOOL  ; 龙门左右手动回#6放料位
W40.10 BOOL  ; 龙门左右手动回#7放料位
W40.11 BOOL  ; 龙门左右手动回#8放料位
W40.12 BOOL  ; 龙门左右手动回#9放料位
W40.13 BOOL  ; 龙门左右手动回#10放料位
W40.14 BOOL  ; 龙门左右手动回#11放料位
W40.15 BOOL  ; 龙门左右手动回#12放料位
W41 CHANNEL  ; 龙门左右运动状态
W41.00 BOOL  ; 龙门左右手动回#13放料位
W41.01 BOOL  ; 龙门左右手动回#14放料位
W41.02 BOOL  ; 龙门左右手动回#15放料位
W41.03 BOOL  ; 龙门左右手动回#16放料位
W41.04 BOOL  ; 龙门左右手动回#17放料位
W41.05 BOOL  ; 龙门左右手动回#18放料位
W41.06 BOOL  ; 龙门左右手动回#19放料位
W41.07 BOOL  ; 龙门左右手动回#20放料位
W41.08 BOOL  ; 龙门左右手动回#21放料位
W41.09 BOOL  ; 龙门左右手动回#22放料位
W41.10 BOOL  ; 龙门左右手动回#23放料位
W41.11 BOOL  ; 龙门左右手动回#24放料位
W41.12 BOOL  ; 龙门左右手动回绝缘NG放料位
W41.13 BOOL  ; 龙门左右手动回检漏NG放料位
W42 CHANNEL  ; 龙门机构手动状态
W42.00 BOOL  ; 龙门升降气缸手动输出
W42.01 BOOL  ; 龙门夹爪气缸手动伸出
W42.02 BOOL  ; #1上顶升气缸手动伸出
W42.03 BOOL  ; #2上顶升气缸手动输出
W42.04 BOOL  ; #1下顶升气缸手动输出
W42.05 BOOL  ; #2下顶升气缸手动输出
W42.06 BOOL  ; 料盒阻挡气缸手动输出
W42.07 BOOL  ; 料盒定位气缸手动输出
W42.08 BOOL  ; 左脱离气缸手动输出
W42.09 BOOL  ; 右脱离气缸手动输出
W42.10 BOOL  ; 料盒上料电机手动输出
W42.11 BOOL  ; 下料缓存电机手动输出
W42.12 BOOL  ; 料盒下料电机手动输出
W42.13 BOOL  ; 绝缘NG电机
W42.14 BOOL  ; 检漏NG电机
W42.15 BOOL  ; 料盘气缸夹紧
W43.00 BOOL  ; 料盘气缸松开
W44 CHANNEL  ; 龙门状态
W44.01 BOOL  ; 料盒平移安全条件
W44.02 BOOL  ; 龙门XY到达第一排指定位置
W44.03 BOOL  ; 龙门XY到达第二排指定位置
W45 CHANNEL  ; 龙门状态
W45.06 BOOL  ; 龙门升降回OK放料位置
W46 CHANNEL  ; 龙门第一排位置
W46.01 BOOL  ; 第一排#1没料
W46.02 BOOL  ; 第一排#2没料
W46.03 BOOL  ; 第一排#3没料
W46.04 BOOL  ; 第一排#4没料
W46.05 BOOL  ; 第一排#5没料
W46.06 BOOL  ; 第一排#6没料
W46.07 BOOL  ; 第一排#7没料
W46.08 BOOL  ; 第一排#8没料
W46.09 BOOL  ; 第一排#9没料
W46.10 BOOL  ; 第一排#10没料
W46.11 BOOL  ; 第一排#11没料
W46.12 BOOL  ; 第一排#12没料
W46.13 BOOL  ; 第一排料满
W47 CHANNEL  ; 龙门第二排位置
W47.00 BOOL  ; 第二排没料
W47.01 BOOL  ; 第二排#1没料
W47.02 BOOL  ; 第二排#2没料
W47.03 BOOL  ; 第二排#3没料
W47.04 BOOL  ; 第二排#4没料
W47.05 BOOL  ; 第二排#5没料
W47.06 BOOL  ; 第二排#6没料
W47.07 BOOL  ; 第二排#7没料
W47.08 BOOL  ; 第二排#8没料
W47.09 BOOL  ; 第二排#9没料
W47.10 BOOL  ; 第二排#10没料
W47.11 BOOL  ; 第二排#11没料
W47.12 BOOL  ; 第二排#12没料
W48 CHANNEL  ; 龙门XY回第一排的位置
W49 CHANNEL  ; 龙门XY第一排所处位置
W4.00 BOOL  ; 右机械手归零-HMI
W4.01 BOOL  ; 右机械手后退-HMI
W4.02 BOOL  ; 右机械手前进-HMI
W4.03 BOOL  ; 上料位置-HMI
W4.04 BOOL  ; 下料位置-HMI
W4.05 BOOL  ; #1模组位置-HMI
W4.06 BOOL  ; #3模组位置-HMI
W4.07 BOOL  ; 升降气缸-HMI
W4.08 BOOL  ; 伸缩气缸-HMI
W4.09 BOOL  ; 左夹爪-HMI
W4.10 BOOL  ; 右夹爪-HMI
W500.00 BOOL  ; 调试
W500.01 BOOL  ; 调试
W5.00 BOOL  ; 自检左气缸-HMI
W5.01 BOOL  ; 自检右气缸-HMI
W5.02 BOOL  ; 左密封气缸-HMI
W5.03 BOOL  ; 右密封气缸-HMI
W5.04 BOOL  ; 左夹爪气缸-HMI
W5.05 BOOL  ; 右夹爪气缸-HMI
W5.06 BOOL  ; #1自检-HMI
W5.07 BOOL  ; 自检左气缸-HMI
W5.08 BOOL  ; 自检右气缸-HMI
W5.09 BOOL  ; 左密封气缸-HMI
W5.10 BOOL  ; 右密封气缸-HMI
W5.11 BOOL  ; 左夹爪气缸-HMI
W5.12 BOOL  ; 右夹爪气缸-HMI
W5.13 BOOL  ; #3自检-HMI
W6.00 BOOL  ; 自检左气缸-HMI
W6.01 BOOL  ; 自检右气缸-HMI
W6.02 BOOL  ; 左密封气缸-HMI
W6.03 BOOL  ; 右密封气缸-HMI
W6.04 BOOL  ; 左夹爪气缸-HMI
W6.05 BOOL  ; 右夹爪气缸-HMI
W6.06 BOOL  ; #2自检-HMI
W6.07 BOOL  ; 自检左气缸-HMI
W6.08 BOOL  ; 自检右气缸-HMI
W6.09 BOOL  ; 左密封气缸-HMI
W6.10 BOOL  ; 右密封气缸-HMI
W6.11 BOOL  ; 左夹爪气缸-HMI
W6.12 BOOL  ; 右夹爪气缸-HMI
W6.13 BOOL  ; #4自检-HMI
W7.00 BOOL  ; 龙门升降归零-HMI
W7.01 BOOL  ; 龙门升降上升-HMI
W7.02 BOOL  ; 龙门升降下降-HMI
W7.03 BOOL  ; 龙门取料位置-HMI
W7.04 BOOL  ; 龙门OK位置-HMI
W7.05 BOOL  ; 龙门绝缘NG位置
W7.06 BOOL  ; 龙门测试NG位置
W7.07 BOOL  ; 料盒升降归零-HMI
W7.08 BOOL  ; 料盒下降-HMI
W7.09 BOOL  ; 料盒上升-HMI
W7.10 BOOL  ; 上料盒位置-HMI
W7.11 BOOL  ; 下料盒位置-HMI
W7.12 BOOL  ; #1上顶升气缸-HMI
W7.13 BOOL  ; #2上顶升气缸-HMI
W7.14 BOOL  ; #1下顶升气缸-HMI
W7.15 BOOL  ; #2下顶升气缸-HMI
W8.00 BOOL  ; 料盒阻挡气缸-HMI
W8.01 BOOL  ; 料盒定位气缸-HMI
W8.02 BOOL  ; 左脱离气缸-HMI
W8.03 BOOL  ; 右脱离气缸-HMI
W8.04 BOOL  ; 龙门升降气缸-HMI
W8.05 BOOL  ; 龙门夹爪气缸-HMI
W8.06 BOOL  ; 料盒上料电机-HMI
W8.07 BOOL  ; 下料缓存电机-HMI
W8.08 BOOL  ; 料盒下料电机-HMI
W8.09 BOOL  ; 绝缘NG电机-HMI
W8.10 BOOL  ; 检漏NG电机-HMI
W8.11 BOOL  ; 料盘气缸夹紧-HMI
W9 CHANNEL  ; 龙门左右手动-HMI
W9.00 BOOL  ; 龙门前后归零-HMI
W9.01 BOOL  ; 龙门前后前进-HMI
W9.02 BOOL  ; 龙门前后后退-HMI
W9.03 BOOL  ; 龙门左右归零-HMI
W9.04 BOOL  ; 龙门左右左移-HMI
W9.05 BOOL  ; 龙门左右右移-HMI
W9.06 BOOL  ; #1左取料位-HMI
W9.07 BOOL  ; #2左取料位-HMI
W9.08 BOOL  ; #1右取料位-HMI
W9.09 BOOL  ; #2右取料位-HMI
W9.10 BOOL  ; #1放料位-HMI
W9.11 BOOL  ; #2放料位-HMI
W9.12 BOOL  ; #3放料位-HMI
W9.13 BOOL  ; #4放料位-HMI
W9.14 BOOL  ; #5放料位-HMI
W9.15 BOOL  ; #6放料位-HMI

## Program 主程序 (cyclic task 0)

### Section Main

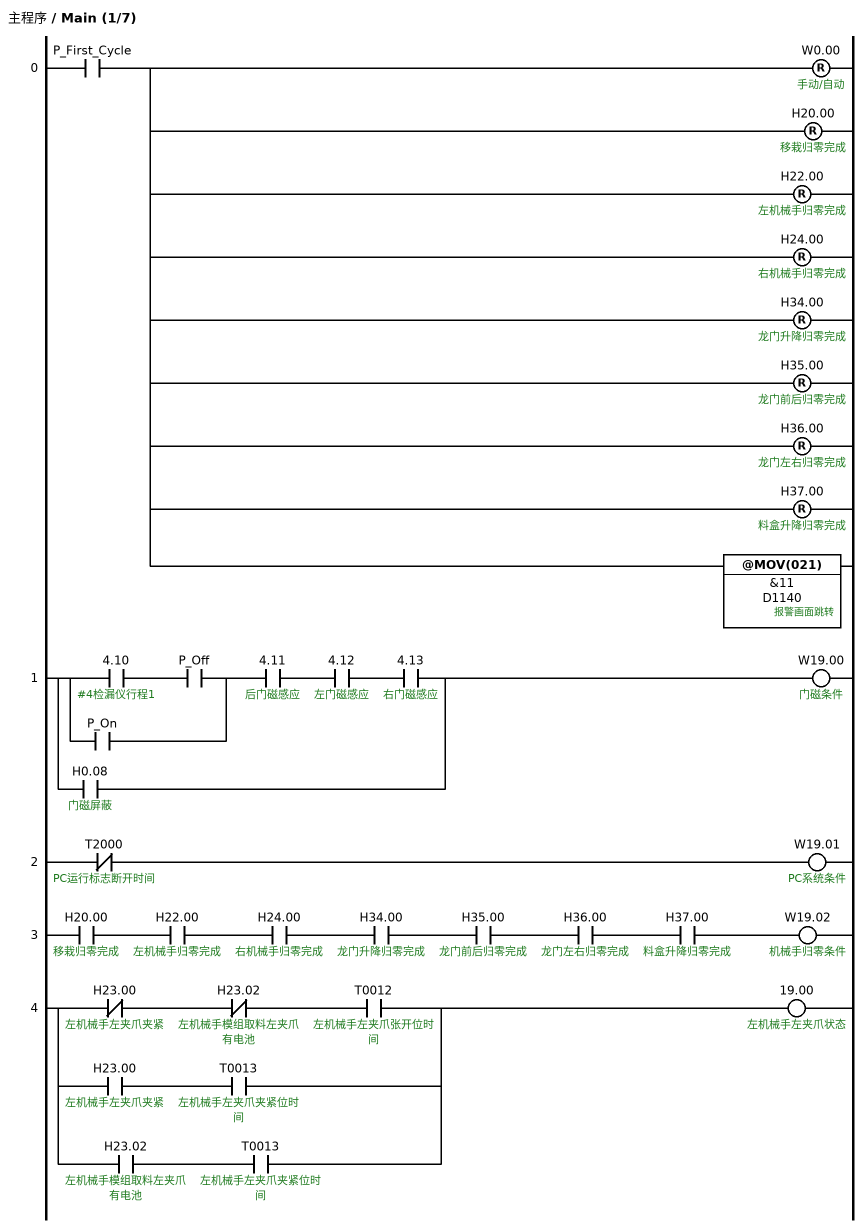
; rung 0
LD P_First_Cycle
RSET W0.00  ; 手动/自动
RSET H20.00  ; 移栽归零完成
RSET H22.00  ; 左机械手归零完成
RSET H24.00  ; 右机械手归零完成
RSET H34.00  ; 龙门升降归零完成
RSET H35.00  ; 龙门前后归零完成
RSET H36.00  ; 龙门左右归零完成
RSET H37.00  ; 料盒升降归零完成
@MOV(021) &11 D1140  ; 报警画面跳转
; rung 1
LD 4.10  ; #4检漏仪行程1
AND P_Off
OR P_On
AND 4.11  ; 后门磁感应
AND 4.12  ; 左门磁感应
AND 4.13  ; 右门磁感应
OR H0.08  ; 门磁屏蔽
OUT W19.00  ; 门磁条件
; rung 2
LDNOT T2000  ; PC运行标志断开时间
OUT W19.01  ; PC系统条件
; rung 3
LD H20.00  ; 移栽归零完成
AND H22.00  ; 左机械手归零完成
AND H24.00  ; 右机械手归零完成
AND H34.00  ; 龙门升降归零完成
AND H35.00  ; 龙门前后归零完成
AND H36.00  ; 龙门左右归零完成
AND H37.00  ; 料盒升降归零完成
OUT W19.02  ; 机械手归零条件
; rung 4
LDNOT H23.00  ; 左机械手左夹爪夹紧
ANDNOT H23.02  ; 左机械手模组取料左夹爪有电池
AND T0012  ; 左机械手左夹爪张开位时间
LD H23.00  ; 左机械手左夹爪夹紧
AND T0013  ; 左机械手左夹爪夹紧位时间
ORLD
LD H23.02  ; 左机械手模组取料左夹爪有电池
AND T0013  ; 左机械手左夹爪夹紧位时间
ORLD
OUT 19.00  ; 左机械手左夹爪状态

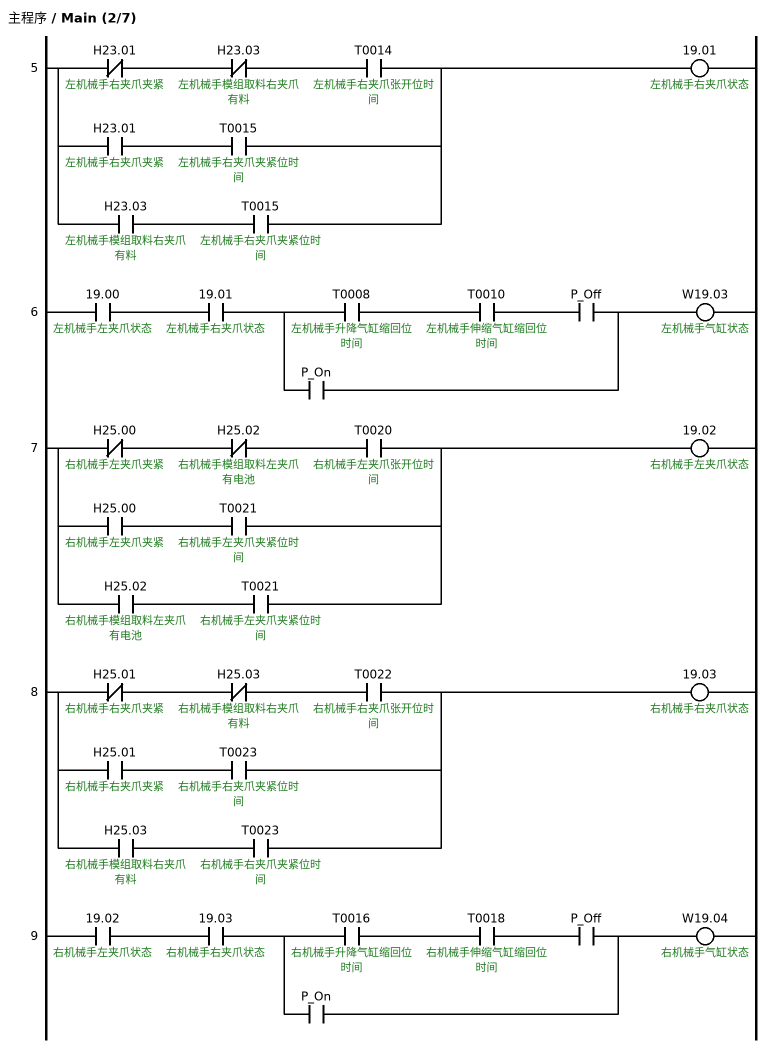
; rung 5
LDNOT H23.01  ; 左机械手右夹爪夹紧
ANDNOT H23.03  ; 左机械手模组取料右夹爪有料
AND T0014  ; 左机械手右夹爪张开位时间
LD H23.01  ; 左机械手右夹爪夹紧
AND T0015  ; 左机械手右夹爪夹紧位时间
ORLD
LD H23.03  ; 左机械手模组取料右夹爪有料
AND T0015  ; 左机械手右夹爪夹紧位时间
ORLD
OUT 19.01  ; 左机械手右夹爪状态
; rung 6
LD 19.00  ; 左机械手左夹爪状态
AND 19.01  ; 左机械手右夹爪状态
LD T0008  ; 左机械手升降气缸缩回位时间
AND T0010  ; 左机械手伸缩气缸缩回位时间
AND P_Off
OR P_On
ANDLD
OUT W19.03  ; 左机械手气缸状态
; rung 7
LDNOT H25.00  ; 右机械手左夹爪夹紧
ANDNOT H25.02  ; 右机械手模组取料左夹爪有电池
AND T0020  ; 右机械手左夹爪张开位时间
LD H25.00  ; 右机械手左夹爪夹紧
AND T0021  ; 右机械手左夹爪夹紧位时间
ORLD
LD H25.02  ; 右机械手模组取料左夹爪有电池
AND T0021  ; 右机械手左夹爪夹紧位时间
ORLD
OUT 19.02  ; 右机械手左夹爪状态
; rung 8
LDNOT H25.01  ; 右机械手右夹爪夹紧
ANDNOT H25.03  ; 右机械手模组取料右夹爪有料
AND T0022  ; 右机械手右夹爪张开位时间
LD H25.01  ; 右机械手右夹爪夹紧
AND T0023  ; 右机械手右夹爪夹紧位时间
ORLD
LD H25.03  ; 右机械手模组取料右夹爪有料
AND T0023  ; 右机械手右夹爪夹紧位时间
ORLD
OUT 19.03  ; 右机械手右夹爪状态
; rung 9
LD 19.02  ; 右机械手左夹爪状态
AND 19.03  ; 右机械手右夹爪状态
LD T0016  ; 右机械手升降气缸缩回位时间
AND T0018  ; 右机械手伸缩气缸缩回位时间
AND P_Off
OR P_On
ANDLD
OUT W19.04  ; 右机械手气缸状态

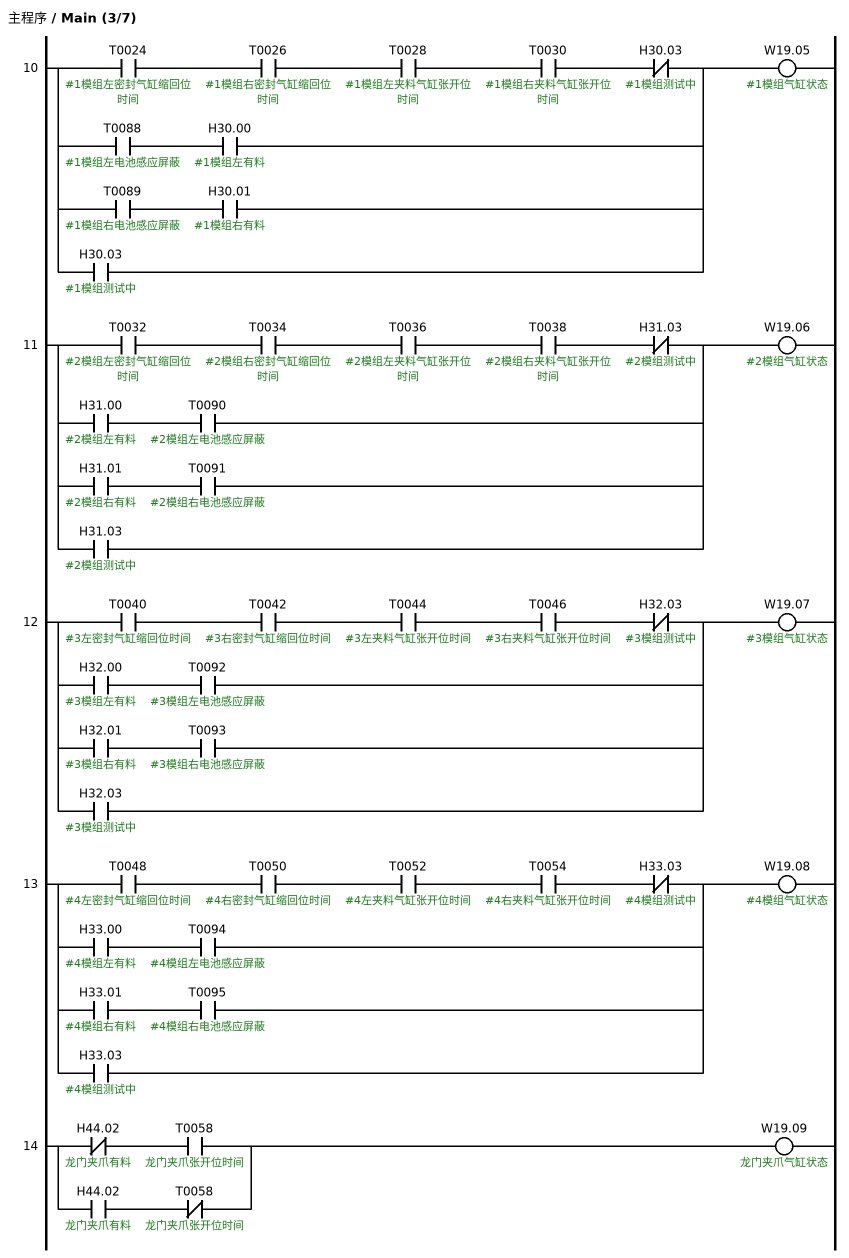
; rung 10
LD T0024  ; #1模组左密封气缸缩回位时间
AND T0026  ; #1模组右密封气缸缩回位时间
AND T0028  ; #1模组左夹料气缸张开位时间
AND T0030  ; #1模组右夹料气缸张开位时间
ANDNOT H30.03  ; #1模组测试中
LD T0088  ; #1模组左电池感应屏蔽
AND H30.00  ; #1模组左有料
ORLD
LD T0089  ; #1模组右电池感应屏蔽
AND H30.01  ; #1模组右有料
ORLD
OR H30.03  ; #1模组测试中
OUT W19.05  ; #1模组气缸状态
; rung 11
LD T0032  ; #2模组左密封气缸缩回位时间
AND T0034  ; #2模组右密封气缸缩回位时间
AND T0036  ; #2模组左夹料气缸张开位时间
AND T0038  ; #2模组右夹料气缸张开位时间
ANDNOT H31.03  ; #2模组测试中
LD H31.00  ; #2模组左有料
AND T0090  ; #2模组左电池感应屏蔽
ORLD
LD H31.01  ; #2模组右有料
AND T0091  ; #2模组右电池感应屏蔽
ORLD
OR H31.03  ; #2模组测试中
OUT W19.06  ; #2模组气缸状态
; rung 12
LD T0040  ; #3左密封气缸缩回位时间
AND T0042  ; #3右密封气缸缩回位时间
AND T0044  ; #3左夹料气缸张开位时间
AND T0046  ; #3右夹料气缸张开位时间
ANDNOT H32.03  ; #3模组测试中
LD H32.00  ; #3模组左有料
AND T0092  ; #3模组左电池感应屏蔽
ORLD
LD H32.01  ; #3模组右有料
AND T0093  ; #3模组右电池感应屏蔽
ORLD
OR H32.03  ; #3模组测试中
OUT W19.07  ; #3模组气缸状态
; rung 13
LD T0048  ; #4左密封气缸缩回位时间
AND T0050  ; #4右密封气缸缩回位时间
AND T0052  ; #4左夹料气缸张开位时间
AND T0054  ; #4右夹料气缸张开位时间
ANDNOT H33.03  ; #4模组测试中
LD H33.00  ; #4模组左有料
AND T0094  ; #4模组左电池感应屏蔽
ORLD
LD H33.01  ; #4模组右有料
AND T0095  ; #4模组右电池感应屏蔽
ORLD
OR H33.03  ; #4模组测试中
OUT W19.08  ; #4模组气缸状态
; rung 14
LDNOT H44.02  ; 龙门夹爪有料
AND T0058  ; 龙门夹爪张开位时间
LD H44.02  ; 龙门夹爪有料
ANDNOT T0058  ; 龙门夹爪张开位时间
ORLD
OUT W19.09  ; 龙门夹爪气缸状态

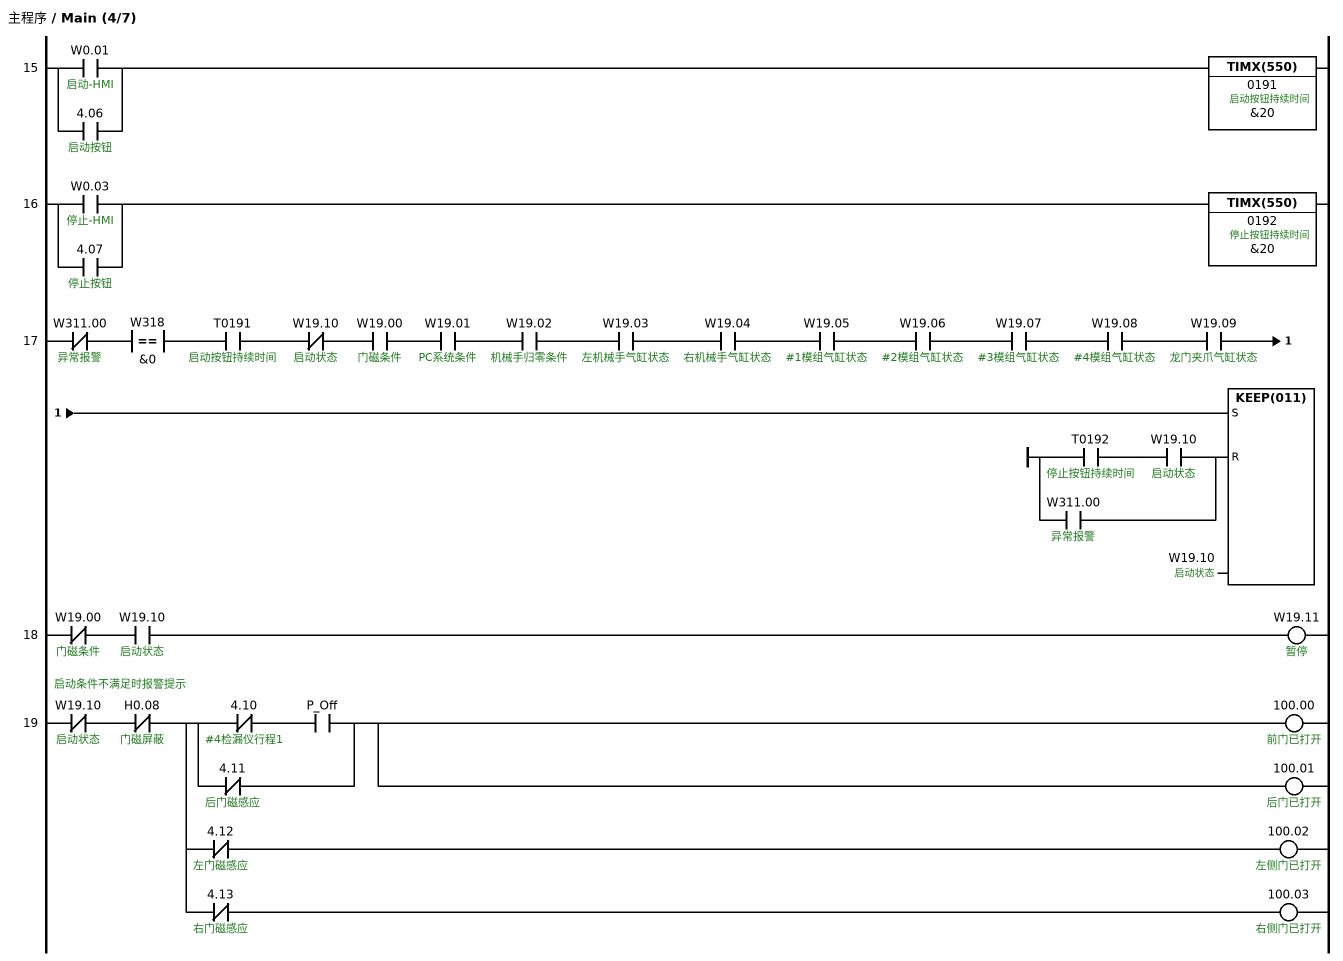
; rung 15
LD W0.01  ; 启动-HMI
OR 4.06  ; 启动按钮
TIMX(550) 0191 &20  ; 启动按钮持续时间
; rung 16
LD W0.03  ; 停止-HMI
OR 4.07  ; 停止按钮
TIMX(550) 0192 &20  ; 停止按钮持续时间
; rung 17
LDNOT W311.00  ; 异常报警
AND=L(301) W318 &0
AND T0191  ; 启动按钮持续时间
ANDNOT W19.10  ; 启动状态
AND W19.00  ; 门磁条件
AND W19.01  ; PC系统条件
AND W19.02  ; 机械手归零条件
AND W19.03  ; 左机械手气缸状态
AND W19.04  ; 右机械手气缸状态
AND W19.05  ; #1模组气缸状态
AND W19.06  ; #2模组气缸状态
AND W19.07  ; #3模组气缸状态
AND W19.08  ; #4模组气缸状态
AND W19.09  ; 龙门夹爪气缸状态
LD T0192  ; 停止按钮持续时间
AND W19.10  ; 启动状态
OR W311.00  ; 异常报警
KEEP(011) W19.10  ; 启动状态
; rung 18
LDNOT W19.00  ; 门磁条件
AND W19.10  ; 启动状态
OUT W19.11  ; 暂停
; rung 19: 启动条件不满足时报警提示
LDNOT W19.10  ; 启动状态
ANDNOT H0.08  ; 门磁屏蔽
OUT TR0
LDNOT 4.10  ; #4检漏仪行程1
AND P_Off
ORNOT 4.11  ; 后门磁感应
ANDLD
OUT 100.00  ; 前门已打开
OUT 100.01  ; 后门已打开
LD TR0
ANDNOT 4.12  ; 左门磁感应
OUT 100.02  ; 左侧门已打开
LD TR0
ANDNOT 4.13  ; 右门磁感应
OUT 100.03  ; 右侧门已打开

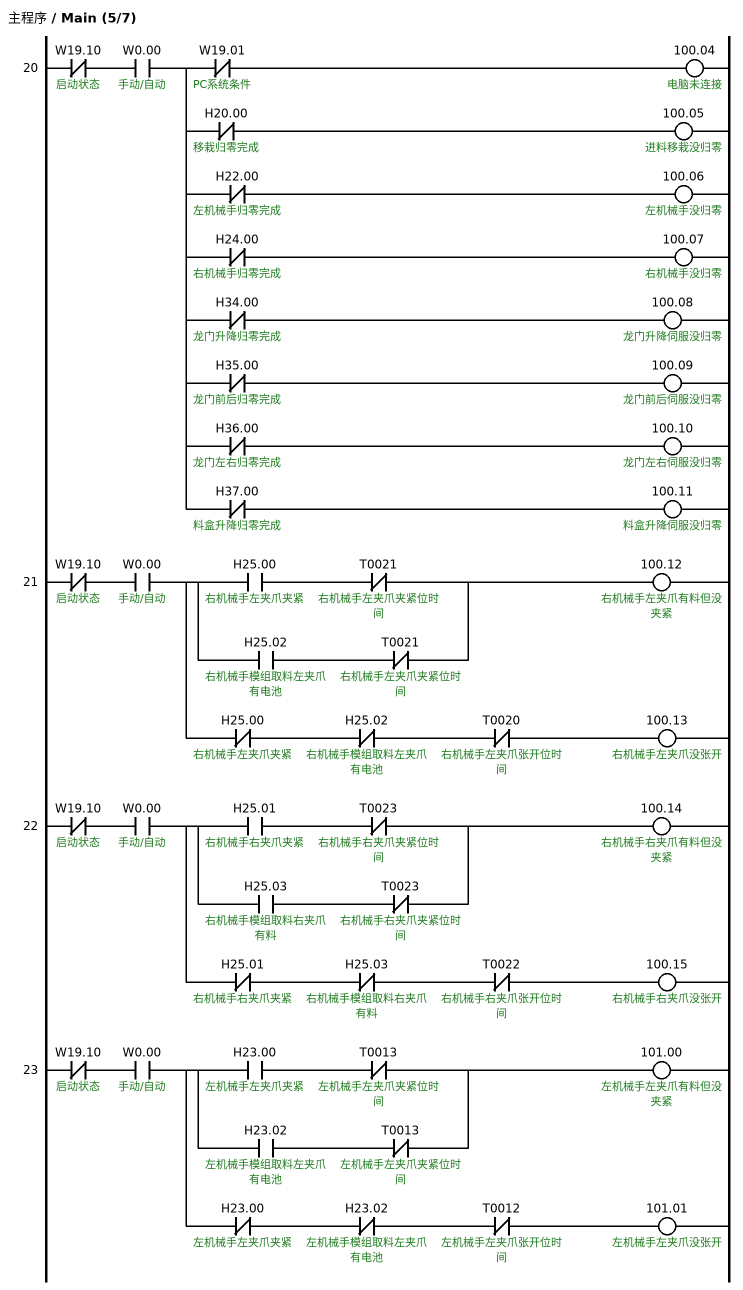
; rung 20
LDNOT W19.10  ; 启动状态
AND W0.00  ; 手动/自动
OUT TR0
ANDNOT W19.01  ; PC系统条件
OUT 100.04  ; 电脑未连接
LD TR0
ANDNOT H20.00  ; 移栽归零完成
OUT 100.05  ; 进料移栽没归零
LD TR0
ANDNOT H22.00  ; 左机械手归零完成
OUT 100.06  ; 左机械手没归零
LD TR0
ANDNOT H24.00  ; 右机械手归零完成
OUT 100.07  ; 右机械手没归零
LD TR0
ANDNOT H34.00  ; 龙门升降归零完成
OUT 100.08  ; 龙门升降伺服没归零
LD TR0
ANDNOT H35.00  ; 龙门前后归零完成
OUT 100.09  ; 龙门前后伺服没归零
LD TR0
ANDNOT H36.00  ; 龙门左右归零完成
OUT 100.10  ; 龙门左右伺服没归零
LD TR0
ANDNOT H37.00  ; 料盒升降归零完成
OUT 100.11  ; 料盒升降伺服没归零
; rung 21
LDNOT W19.10  ; 启动状态
AND W0.00  ; 手动/自动
OUT TR0
LD H25.00  ; 右机械手左夹爪夹紧
ANDNOT T0021  ; 右机械手左夹爪夹紧位时间
LD H25.02  ; 右机械手模组取料左夹爪有电池
ANDNOT T0021  ; 右机械手左夹爪夹紧位时间
ORLD
ANDLD
OUT 100.12  ; 右机械手左夹爪有料但没夹紧
LD TR0
ANDNOT H25.00  ; 右机械手左夹爪夹紧
ANDNOT H25.02  ; 右机械手模组取料左夹爪有电池
ANDNOT T0020  ; 右机械手左夹爪张开位时间
OUT 100.13  ; 右机械手左夹爪没张开
; rung 22
LDNOT W19.10  ; 启动状态
AND W0.00  ; 手动/自动
OUT TR0
LD H25.01  ; 右机械手右夹爪夹紧
ANDNOT T0023  ; 右机械手右夹爪夹紧位时间
LD H25.03  ; 右机械手模组取料右夹爪有料
ANDNOT T0023  ; 右机械手右夹爪夹紧位时间
ORLD
ANDLD
OUT 100.14  ; 右机械手右夹爪有料但没夹紧
LD TR0
ANDNOT H25.01  ; 右机械手右夹爪夹紧
ANDNOT H25.03  ; 右机械手模组取料右夹爪有料
ANDNOT T0022  ; 右机械手右夹爪张开位时间
OUT 100.15  ; 右机械手右夹爪没张开
; rung 23
LDNOT W19.10  ; 启动状态
AND W0.00  ; 手动/自动
OUT TR0
LD H23.00  ; 左机械手左夹爪夹紧
ANDNOT T0013  ; 左机械手左夹爪夹紧位时间
LD H23.02  ; 左机械手模组取料左夹爪有电池
ANDNOT T0013  ; 左机械手左夹爪夹紧位时间
ORLD
ANDLD
OUT 101.00  ; 左机械手左夹爪有料但没夹紧
LD TR0
ANDNOT H23.00  ; 左机械手左夹爪夹紧
ANDNOT H23.02  ; 左机械手模组取料左夹爪有电池
ANDNOT T0012  ; 左机械手左夹爪张开位时间
OUT 101.01  ; 左机械手左夹爪没张开

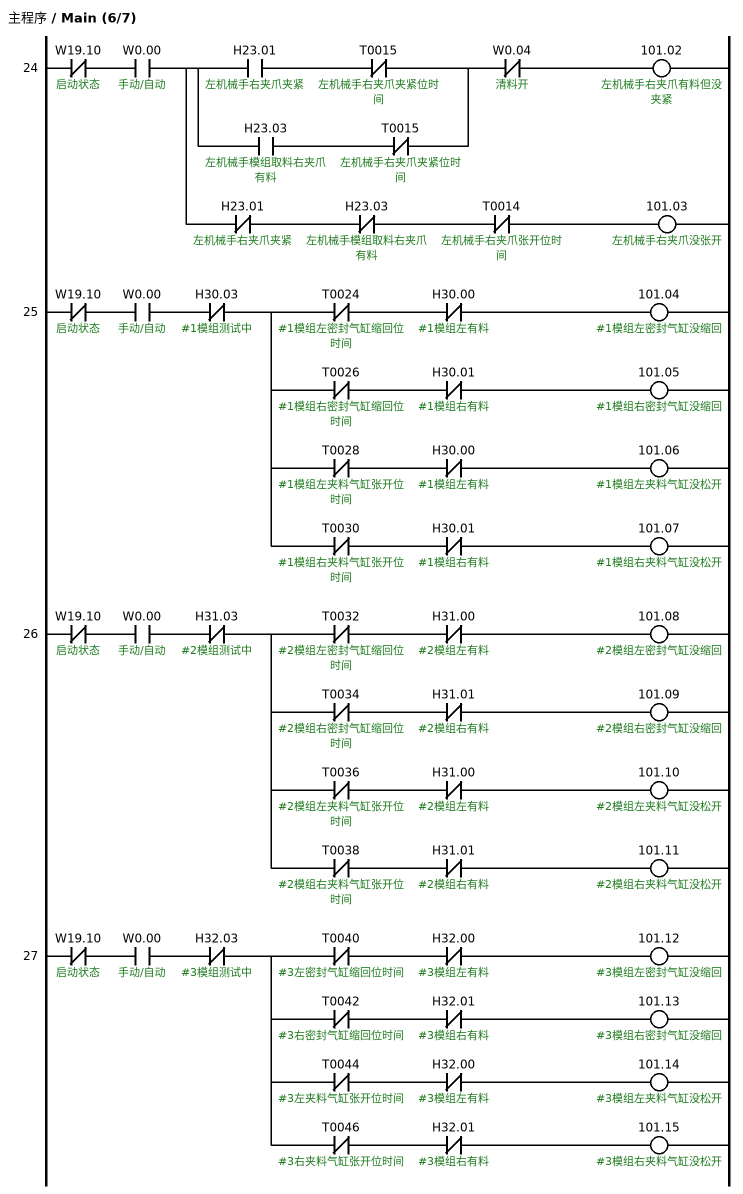
; rung 24
LDNOT W19.10  ; 启动状态
AND W0.00  ; 手动/自动
OUT TR0
LD H23.01  ; 左机械手右夹爪夹紧
ANDNOT T0015  ; 左机械手右夹爪夹紧位时间
LD H23.03  ; 左机械手模组取料右夹爪有料
ANDNOT T0015  ; 左机械手右夹爪夹紧位时间
ORLD
ANDLD
ANDNOT W0.04  ; 清料开
OUT 101.02  ; 左机械手右夹爪有料但没夹紧
LD TR0
ANDNOT H23.01  ; 左机械手右夹爪夹紧
ANDNOT H23.03  ; 左机械手模组取料右夹爪有料
ANDNOT T0014  ; 左机械手右夹爪张开位时间
OUT 101.03  ; 左机械手右夹爪没张开
; rung 25
LDNOT W19.10  ; 启动状态
AND W0.00  ; 手动/自动
ANDNOT H30.03  ; #1模组测试中
OUT TR0
ANDNOT T0024  ; #1模组左密封气缸缩回位时间
ANDNOT H30.00  ; #1模组左有料
OUT 101.04  ; #1模组左密封气缸没缩回
LD TR0
ANDNOT T0026  ; #1模组右密封气缸缩回位时间
ANDNOT H30.01  ; #1模组右有料
OUT 101.05  ; #1模组右密封气缸没缩回
LD TR0
ANDNOT T0028  ; #1模组左夹料气缸张开位时间
ANDNOT H30.00  ; #1模组左有料
OUT 101.06  ; #1模组左夹料气缸没松开
LD TR0
ANDNOT T0030  ; #1模组右夹料气缸张开位时间
ANDNOT H30.01  ; #1模组右有料
OUT 101.07  ; #1模组右夹料气缸没松开
; rung 26
LDNOT W19.10  ; 启动状态
AND W0.00  ; 手动/自动
ANDNOT H31.03  ; #2模组测试中
OUT TR0
ANDNOT T0032  ; #2模组左密封气缸缩回位时间
ANDNOT H31.00  ; #2模组左有料
OUT 101.08  ; #2模组左密封气缸没缩回
LD TR0
ANDNOT T0034  ; #2模组右密封气缸缩回位时间
ANDNOT H31.01  ; #2模组右有料
OUT 101.09  ; #2模组右密封气缸没缩回
LD TR0
ANDNOT T0036  ; #2模组左夹料气缸张开位时间
ANDNOT H31.00  ; #2模组左有料
OUT 101.10  ; #2模组左夹料气缸没松开
LD TR0
ANDNOT T0038  ; #2模组右夹料气缸张开位时间
ANDNOT H31.01  ; #2模组右有料
OUT 101.11  ; #2模组右夹料气缸没松开
; rung 27
LDNOT W19.10  ; 启动状态
AND W0.00  ; 手动/自动
ANDNOT H32.03  ; #3模组测试中
OUT TR0
ANDNOT T0040  ; #3左密封气缸缩回位时间
ANDNOT H32.00  ; #3模组左有料
OUT 101.12  ; #3模组左密封气缸没缩回
LD TR0
ANDNOT T0042  ; #3右密封气缸缩回位时间
ANDNOT H32.01  ; #3模组右有料
OUT 101.13  ; #3模组右密封气缸没缩回
LD TR0
ANDNOT T0044  ; #3左夹料气缸张开位时间
ANDNOT H32.00  ; #3模组左有料
OUT 101.14  ; #3模组左夹料气缸没松开
LD TR0
ANDNOT T0046  ; #3右夹料气缸张开位时间
ANDNOT H32.01  ; #3模组右有料
OUT 101.15  ; #3模组右夹料气缸没松开

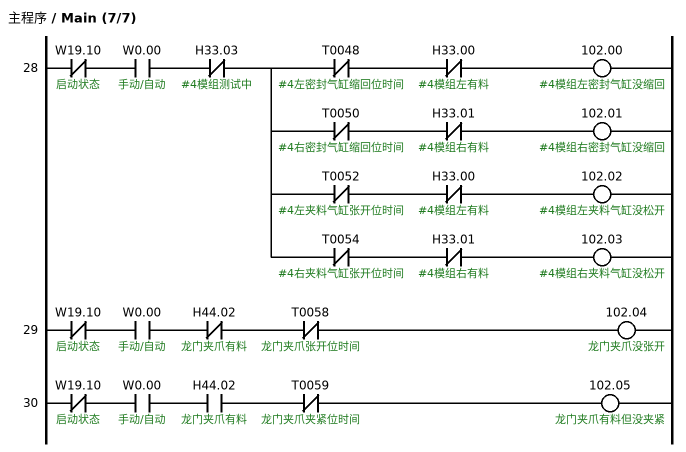
; rung 28
LDNOT W19.10  ; 启动状态
AND W0.00  ; 手动/自动
ANDNOT H33.03  ; #4模组测试中
OUT TR0
ANDNOT T0048  ; #4左密封气缸缩回位时间
ANDNOT H33.00  ; #4模组左有料
OUT 102.00  ; #4模组左密封气缸没缩回
LD TR0
ANDNOT T0050  ; #4右密封气缸缩回位时间
ANDNOT H33.01  ; #4模组右有料
OUT 102.01  ; #4模组右密封气缸没缩回
LD TR0
ANDNOT T0052  ; #4左夹料气缸张开位时间
ANDNOT H33.00  ; #4模组左有料
OUT 102.02  ; #4模组左夹料气缸没松开
LD TR0
ANDNOT T0054  ; #4右夹料气缸张开位时间
ANDNOT H33.01  ; #4模组右有料
OUT 102.03  ; #4模组右夹料气缸没松开
; rung 29
LDNOT W19.10  ; 启动状态
AND W0.00  ; 手动/自动
ANDNOT H44.02  ; 龙门夹爪有料
ANDNOT T0058  ; 龙门夹爪张开位时间
OUT 102.04  ; 龙门夹爪没张开
; rung 30
LDNOT W19.10  ; 启动状态
AND W0.00  ; 手动/自动
AND H44.02  ; 龙门夹爪有料
ANDNOT T0059  ; 龙门夹爪夹紧位时间
OUT 102.05  ; 龙门夹爪有料但没夹紧

### Section 外部输出

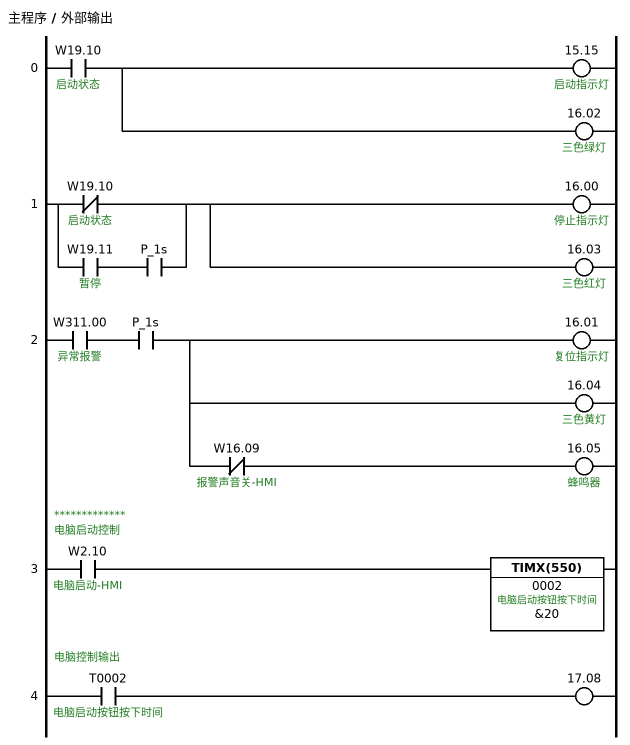
; rung 0
LD W19.10  ; 启动状态
OUT 15.15  ; 启动指示灯
OUT 16.02  ; 三色绿灯
; rung 1
LDNOT W19.10  ; 启动状态
LD W19.11  ; 暂停
AND P_1s
ORLD
OUT 16.00  ; 停止指示灯
OUT 16.03  ; 三色红灯
; rung 2
LD W311.00  ; 异常报警
AND P_1s
OUT 16.01  ; 复位指示灯
OUT 16.04  ; 三色黄灯
ANDNOT W16.09  ; 报警声音关-HMI
OUT 16.05  ; 蜂鸣器
; rung 3: ************* / 电脑启动控制
LD W2.10  ; 电脑启动-HMI
TIMX(550) 0002 &20  ; 电脑启动按钮按下时间
; rung 4: 电脑控制输出
LD T0002  ; 电脑启动按钮按下时间
OUT 17.08

### Section 异常报警复位

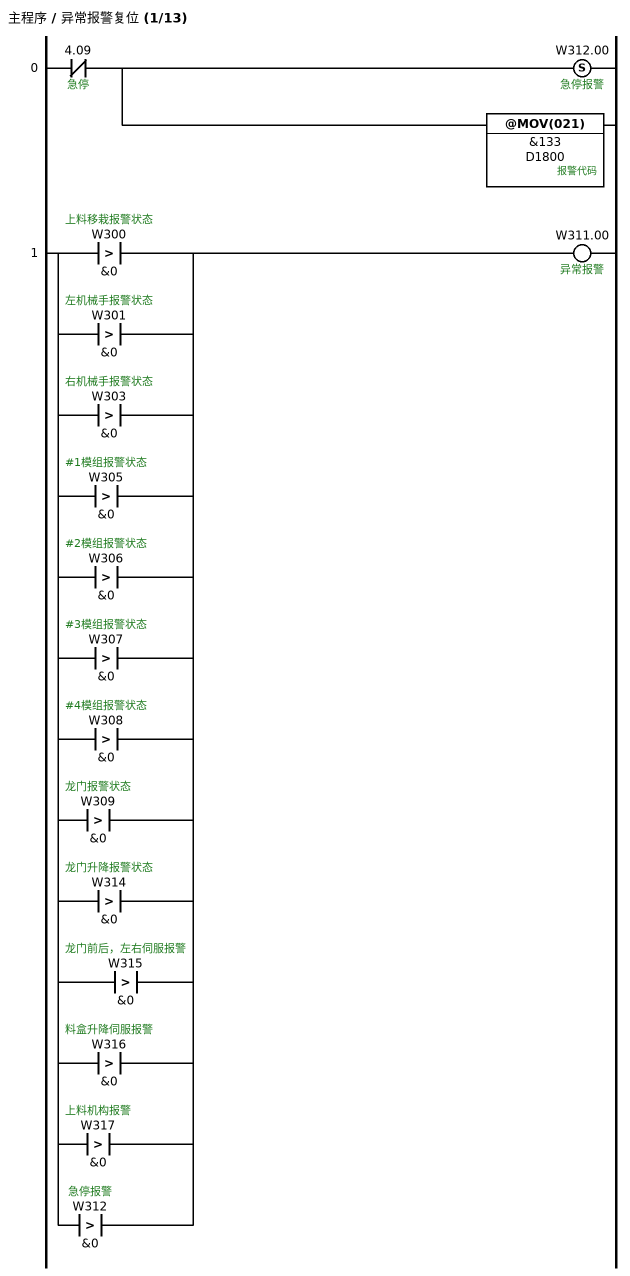
; rung 0
LDNOT 4.09  ; 急停
SET W312.00  ; 急停报警
@MOV(021) &133 D1800  ; 报警代码
; rung 1
LD>(320) W300 &0  ; 上料移栽报警状态
OR>L(321) W301 &0  ; 左机械手报警状态
OR>L(321) W303 &0  ; 右机械手报警状态
OR>(320) W305 &0  ; #1模组报警状态
OR>(320) W306 &0  ; #2模组报警状态
OR>(320) W307 &0  ; #3模组报警状态
OR>(320) W308 &0  ; #4模组报警状态
OR>L(321) W309 &0  ; 龙门报警状态
OR>(320) W314 &0  ; 龙门升降报警状态
OR>(320) W315 &0  ; 龙门前后，左右伺服报警
OR>(320) W316 &0  ; 料盒升降伺服报警
OR>(320) W317 &0  ; 上料机构报警
OR>(320) W312 &0  ; 急停报警
OUT W311.00  ; 异常报警

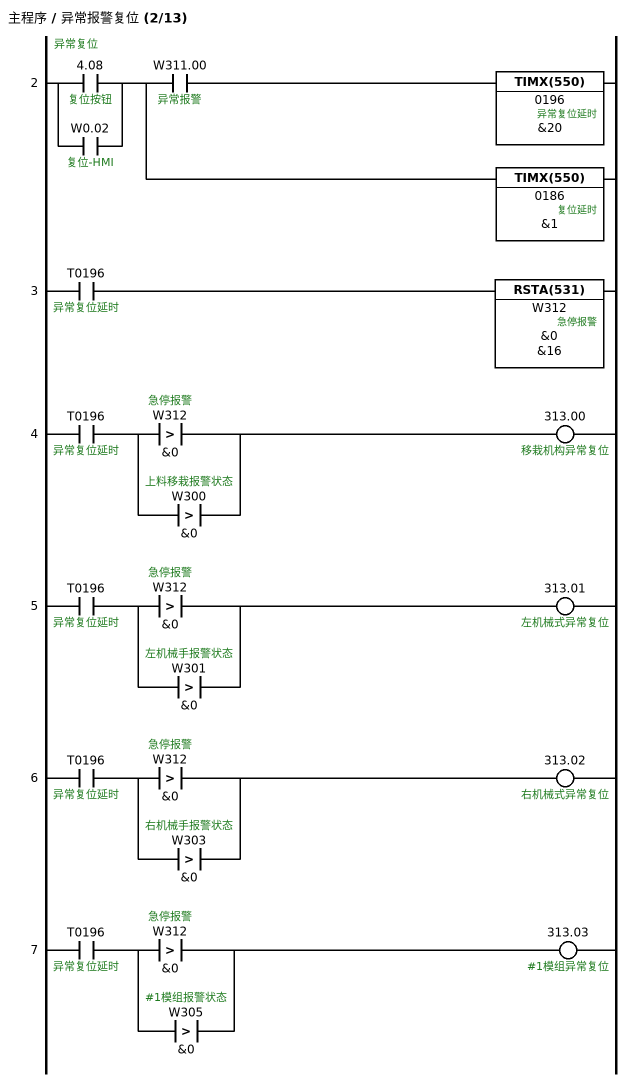
; rung 2: 异常复位
LD 4.08  ; 复位按钮
OR W0.02  ; 复位-HMI
OUT TR0
AND W311.00  ; 异常报警
TIMX(550) 0196 &20  ; 异常复位延时
LD TR0
TIMX(550) 0186 &1  ; 复位延时
; rung 3
LD T0196  ; 异常复位延时
RSTA(531) W312 &0 &16  ; 急停报警
; rung 4
LD T0196  ; 异常复位延时
LD>(320) W312 &0  ; 急停报警
OR>(320) W300 &0  ; 上料移栽报警状态
ANDLD
OUT 313.00  ; 移栽机构异常复位
; rung 5
LD T0196  ; 异常复位延时
LD>(320) W312 &0  ; 急停报警
OR>L(321) W301 &0  ; 左机械手报警状态
ANDLD
OUT 313.01  ; 左机械式异常复位
; rung 6
LD T0196  ; 异常复位延时
LD>(320) W312 &0  ; 急停报警
OR>L(321) W303 &0  ; 右机械手报警状态
ANDLD
OUT 313.02  ; 右机械式异常复位
; rung 7
LD T0196  ; 异常复位延时
LD>(320) W312 &0  ; 急停报警
OR>(320) W305 &0  ; #1模组报警状态
ANDLD
OUT 313.03  ; #1模组异常复位

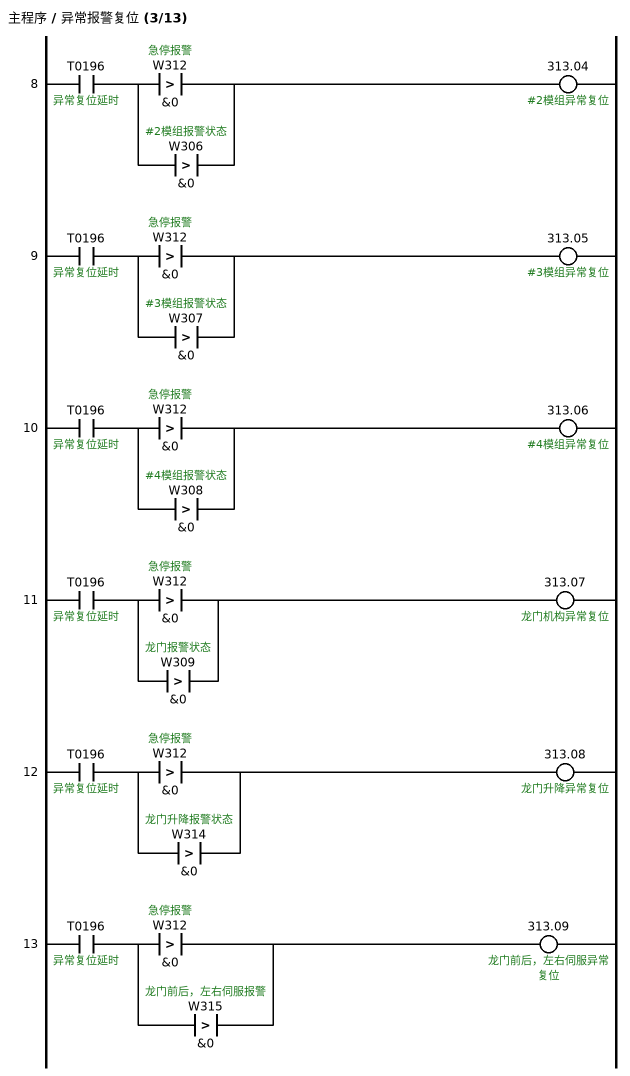
; rung 8
LD T0196  ; 异常复位延时
LD>(320) W312 &0  ; 急停报警
OR>(320) W306 &0  ; #2模组报警状态
ANDLD
OUT 313.04  ; #2模组异常复位
; rung 9
LD T0196  ; 异常复位延时
LD>(320) W312 &0  ; 急停报警
OR>(320) W307 &0  ; #3模组报警状态
ANDLD
OUT 313.05  ; #3模组异常复位
; rung 10
LD T0196  ; 异常复位延时
LD>(320) W312 &0  ; 急停报警
OR>(320) W308 &0  ; #4模组报警状态
ANDLD
OUT 313.06  ; #4模组异常复位
; rung 11
LD T0196  ; 异常复位延时
LD>(320) W312 &0  ; 急停报警
OR>L(321) W309 &0  ; 龙门报警状态
ANDLD
OUT 313.07  ; 龙门机构异常复位
; rung 12
LD T0196  ; 异常复位延时
LD>(320) W312 &0  ; 急停报警
OR>(320) W314 &0  ; 龙门升降报警状态
ANDLD
OUT 313.08  ; 龙门升降异常复位
; rung 13
LD T0196  ; 异常复位延时
LD>(320) W312 &0  ; 急停报警
OR>(320) W315 &0  ; 龙门前后，左右伺服报警
ANDLD
OUT 313.09  ; 龙门前后，左右伺服异常复位

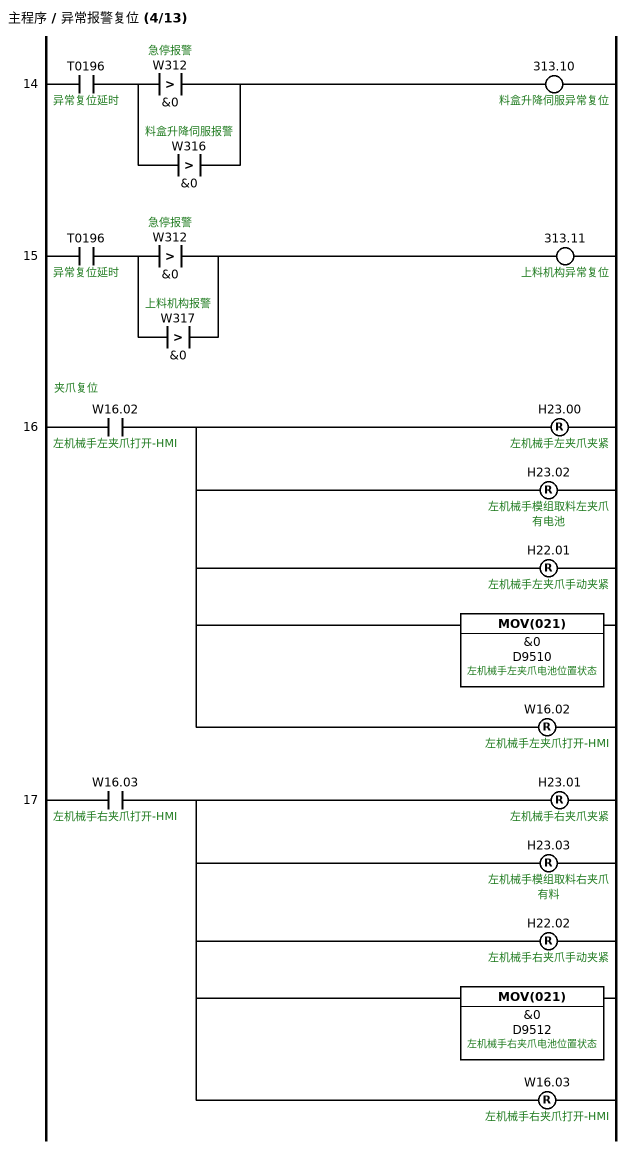
; rung 14
LD T0196  ; 异常复位延时
LD>(320) W312 &0  ; 急停报警
OR>(320) W316 &0  ; 料盒升降伺服报警
ANDLD
OUT 313.10  ; 料盒升降伺服异常复位
; rung 15
LD T0196  ; 异常复位延时
LD>(320) W312 &0  ; 急停报警
OR>(320) W317 &0  ; 上料机构报警
ANDLD
OUT 313.11  ; 上料机构异常复位
; rung 16: 夹爪复位
LD W16.02  ; 左机械手左夹爪打开-HMI
RSET H23.00  ; 左机械手左夹爪夹紧
RSET H23.02  ; 左机械手模组取料左夹爪有电池
RSET H22.01  ; 左机械手左夹爪手动夹紧
MOV(021) &0 D9510  ; 左机械手左夹爪电池位置状态
RSET W16.02  ; 左机械手左夹爪打开-HMI
; rung 17
LD W16.03  ; 左机械手右夹爪打开-HMI
RSET H23.01  ; 左机械手右夹爪夹紧
RSET H23.03  ; 左机械手模组取料右夹爪有料
RSET H22.02  ; 左机械手右夹爪手动夹紧
MOV(021) &0 D9512  ; 左机械手右夹爪电池位置状态
RSET W16.03  ; 左机械手右夹爪打开-HMI

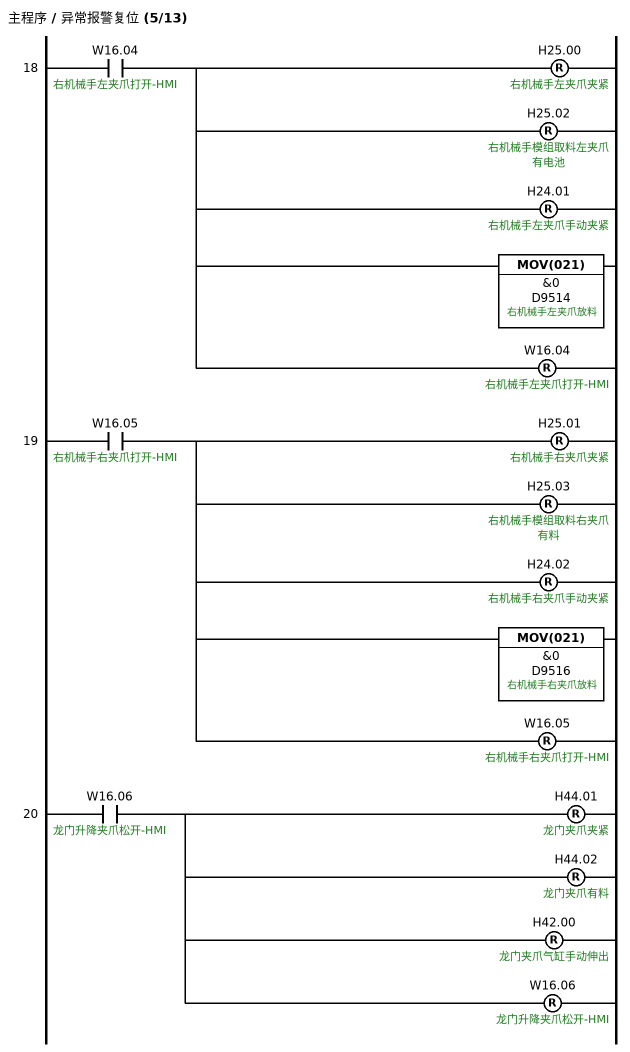
; rung 18
LD W16.04  ; 右机械手左夹爪打开-HMI
RSET H25.00  ; 右机械手左夹爪夹紧
RSET H25.02  ; 右机械手模组取料左夹爪有电池
RSET H24.01  ; 右机械手左夹爪手动夹紧
MOV(021) &0 D9514  ; 右机械手左夹爪放料
RSET W16.04  ; 右机械手左夹爪打开-HMI
; rung 19
LD W16.05  ; 右机械手右夹爪打开-HMI
RSET H25.01  ; 右机械手右夹爪夹紧
RSET H25.03  ; 右机械手模组取料右夹爪有料
RSET H24.02  ; 右机械手右夹爪手动夹紧
MOV(021) &0 D9516  ; 右机械手右夹爪放料
RSET W16.05  ; 右机械手右夹爪打开-HMI
; rung 20
LD W16.06  ; 龙门升降夹爪松开-HMI
RSET H44.01  ; 龙门夹爪夹紧
RSET H44.02  ; 龙门夹爪有料
RSET H42.00  ; 龙门夹爪气缸手动伸出
RSET W16.06  ; 龙门升降夹爪松开-HMI

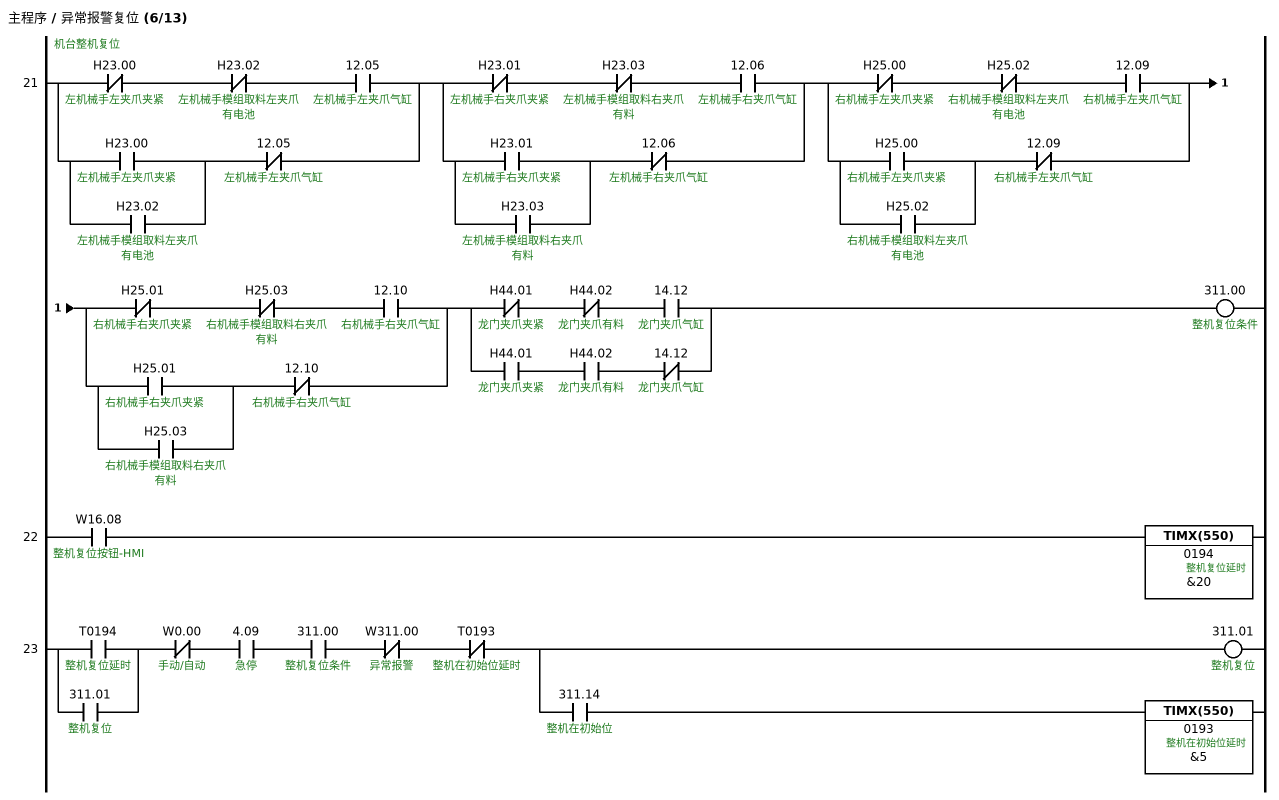
; rung 21: 机台整机复位
LDNOT H23.00  ; 左机械手左夹爪夹紧
ANDNOT H23.02  ; 左机械手模组取料左夹爪有电池
AND 12.05  ; 左机械手左夹爪气缸
LD H23.00  ; 左机械手左夹爪夹紧
OR H23.02  ; 左机械手模组取料左夹爪有电池
ANDNOT 12.05  ; 左机械手左夹爪气缸
ORLD
LDNOT H23.01  ; 左机械手右夹爪夹紧
ANDNOT H23.03  ; 左机械手模组取料右夹爪有料
AND 12.06  ; 左机械手右夹爪气缸
LD H23.01  ; 左机械手右夹爪夹紧
OR H23.03  ; 左机械手模组取料右夹爪有料
ANDNOT 12.06  ; 左机械手右夹爪气缸
ORLD
ANDLD
LDNOT H25.00  ; 右机械手左夹爪夹紧
ANDNOT H25.02  ; 右机械手模组取料左夹爪有电池
AND 12.09  ; 右机械手左夹爪气缸
LD H25.00  ; 右机械手左夹爪夹紧
OR H25.02  ; 右机械手模组取料左夹爪有电池
ANDNOT 12.09  ; 右机械手左夹爪气缸
ORLD
ANDLD
LDNOT H25.01  ; 右机械手右夹爪夹紧
ANDNOT H25.03  ; 右机械手模组取料右夹爪有料
AND 12.10  ; 右机械手右夹爪气缸
LD H25.01  ; 右机械手右夹爪夹紧
OR H25.03  ; 右机械手模组取料右夹爪有料
ANDNOT 12.10  ; 右机械手右夹爪气缸
ORLD
ANDLD
LDNOT H44.01  ; 龙门夹爪夹紧
ANDNOT H44.02  ; 龙门夹爪有料
AND 14.12  ; 龙门夹爪气缸
LD H44.01  ; 龙门夹爪夹紧
AND H44.02  ; 龙门夹爪有料
ANDNOT 14.12  ; 龙门夹爪气缸
ORLD
ANDLD
OUT 311.00  ; 整机复位条件
; rung 22
LD W16.08  ; 整机复位按钮-HMI
TIMX(550) 0194 &20  ; 整机复位延时
; rung 23
LD T0194  ; 整机复位延时
OR 311.01  ; 整机复位
ANDNOT W0.00  ; 手动/自动
AND 4.09  ; 急停
AND 311.00  ; 整机复位条件
ANDNOT W311.00  ; 异常报警
ANDNOT T0193  ; 整机在初始位延时
OUT 311.01  ; 整机复位
AND 311.14  ; 整机在初始位
TIMX(550) 0193 &5  ; 整机在初始位延时

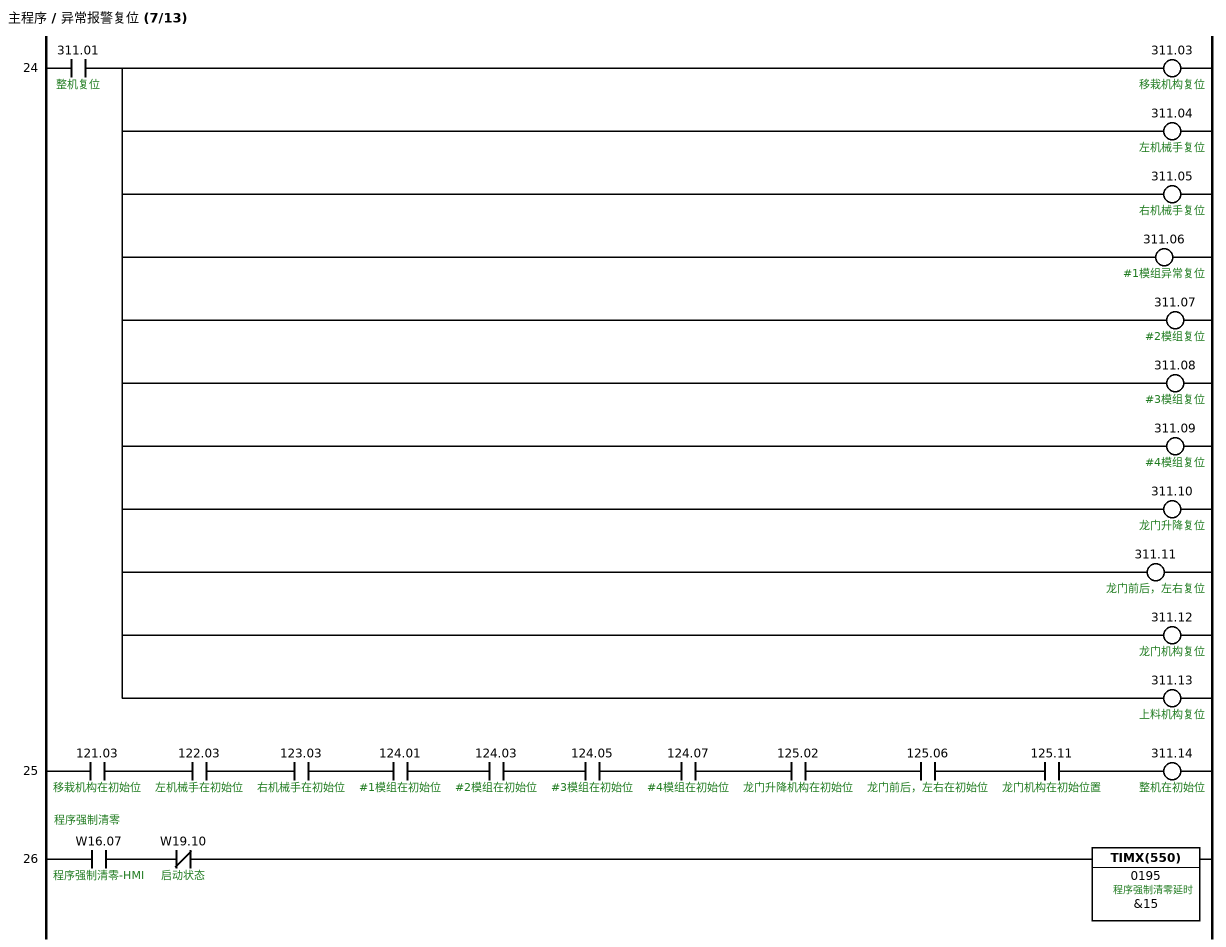
; rung 24
LD 311.01  ; 整机复位
OUT 311.03  ; 移栽机构复位
OUT 311.04  ; 左机械手复位
OUT 311.05  ; 右机械手复位
OUT 311.06  ; #1模组异常复位
OUT 311.07  ; #2模组复位
OUT 311.08  ; #3模组复位
OUT 311.09  ; #4模组复位
OUT 311.10  ; 龙门升降复位
OUT 311.11  ; 龙门前后，左右复位
OUT 311.12  ; 龙门机构复位
OUT 311.13  ; 上料机构复位
; rung 25
LD 121.03  ; 移栽机构在初始位
AND 122.03  ; 左机械手在初始位
AND 123.03  ; 右机械手在初始位
AND 124.01  ; #1模组在初始位
AND 124.03  ; #2模组在初始位
AND 124.05  ; #3模组在初始位
AND 124.07  ; #4模组在初始位
AND 125.02  ; 龙门升降机构在初始位
AND 125.06  ; 龙门前后，左右在初始位
AND 125.11  ; 龙门机构在初始位置
OUT 311.14  ; 整机在初始位
; rung 26: 程序强制清零
LD W16.07  ; 程序强制清零-HMI
ANDNOT W19.10  ; 启动状态
TIMX(550) 0195 &15  ; 程序强制清零延时

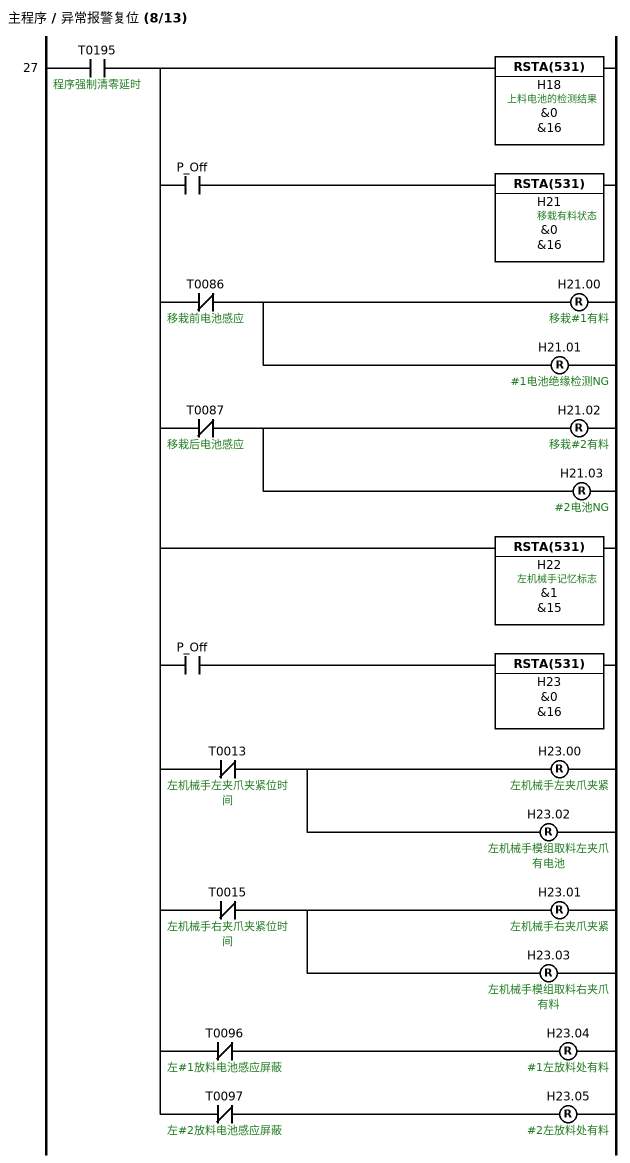
; rung 27
LD T0195  ; 程序强制清零延时
OUT TR0
RSTA(531) H18 &0 &16  ; 上料电池的检测结果
AND P_Off
RSTA(531) H21 &0 &16  ; 移栽有料状态
LD TR0
ANDNOT T0086  ; 移栽前电池感应
RSET H21.00  ; 移栽#1有料
RSET H21.01  ; #1电池绝缘检测NG
LD TR0
ANDNOT T0087  ; 移栽后电池感应
RSET H21.02  ; 移栽#2有料
RSET H21.03  ; #2电池NG
LD TR0
RSTA(531) H22 &1 &15  ; 左机械手记忆标志
AND P_Off
RSTA(531) H23 &0 &16
LD TR0
ANDNOT T0013  ; 左机械手左夹爪夹紧位时间
RSET H23.00  ; 左机械手左夹爪夹紧
RSET H23.02  ; 左机械手模组取料左夹爪有电池
LD TR0
ANDNOT T0015  ; 左机械手右夹爪夹紧位时间
RSET H23.01  ; 左机械手右夹爪夹紧
RSET H23.03  ; 左机械手模组取料右夹爪有料
LD TR0
ANDNOT T0096  ; 左#1放料电池感应屏蔽
RSET H23.04  ; #1左放料处有料
LD TR0
ANDNOT T0097  ; 左#2放料电池感应屏蔽
RSET H23.05  ; #2左放料处有料

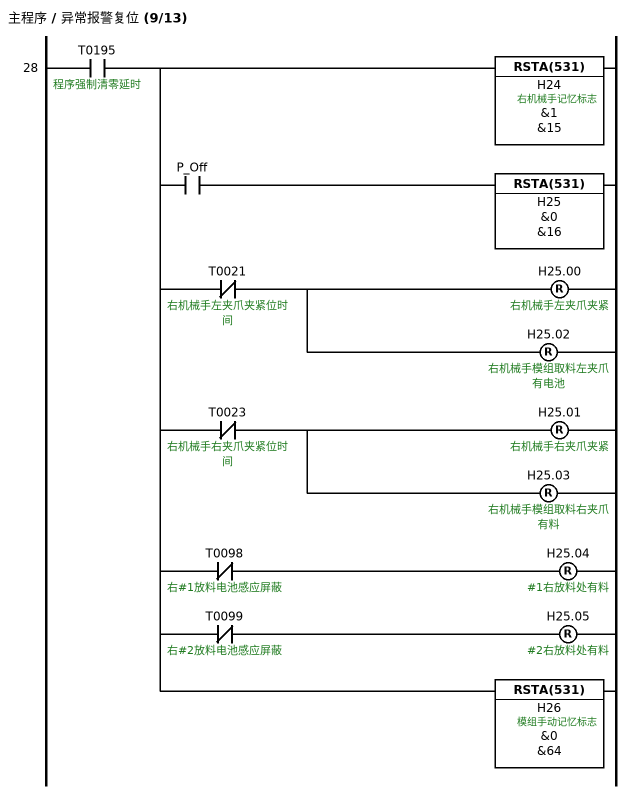
; rung 28
LD T0195  ; 程序强制清零延时
OUT TR0
RSTA(531) H24 &1 &15  ; 右机械手记忆标志
AND P_Off
RSTA(531) H25 &0 &16
LD TR0
ANDNOT T0021  ; 右机械手左夹爪夹紧位时间
RSET H25.00  ; 右机械手左夹爪夹紧
RSET H25.02  ; 右机械手模组取料左夹爪有电池
LD TR0
ANDNOT T0023  ; 右机械手右夹爪夹紧位时间
RSET H25.01  ; 右机械手右夹爪夹紧
RSET H25.03  ; 右机械手模组取料右夹爪有料
LD TR0
ANDNOT T0098  ; 右#1放料电池感应屏蔽
RSET H25.04  ; #1右放料处有料
LD TR0
ANDNOT T0099  ; 右#2放料电池感应屏蔽
RSET H25.05  ; #2右放料处有料
LD TR0
RSTA(531) H26 &0 &64  ; 模组手动记忆标志

